REGION Network 33: ET01 - ESTADO REPOSO VACIO
   RUNG wire#powerrail
      Contact( #Mx_ET00 )
      Contact( #EstadoZona.Marcha_CBx )
      I_Contact( #EstadoZona.PerReset_CBx )
      I_Contact( #pHsMx_MQ1 )
      I_Contact( #pHsMx_MQ2 )
      wire#w1
      S_SR(operand := #Mx_ET01, r1 := wire#w2)
   END_RUNG
   RUNG wire#powerrail
      Contact( #Mx_ET51 )
      Contact( #Mx_ET151 )
      I_Contact( #Mx_ET50 )
      I_Contact( #Mx_ET150 )
      I_Contact( #Simultaneo_Mx )
      I_Contact( #EstadoVI.Descarga_Act )
      I_Contact( #pHsMx_MQ1 )
      I_Contact( #pHsMx_MQ2 )
      I_Contact( #Selec_Salida_MQ1_2 )
      I_Contact( #Selec_Salida_MQ1 )
      I_Contact( #Selec_Salida_MQ2 )
   END_RUNG wire#w1
   RUNG wire#powerrail
      Contact( #Mx_ET10 )
      Contact( #Mx_ET110 )
   END_RUNG wire#w2
   // the same network as SCL:
   IF (#Mx_ET00 AND #EstadoZona.Marcha_CBx AND NOT #EstadoZona.PerReset_CBx AND NOT #pHsMx_MQ1 AND NOT #pHsMx_MQ2) OR (#Mx_ET51 AND #Mx_ET151 AND NOT #Mx_ET50 AND NOT #Mx_ET150 AND NOT #Simultaneo_Mx AND NOT #EstadoVI.Descarga_Act AND NOT #pHsMx_MQ1 AND NOT #pHsMx_MQ2 AND NOT #Selec_Salida_MQ1_2 AND NOT #Selec_Salida_MQ1 AND NOT #Selec_Salida_MQ2) THEN
       #Mx_ET01 := TRUE;   // SR flip-flop
   END_IF;
   IF #Mx_ET10 AND #Mx_ET110 THEN #Mx_ET01 := FALSE; END_IF;
END_REGION

REGION Network 34: ET00 - ESTADO DE INICIO
   RUNG wire#powerrail
      I_Contact( #Mx_ET50 )
      I_Contact( #Mx_ET51 )
      I_Contact( #Mx_ET150 )
      I_Contact( #Mx_ET151 )
      Coil( #Aux_ET00 )
   END_RUNG
   // the same network as SCL:
   #Aux_ET00 := NOT #Mx_ET50 AND NOT #Mx_ET51 AND NOT #Mx_ET150 AND NOT #Mx_ET151;
END_REGION

REGION Network 35: ----
   RUNG wire#powerrail
      Contact( #Aux_ET00 )
      I_Contact( #Mx_ET10 )
      I_Contact( #Mx_ET11 )
      I_Contact( #Mx_ET12 )
      I_Contact( #Mx_ET110 )
      I_Contact( #Mx_ET111 )
      Coil( #Aux_ET00 )
   END_RUNG
   // the same network as SCL:
   #Aux_ET00 := #Aux_ET00 AND NOT #Mx_ET10 AND NOT #Mx_ET11 AND NOT #Mx_ET12 AND NOT #Mx_ET110 AND NOT #Mx_ET111;
END_REGION

REGION Network 36: ----
   RUNG wire#powerrail
      Contact( #Aux_ET00 )
      I_Contact( #Mx_ET00 )
      I_Contact( #Mx_ET01 )
      I_Contact( #Mx_ET02 )
      I_Contact( #Mx_ET06 )
      I_Contact( #Mx_ET07 )
      I_Contact( #Mx_ET08 )
      I_Contact( #Mx_ET09 )
      S_SR(operand := #Mx_ET00, r1 := wire#w1)
   END_RUNG
   RUNG wire#powerrail
      Contact( #Mx_ET01 )
   END_RUNG wire#w1
   RUNG wire#powerrail
      Contact( #Mx_ET06 )
   END_RUNG wire#w1
   // the same network as SCL:
   IF #Aux_ET00 AND NOT #Mx_ET00 AND NOT #Mx_ET01 AND NOT #Mx_ET02 AND NOT #Mx_ET06 AND NOT #Mx_ET07 AND NOT #Mx_ET08 AND NOT #Mx_ET09 THEN
       #Mx_ET00 := TRUE;   // SR flip-flop
   END_IF;
   IF #Mx_ET01 OR #Mx_ET06 THEN #Mx_ET00 := FALSE; END_IF;
END_REGION

REGION Network 37: CONTADOR DE SEGURIDAD DE PRESENCIA - CNTSeg_pHsMx
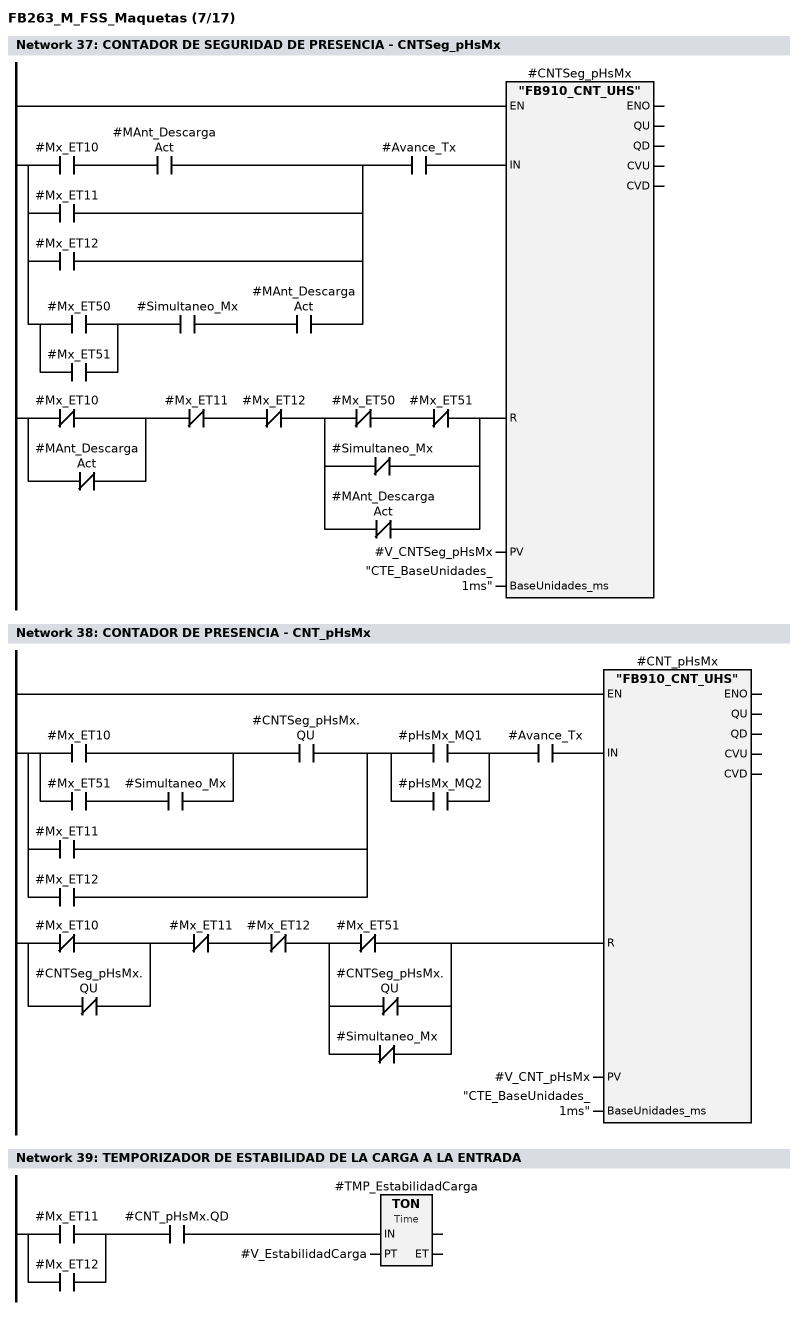
   RUNG wire#powerrail
      #CNTSeg_pHsMx(IN := wire#w3, R := wire#w6, PV := #V_CNTSeg_pHsMx, BaseUnidades_ms := "CTE_BaseUnidades_1ms", QU =>, QD =>, CVU =>, CVD =>)
   END_RUNG
   RUNG wire#powerrail
      Contact( #Mx_ET10 )
      Contact( #MAnt_DescargaAct )
      wire#w1
      Contact( #Avance_Tx )
   END_RUNG wire#w3
   RUNG wire#powerrail
      Contact( #Mx_ET11 )
   END_RUNG wire#w1
   RUNG wire#powerrail
      Contact( #Mx_ET12 )
   END_RUNG wire#w1
   RUNG wire#powerrail
      Contact( #Mx_ET50 )
      wire#w2
      Contact( #Simultaneo_Mx )
      Contact( #MAnt_DescargaAct )
   END_RUNG wire#w1
   RUNG wire#powerrail
      Contact( #Mx_ET51 )
   END_RUNG wire#w2
   RUNG wire#powerrail
      I_Contact( #Mx_ET10 )
      wire#w4
      I_Contact( #Mx_ET11 )
      I_Contact( #Mx_ET12 )
      wire#w5
      I_Contact( #Mx_ET50 )
      I_Contact( #Mx_ET51 )
   END_RUNG wire#w6
   RUNG wire#powerrail
      I_Contact( #MAnt_DescargaAct )
   END_RUNG wire#w4
   RUNG wire#w5
      I_Contact( #Simultaneo_Mx )
   END_RUNG wire#w6
   RUNG wire#w5
      I_Contact( #MAnt_DescargaAct )
   END_RUNG wire#w6
   // the same network as SCL:
   #CNTSeg_pHsMx(IN := ((#Mx_ET10 AND #MAnt_DescargaAct) OR #Mx_ET11 OR #Mx_ET12 OR ((#Mx_ET50 OR #Mx_ET51) AND #Simultaneo_Mx AND #MAnt_DescargaAct)) AND #Avance_Tx,   // "FB910_CNT_UHS"
                 R := (NOT #Mx_ET10 OR NOT #MAnt_DescargaAct) AND NOT #Mx_ET11 AND NOT #Mx_ET12 AND ((NOT #Mx_ET50 AND NOT #Mx_ET51) OR NOT #Simultaneo_Mx OR NOT #MAnt_DescargaAct),
                 PV := #V_CNTSeg_pHsMx,
                 BaseUnidades_ms := "CTE_BaseUnidades_1ms");
END_REGION

REGION Network 38: CONTADOR DE PRESENCIA - CNT_pHsMx
   RUNG wire#powerrail
      #CNT_pHsMx(IN := wire#w4, R := wire#w7, PV := #V_CNT_pHsMx, BaseUnidades_ms := "CTE_BaseUnidades_1ms", QU =>, QD =>, CVU =>, CVD =>)
   END_RUNG
   RUNG wire#powerrail
      Contact( #Mx_ET10 )
      wire#w1
      Contact( #CNTSeg_pHsMx.QU )
      wire#w2
      Contact( #pHsMx_MQ1 )
      wire#w3
      Contact( #Avance_Tx )
   END_RUNG wire#w4
   RUNG wire#powerrail
      Contact( #Mx_ET51 )
      Contact( #Simultaneo_Mx )
   END_RUNG wire#w1
   RUNG wire#powerrail
      Contact( #Mx_ET11 )
   END_RUNG wire#w2
   RUNG wire#powerrail
      Contact( #Mx_ET12 )
   END_RUNG wire#w2
   RUNG wire#w2
      Contact( #pHsMx_MQ2 )
   END_RUNG wire#w3
   RUNG wire#powerrail
      I_Contact( #Mx_ET10 )
      wire#w5
      I_Contact( #Mx_ET11 )
      I_Contact( #Mx_ET12 )
      wire#w6
      I_Contact( #Mx_ET51 )
   END_RUNG wire#w7
   RUNG wire#powerrail
      I_Contact( #CNTSeg_pHsMx.QU )
   END_RUNG wire#w5
   RUNG wire#w6
      I_Contact( #CNTSeg_pHsMx.QU )
   END_RUNG wire#w7
   RUNG wire#w6
      I_Contact( #Simultaneo_Mx )
   END_RUNG wire#w7
   // the same network as SCL:
   #CNT_pHsMx(IN := (((#Mx_ET10 OR (#Mx_ET51 AND #Simultaneo_Mx)) AND #CNTSeg_pHsMx.QU) OR #Mx_ET11 OR #Mx_ET12) AND (#pHsMx_MQ1 OR #pHsMx_MQ2) AND #Avance_Tx,   // "FB910_CNT_UHS"
              R := (NOT #Mx_ET10 OR NOT #CNTSeg_pHsMx.QU) AND NOT #Mx_ET11 AND NOT #Mx_ET12 AND (NOT #Mx_ET51 OR NOT #CNTSeg_pHsMx.QU OR NOT #Simultaneo_Mx),
              PV := #V_CNT_pHsMx,
              BaseUnidades_ms := "CTE_BaseUnidades_1ms");
END_REGION

REGION Network 39: TEMPORIZADOR DE ESTABILIDAD DE LA CARGA A LA ENTRADA
   RUNG wire#powerrail
      Contact( #Mx_ET11 )
      wire#w1
      Contact( #CNT_pHsMx.QD )
      { S7_Templates := "time_type := Time" } #TMP_EstabilidadCarga.TON(pt := #V_EstabilidadCarga, et =>)
   END_RUNG
   RUNG wire#powerrail
      Contact( #Mx_ET12 )
   END_RUNG wire#w1
   // the same network as SCL:
   #TMP_EstabilidadCarga(IN := (#Mx_ET11 OR #Mx_ET12) AND #CNT_pHsMx.QD, PT := #V_EstabilidadCarga);   // TON
END_REGION

REGION Network 40: DETERMINA PASO ET10 - ET11 (Nota: Control de Tiempo para dar el FTF a la Mesa Anterior)
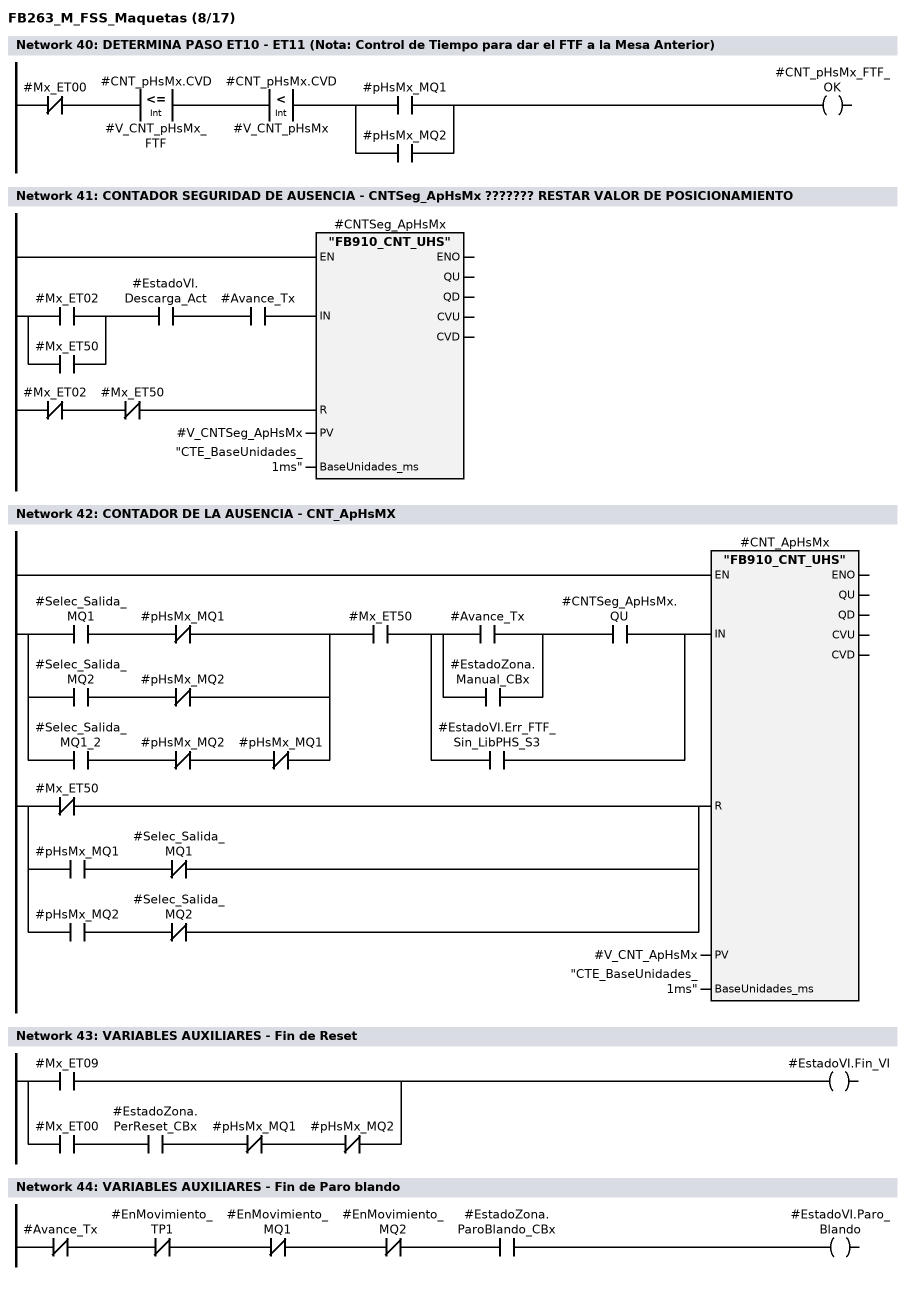
   RUNG wire#powerrail
      I_Contact( #Mx_ET00 )
      { S7_Templates := "SrcType := Int" } LE_Contact(in1 := #CNT_pHsMx.CVD, in2 := #V_CNT_pHsMx_FTF)
      { S7_Templates := "SrcType := Int" } LT_Contact(in1 := #CNT_pHsMx.CVD, in2 := #V_CNT_pHsMx)
      wire#w1
      Contact( #pHsMx_MQ1 )
      wire#w2
      Coil( #CNT_pHsMx_FTF_OK )
   END_RUNG
   RUNG wire#w1
      Contact( #pHsMx_MQ2 )
   END_RUNG wire#w2
   // the same network as SCL:
   #CNT_pHsMx_FTF_OK := NOT #Mx_ET00 AND (#CNT_pHsMx.CVD <= #V_CNT_pHsMx_FTF) AND (#CNT_pHsMx.CVD < #V_CNT_pHsMx) AND (#pHsMx_MQ1 OR #pHsMx_MQ2);
END_REGION

REGION Network 41: CONTADOR SEGURIDAD DE AUSENCIA - CNTSeg_ApHsMx ??????? RESTAR VALOR DE POSICIONAMIENTO
   RUNG wire#powerrail
      #CNTSeg_ApHsMx(IN := wire#w2, R := wire#w3, PV := #V_CNTSeg_ApHsMx, BaseUnidades_ms := "CTE_BaseUnidades_1ms", QU =>, QD =>, CVU =>, CVD =>)
   END_RUNG
   RUNG wire#powerrail
      Contact( #Mx_ET02 )
      wire#w1
      Contact( #EstadoVI.Descarga_Act )
      Contact( #Avance_Tx )
   END_RUNG wire#w2
   RUNG wire#powerrail
      Contact( #Mx_ET50 )
   END_RUNG wire#w1
   RUNG wire#powerrail
      I_Contact( #Mx_ET02 )
      I_Contact( #Mx_ET50 )
   END_RUNG wire#w3
   // the same network as SCL:
   #CNTSeg_ApHsMx(IN := (#Mx_ET02 OR #Mx_ET50) AND #EstadoVI.Descarga_Act AND #Avance_Tx,   // "FB910_CNT_UHS"
                  R := NOT #Mx_ET02 AND NOT #Mx_ET50,
                  PV := #V_CNTSeg_ApHsMx,
                  BaseUnidades_ms := "CTE_BaseUnidades_1ms");
END_REGION

REGION Network 42: CONTADOR DE LA AUSENCIA - CNT_ApHsMX
   RUNG wire#powerrail
      #CNT_ApHsMx(IN := wire#w4, R := wire#w5, PV := #V_CNT_ApHsMx, BaseUnidades_ms := "CTE_BaseUnidades_1ms", QU =>, QD =>, CVU =>, CVD =>)
   END_RUNG
   RUNG wire#powerrail
      Contact( #Selec_Salida_MQ1 )
      I_Contact( #pHsMx_MQ1 )
      wire#w1
      Contact( #Mx_ET50 )
      wire#w2
      Contact( #Avance_Tx )
      wire#w3
      Contact( #CNTSeg_ApHsMx.QU )
   END_RUNG wire#w4
   RUNG wire#powerrail
      Contact( #Selec_Salida_MQ2 )
      I_Contact( #pHsMx_MQ2 )
   END_RUNG wire#w1
   RUNG wire#powerrail
      Contact( #Selec_Salida_MQ1_2 )
      I_Contact( #pHsMx_MQ2 )
      I_Contact( #pHsMx_MQ1 )
   END_RUNG wire#w1
   RUNG wire#w2
      Contact( #EstadoZona.Manual_CBx )
   END_RUNG wire#w3
   RUNG wire#w2
      Contact( #EstadoVI.Err_FTF_Sin_LibPHS_S3 )
   END_RUNG wire#w4
   RUNG wire#powerrail
      I_Contact( #Mx_ET50 )
   END_RUNG wire#w5
   RUNG wire#powerrail
      Contact( #pHsMx_MQ1 )
      I_Contact( #Selec_Salida_MQ1 )
   END_RUNG wire#w5
   RUNG wire#powerrail
      Contact( #pHsMx_MQ2 )
      I_Contact( #Selec_Salida_MQ2 )
   END_RUNG wire#w5
   // the same network as SCL:
   #CNT_ApHsMx(IN := ((#Selec_Salida_MQ1 AND NOT #pHsMx_MQ1) OR (#Selec_Salida_MQ2 AND NOT #pHsMx_MQ2) OR (#Selec_Salida_MQ1_2 AND NOT #pHsMx_MQ2 AND NOT #pHsMx_MQ1)) AND #Mx_ET50 AND (((#Avance_Tx OR #EstadoZona.Manual_CBx) AND #CNTSeg_ApHsMx.QU) OR #EstadoVI.Err_FTF_Sin_LibPHS_S3),   // "FB910_CNT_UHS"
               R := NOT #Mx_ET50 OR (#pHsMx_MQ1 AND NOT #Selec_Salida_MQ1) OR (#pHsMx_MQ2 AND NOT #Selec_Salida_MQ2),
               PV := #V_CNT_ApHsMx,
               BaseUnidades_ms := "CTE_BaseUnidades_1ms");
END_REGION

REGION Network 43: VARIABLES AUXILIARES - Fin de Reset
   RUNG wire#powerrail
      Contact( #Mx_ET09 )
      wire#w1
      Coil( #EstadoVI.Fin_VI )
   END_RUNG
   RUNG wire#powerrail
      Contact( #Mx_ET00 )
      Contact( #EstadoZona.PerReset_CBx )
      I_Contact( #pHsMx_MQ1 )
      I_Contact( #pHsMx_MQ2 )
   END_RUNG wire#w1
   // the same network as SCL:
   #EstadoVI.Fin_VI := #Mx_ET09 OR (#Mx_ET00 AND #EstadoZona.PerReset_CBx AND NOT #pHsMx_MQ1 AND NOT #pHsMx_MQ2);
END_REGION

REGION Network 44: VARIABLES AUXILIARES - Fin de Paro blando
   RUNG wire#powerrail
      I_Contact( #Avance_Tx )
      I_Contact( #EnMovimiento_TP1 )
      I_Contact( #EnMovimiento_MQ1 )
      I_Contact( #EnMovimiento_MQ2 )
      Contact( #EstadoZona.ParoBlando_CBx )
      Coil( #EstadoVI.Paro_Blando )
   END_RUNG
   // the same network as SCL:
   #EstadoVI.Paro_Blando := NOT #Avance_Tx AND NOT #EnMovimiento_TP1 AND NOT #EnMovimiento_MQ1 AND NOT #EnMovimiento_MQ2 AND #EstadoZona.ParoBlando_CBx;
END_REGION

REGION Network 45: VARIABLES AUXILIARES - Permiso de Entrada - PTF_MAnt_Mx
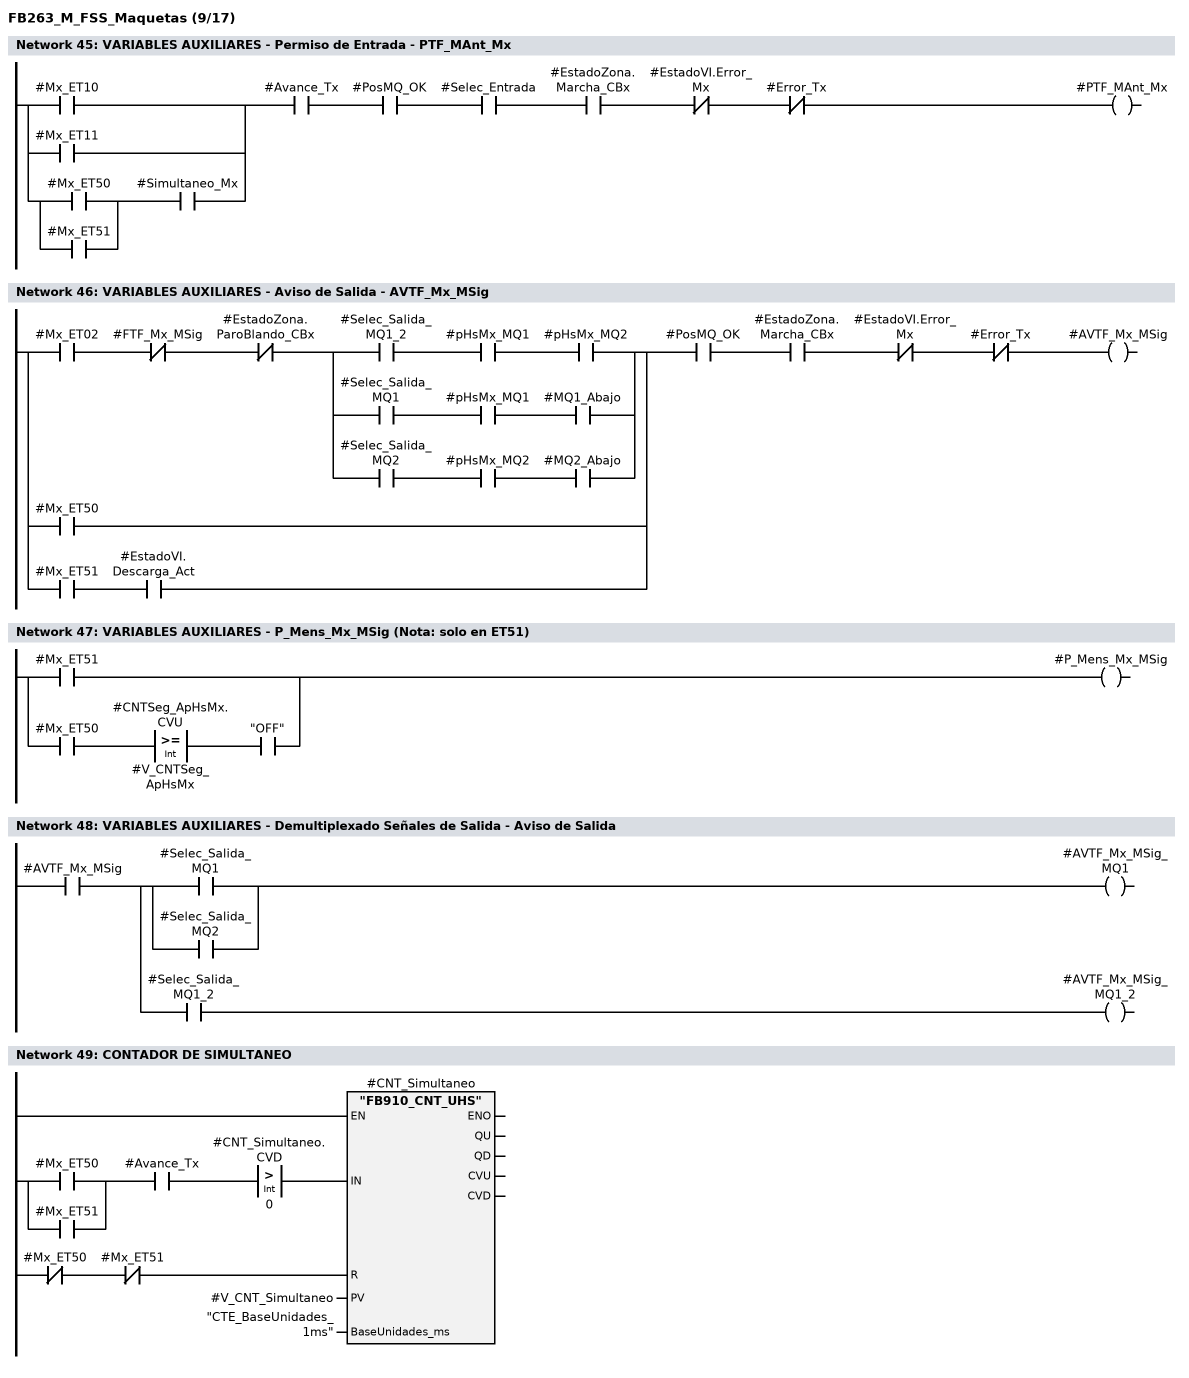
   RUNG wire#powerrail
      Contact( #Mx_ET10 )
      wire#w1
      Contact( #Avance_Tx )
      Contact( #PosMQ_OK )
      Contact( #Selec_Entrada )
      Contact( #EstadoZona.Marcha_CBx )
      I_Contact( #EstadoVI.Error_Mx )
      I_Contact( #Error_Tx )
      Coil( #PTF_MAnt_Mx )
   END_RUNG
   RUNG wire#powerrail
      Contact( #Mx_ET11 )
   END_RUNG wire#w1
   RUNG wire#powerrail
      Contact( #Mx_ET50 )
      wire#w2
      Contact( #Simultaneo_Mx )
   END_RUNG wire#w1
   RUNG wire#powerrail
      Contact( #Mx_ET51 )
   END_RUNG wire#w2
   // the same network as SCL:
   #PTF_MAnt_Mx := (#Mx_ET10 OR #Mx_ET11 OR ((#Mx_ET50 OR #Mx_ET51) AND #Simultaneo_Mx)) AND #Avance_Tx AND #PosMQ_OK AND #Selec_Entrada AND #EstadoZona.Marcha_CBx AND NOT #EstadoVI.Error_Mx AND NOT #Error_Tx;
END_REGION

REGION Network 46: VARIABLES AUXILIARES - Aviso de Salida - AVTF_Mx_MSig
   RUNG wire#powerrail
      Contact( #Mx_ET02 )
      I_Contact( #FTF_Mx_MSig )
      I_Contact( #EstadoZona.ParoBlando_CBx )
      wire#w1
      Contact( #Selec_Salida_MQ1_2 )
      Contact( #pHsMx_MQ1 )
      Contact( #pHsMx_MQ2 )
      wire#w2
      Contact( #PosMQ_OK )
      Contact( #EstadoZona.Marcha_CBx )
      I_Contact( #EstadoVI.Error_Mx )
      I_Contact( #Error_Tx )
      Coil( #AVTF_Mx_MSig )
   END_RUNG
   RUNG wire#w1
      Contact( #Selec_Salida_MQ1 )
      Contact( #pHsMx_MQ1 )
      Contact( #MQ1_Abajo )
   END_RUNG wire#w2
   RUNG wire#w1
      Contact( #Selec_Salida_MQ2 )
      Contact( #pHsMx_MQ2 )
      Contact( #MQ2_Abajo )
   END_RUNG wire#w2
   RUNG wire#powerrail
      Contact( #Mx_ET50 )
   END_RUNG wire#w2
   RUNG wire#powerrail
      Contact( #Mx_ET51 )
      Contact( #EstadoVI.Descarga_Act )
   END_RUNG wire#w2
   // the same network as SCL:
   #AVTF_Mx_MSig := ((#Mx_ET02 AND NOT #FTF_Mx_MSig AND NOT #EstadoZona.ParoBlando_CBx AND ((#Selec_Salida_MQ1_2 AND #pHsMx_MQ1 AND #pHsMx_MQ2) OR (#Selec_Salida_MQ1 AND #pHsMx_MQ1 AND #MQ1_Abajo) OR (#Selec_Salida_MQ2 AND #pHsMx_MQ2 AND #MQ2_Abajo))) OR #Mx_ET50 OR (#Mx_ET51 AND #EstadoVI.Descarga_Act)) AND #PosMQ_OK AND #EstadoZona.Marcha_CBx AND NOT #EstadoVI.Error_Mx AND NOT #Error_Tx;
END_REGION

REGION Network 47: VARIABLES AUXILIARES - P_Mens_Mx_MSig (Nota: solo en ET51)
   RUNG wire#powerrail
      Contact( #Mx_ET51 )
      wire#w1
      Coil( #P_Mens_Mx_MSig )
   END_RUNG
   RUNG wire#powerrail
      Contact( #Mx_ET50 )
      { S7_Templates := "SrcType := Int" } GE_Contact(in1 := #CNTSeg_ApHsMx.CVU, in2 := #V_CNTSeg_ApHsMx)
      Contact( "OFF" )
   END_RUNG wire#w1
   // the same network as SCL:
   #P_Mens_Mx_MSig := #Mx_ET51 OR (#Mx_ET50 AND (#CNTSeg_ApHsMx.CVU >= #V_CNTSeg_ApHsMx) AND "OFF");
END_REGION

REGION Network 48: VARIABLES AUXILIARES - Demultiplexado Señales de Salida - Aviso de Salida
   RUNG wire#powerrail
      Contact( #AVTF_Mx_MSig )
      wire#w1
      Contact( #Selec_Salida_MQ1 )
      wire#w2
      Coil( #AVTF_Mx_MSig_MQ1 )
   END_RUNG
   RUNG wire#w1
      Contact( #Selec_Salida_MQ2 )
   END_RUNG wire#w2
   RUNG wire#w1
      Contact( #Selec_Salida_MQ1_2 )
      Coil( #AVTF_Mx_MSig_MQ1_2 )
   END_RUNG
   // the same network as SCL:
   #AVTF_Mx_MSig_MQ1 := #AVTF_Mx_MSig AND (#Selec_Salida_MQ1 OR #Selec_Salida_MQ2);
   #AVTF_Mx_MSig_MQ1_2 := #AVTF_Mx_MSig AND #Selec_Salida_MQ1_2;
END_REGION

REGION Network 49: CONTADOR DE SIMULTANEO
   RUNG wire#powerrail
      #CNT_Simultaneo(IN := wire#w2, R := wire#w3, PV := #V_CNT_Simultaneo, BaseUnidades_ms := "CTE_BaseUnidades_1ms", QU =>, QD =>, CVU =>, CVD =>)
   END_RUNG
   RUNG wire#powerrail
      Contact( #Mx_ET50 )
      wire#w1
      Contact( #Avance_Tx )
      { S7_Templates := "SrcType := Int" } GT_Contact(in1 := #CNT_Simultaneo.CVD, in2 := 0)
   END_RUNG wire#w2
   RUNG wire#powerrail
      Contact( #Mx_ET51 )
   END_RUNG wire#w1
   RUNG wire#powerrail
      I_Contact( #Mx_ET50 )
      I_Contact( #Mx_ET51 )
   END_RUNG wire#w3
   // the same network as SCL:
   #CNT_Simultaneo(IN := (#Mx_ET50 OR #Mx_ET51) AND #Avance_Tx AND (#CNT_Simultaneo.CVD > 0),   // "FB910_CNT_UHS"
                   R := NOT #Mx_ET50 AND NOT #Mx_ET51,
                   PV := #V_CNT_Simultaneo,
                   BaseUnidades_ms := "CTE_BaseUnidades_1ms");
END_REGION

REGION Network 50: CONTROL DE MOVIMIENTO SIMULTANEO
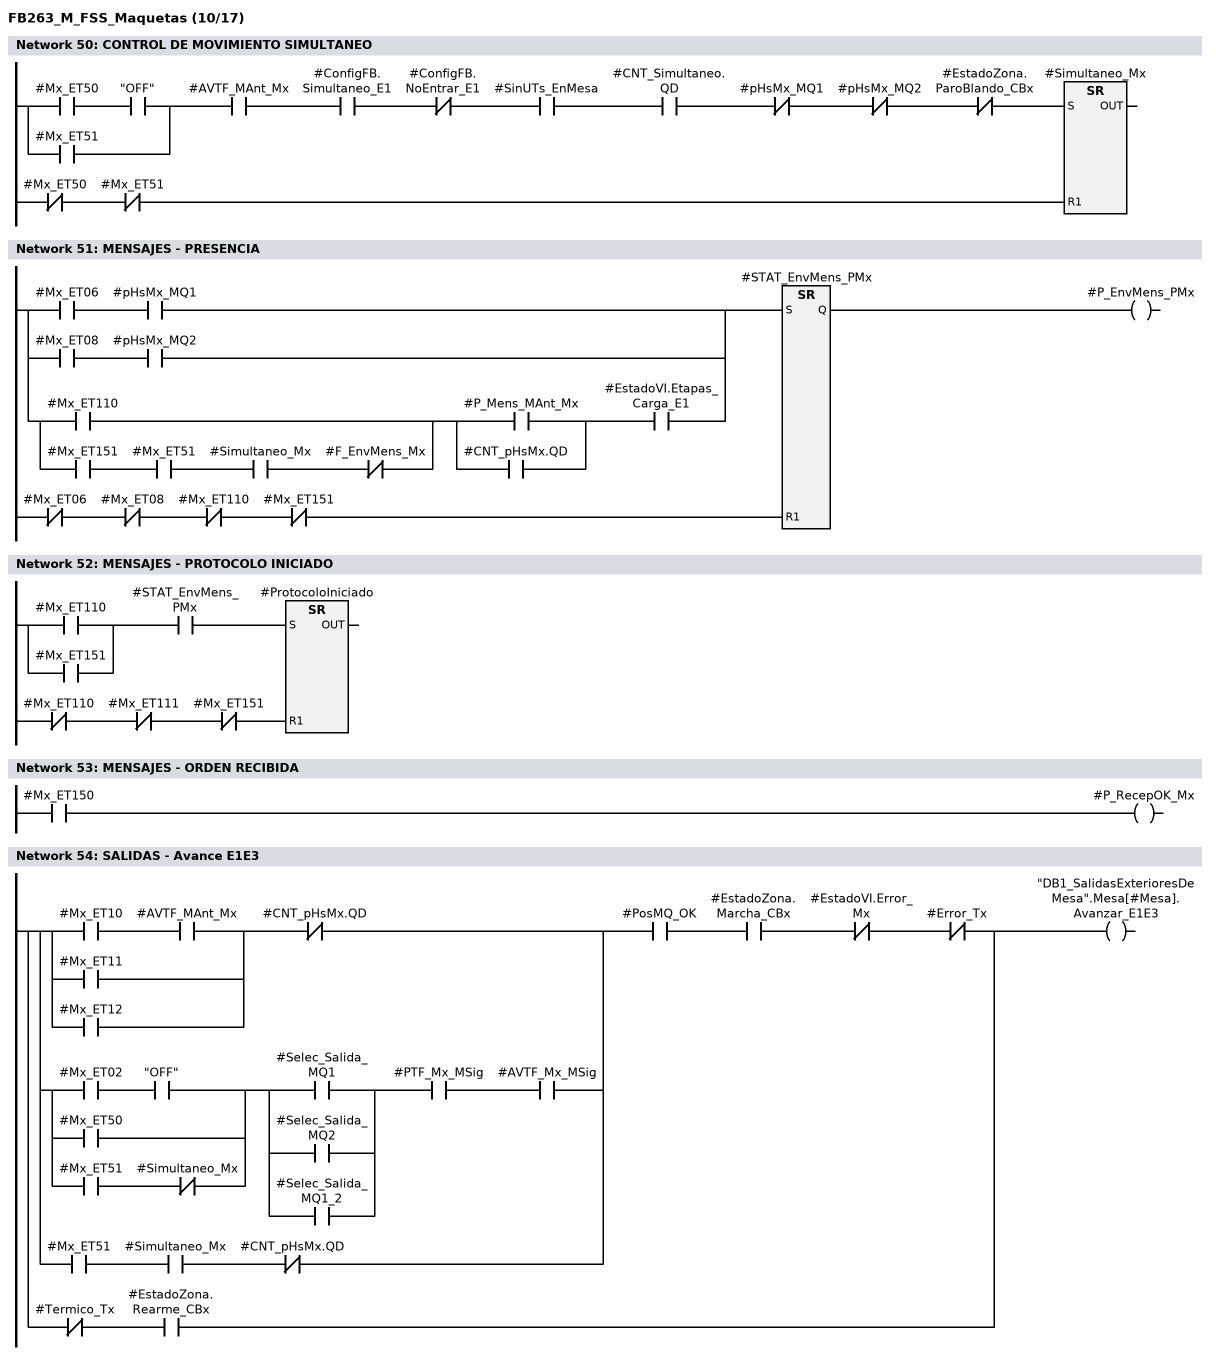
   RUNG wire#powerrail
      Contact( #Mx_ET50 )
      Contact( "OFF" )
      wire#w1
      Contact( #AVTF_MAnt_Mx )
      Contact( #ConfigFB.Simultaneo_E1 )
      I_Contact( #ConfigFB.NoEntrar_E1 )
      Contact( #SinUTs_EnMesa )
      Contact( #CNT_Simultaneo.QD )
      I_Contact( #pHsMx_MQ1 )
      I_Contact( #pHsMx_MQ2 )
      I_Contact( #EstadoZona.ParoBlando_CBx )
      S_SR(operand := #Simultaneo_Mx, r1 := wire#w2)
   END_RUNG
   RUNG wire#powerrail
      Contact( #Mx_ET51 )
   END_RUNG wire#w1
   RUNG wire#powerrail
      I_Contact( #Mx_ET50 )
      I_Contact( #Mx_ET51 )
   END_RUNG wire#w2
   // the same network as SCL:
   IF ((#Mx_ET50 AND "OFF") OR #Mx_ET51) AND #AVTF_MAnt_Mx AND #ConfigFB.Simultaneo_E1 AND NOT #ConfigFB.NoEntrar_E1 AND #SinUTs_EnMesa AND #CNT_Simultaneo.QD AND NOT #pHsMx_MQ1 AND NOT #pHsMx_MQ2 AND NOT #EstadoZona.ParoBlando_CBx THEN
       #Simultaneo_Mx := TRUE;   // SR flip-flop
   END_IF;
   IF NOT #Mx_ET50 AND NOT #Mx_ET51 THEN #Simultaneo_Mx := FALSE; END_IF;
END_REGION

REGION Network 51: MENSAJES - PRESENCIA
   RUNG wire#powerrail
      Contact( #Mx_ET06 )
      Contact( #pHsMx_MQ1 )
      wire#w1
      S_SR(operand := #STAT_EnvMens_PMx, r1 := wire#w4)
      Coil( #P_EnvMens_PMx )
   END_RUNG
   RUNG wire#powerrail
      Contact( #Mx_ET08 )
      Contact( #pHsMx_MQ2 )
   END_RUNG wire#w1
   RUNG wire#powerrail
      Contact( #Mx_ET110 )
      wire#w2
      Contact( #P_Mens_MAnt_Mx )
      wire#w3
      Contact( #EstadoVI.Etapas_Carga_E1 )
   END_RUNG wire#w1
   RUNG wire#powerrail
      Contact( #Mx_ET151 )
      Contact( #Mx_ET51 )
      Contact( #Simultaneo_Mx )
      I_Contact( #F_EnvMens_Mx )
   END_RUNG wire#w2
   RUNG wire#w2
      Contact( #CNT_pHsMx.QD )
   END_RUNG wire#w3
   RUNG wire#powerrail
      I_Contact( #Mx_ET06 )
      I_Contact( #Mx_ET08 )
      I_Contact( #Mx_ET110 )
      I_Contact( #Mx_ET151 )
   END_RUNG wire#w4
   // the same network as SCL:
   IF (#Mx_ET06 AND #pHsMx_MQ1) OR (#Mx_ET08 AND #pHsMx_MQ2) OR ((#Mx_ET110 OR (#Mx_ET151 AND #Mx_ET51 AND #Simultaneo_Mx AND NOT #F_EnvMens_Mx)) AND (#P_Mens_MAnt_Mx OR #CNT_pHsMx.QD) AND #EstadoVI.Etapas_Carga_E1) THEN
       #STAT_EnvMens_PMx := TRUE;   // SR flip-flop
   END_IF;
   IF NOT #Mx_ET06 AND NOT #Mx_ET08 AND NOT #Mx_ET110 AND NOT #Mx_ET151 THEN
       #STAT_EnvMens_PMx := FALSE;
   END_IF;
   #P_EnvMens_PMx := #STAT_EnvMens_PMx;
END_REGION

REGION Network 52: MENSAJES - PROTOCOLO INICIADO
   RUNG wire#powerrail
      Contact( #Mx_ET110 )
      wire#w1
      Contact( #STAT_EnvMens_PMx )
      S_SR(operand := #ProtocoloIniciado, r1 := wire#w2)
   END_RUNG
   RUNG wire#powerrail
      Contact( #Mx_ET151 )
   END_RUNG wire#w1
   RUNG wire#powerrail
      I_Contact( #Mx_ET110 )
      I_Contact( #Mx_ET111 )
      I_Contact( #Mx_ET151 )
   END_RUNG wire#w2
   // the same network as SCL:
   IF (#Mx_ET110 OR #Mx_ET151) AND #STAT_EnvMens_PMx THEN
       #ProtocoloIniciado := TRUE;   // SR flip-flop
   END_IF;
   IF NOT #Mx_ET110 AND NOT #Mx_ET111 AND NOT #Mx_ET151 THEN #ProtocoloIniciado := FALSE; END_IF;
END_REGION

REGION Network 53: MENSAJES - ORDEN RECIBIDA
   RUNG wire#powerrail
      Contact( #Mx_ET150 )
      Coil( #P_RecepOK_Mx )
   END_RUNG
   // the same network as SCL:
   #P_RecepOK_Mx := #Mx_ET150;
END_REGION

REGION Network 54: SALIDAS - Avance E1E3
   RUNG wire#powerrail
      Contact( #Mx_ET10 )
      Contact( #AVTF_MAnt_Mx )
      wire#w1
      I_Contact( #CNT_pHsMx.QD )
      wire#w2
      Contact( #PosMQ_OK )
      Contact( #EstadoZona.Marcha_CBx )
      I_Contact( #EstadoVI.Error_Mx )
      I_Contact( #Error_Tx )
      wire#w5
      Coil( "DB1_SalidasExterioresDeMesa".Mesa[#Mesa].Avanzar_E1E3 )
   END_RUNG
   RUNG wire#powerrail
      Contact( #Mx_ET11 )
   END_RUNG wire#w1
   RUNG wire#powerrail
      Contact( #Mx_ET12 )
   END_RUNG wire#w1
   RUNG wire#powerrail
      Contact( #Mx_ET02 )
      Contact( "OFF" )
      wire#w3
      Contact( #Selec_Salida_MQ1 )
      wire#w4
      Contact( #PTF_Mx_MSig )
      Contact( #AVTF_Mx_MSig )
   END_RUNG wire#w2
   RUNG wire#powerrail
      Contact( #Mx_ET50 )
   END_RUNG wire#w3
   RUNG wire#powerrail
      Contact( #Mx_ET51 )
      I_Contact( #Simultaneo_Mx )
   END_RUNG wire#w3
   RUNG wire#w3
      Contact( #Selec_Salida_MQ2 )
   END_RUNG wire#w4
   RUNG wire#w3
      Contact( #Selec_Salida_MQ1_2 )
   END_RUNG wire#w4
   RUNG wire#powerrail
      Contact( #Mx_ET51 )
      Contact( #Simultaneo_Mx )
      I_Contact( #CNT_pHsMx.QD )
   END_RUNG wire#w2
   RUNG wire#powerrail
      I_Contact( #Termico_Tx )
      Contact( #EstadoZona.Rearme_CBx )
   END_RUNG wire#w5
   // the same network as SCL:
   "DB1_SalidasExterioresDeMesa".Mesa[#Mesa].Avanzar_E1E3 := (((((#Mx_ET10 AND #AVTF_MAnt_Mx) OR #Mx_ET11 OR #Mx_ET12) AND NOT #CNT_pHsMx.QD) OR (((#Mx_ET02 AND "OFF") OR #Mx_ET50 OR (#Mx_ET51 AND NOT #Simultaneo_Mx)) AND (#Selec_Salida_MQ1 OR #Selec_Salida_MQ2 OR #Selec_Salida_MQ1_2) AND #PTF_Mx_MSig AND #AVTF_Mx_MSig) OR (#Mx_ET51 AND #Simultaneo_Mx AND NOT #CNT_pHsMx.QD)) AND #PosMQ_OK AND #EstadoZona.Marcha_CBx AND NOT #EstadoVI.Error_Mx AND NOT #Error_Tx) OR (NOT #Termico_Tx AND #EstadoZona.Rearme_CBx);
END_REGION

REGION Network 55: SALIDAS - Subir Tope (TP1)
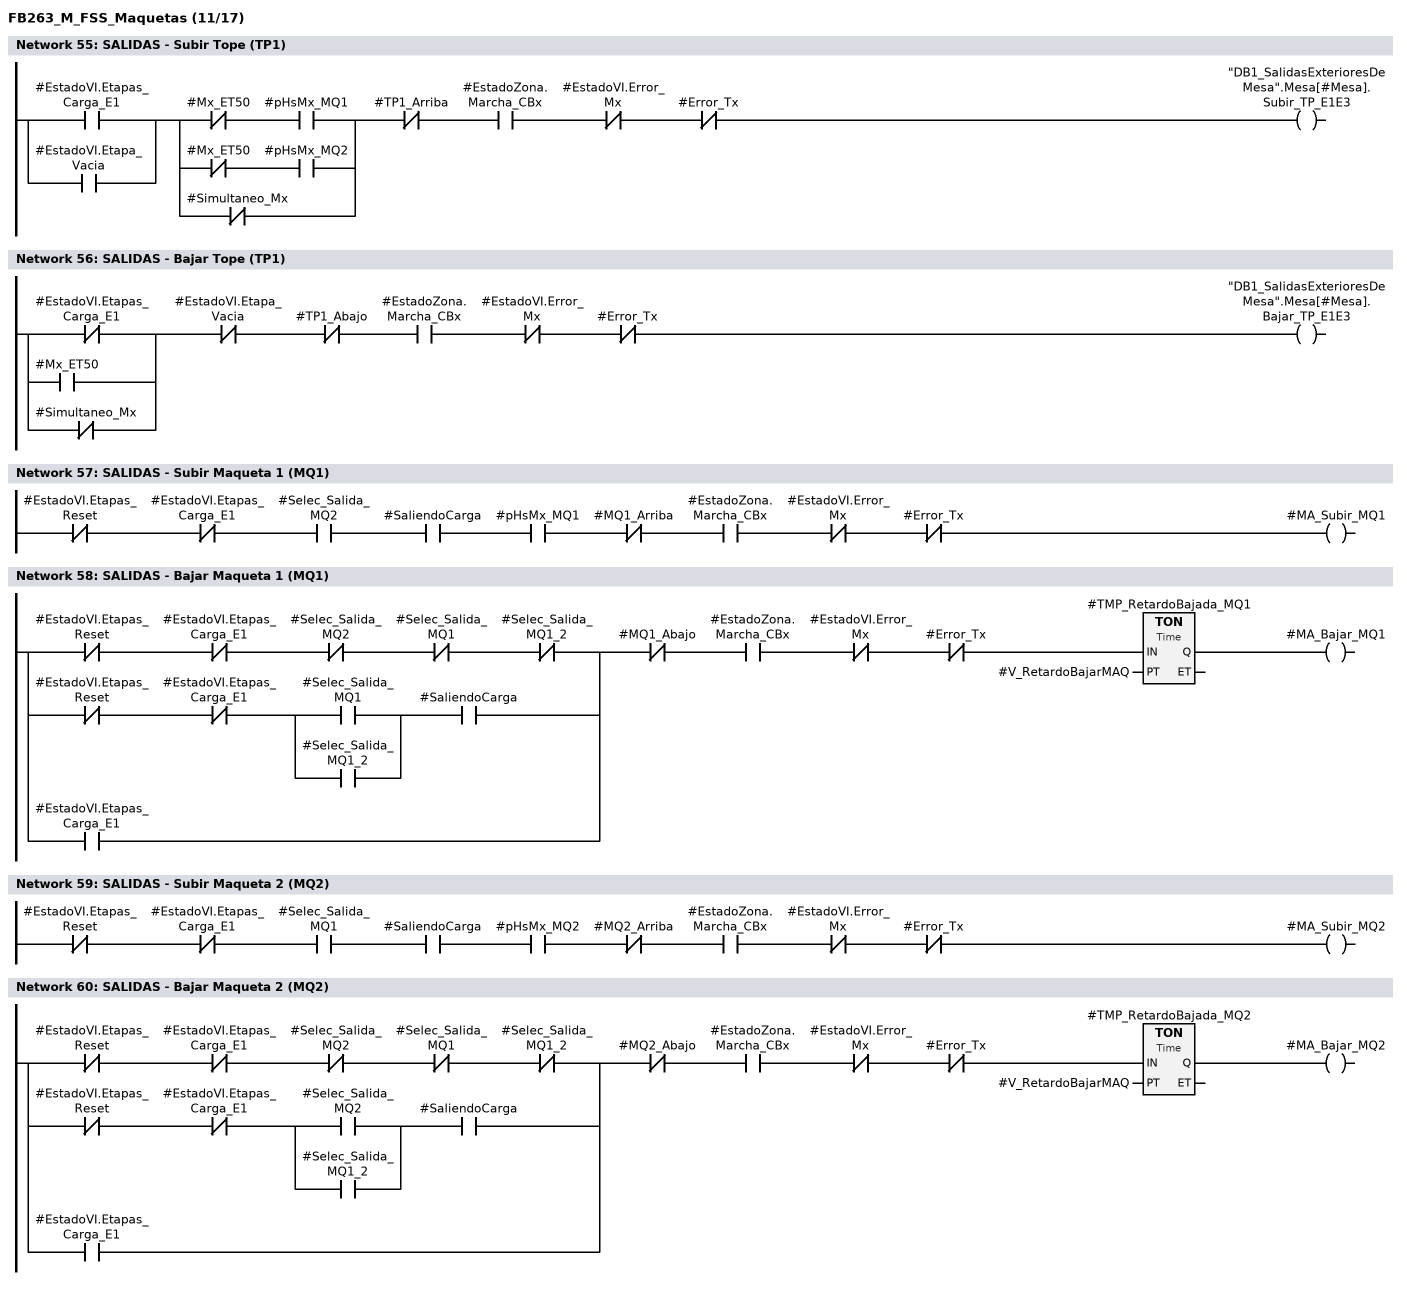
   RUNG wire#powerrail
      Contact( #EstadoVI.Etapas_Carga_E1 )
      wire#w1
      I_Contact( #Mx_ET50 )
      Contact( #pHsMx_MQ1 )
      wire#w2
      I_Contact( #TP1_Arriba )
      Contact( #EstadoZona.Marcha_CBx )
      I_Contact( #EstadoVI.Error_Mx )
      I_Contact( #Error_Tx )
      Coil( "DB1_SalidasExterioresDeMesa".Mesa[#Mesa].Subir_TP_E1E3 )
   END_RUNG
   RUNG wire#powerrail
      Contact( #EstadoVI.Etapa_Vacia )
   END_RUNG wire#w1
   RUNG wire#w1
      I_Contact( #Mx_ET50 )
      Contact( #pHsMx_MQ2 )
   END_RUNG wire#w2
   RUNG wire#w1
      I_Contact( #Simultaneo_Mx )
   END_RUNG wire#w2
   // the same network as SCL:
   "DB1_SalidasExterioresDeMesa".Mesa[#Mesa].Subir_TP_E1E3 := (#EstadoVI.Etapas_Carga_E1 OR #EstadoVI.Etapa_Vacia) AND ((NOT #Mx_ET50 AND #pHsMx_MQ1) OR (NOT #Mx_ET50 AND #pHsMx_MQ2) OR NOT #Simultaneo_Mx) AND NOT #TP1_Arriba AND #EstadoZona.Marcha_CBx AND NOT #EstadoVI.Error_Mx AND NOT #Error_Tx;
END_REGION

REGION Network 56: SALIDAS - Bajar Tope (TP1)
   RUNG wire#powerrail
      I_Contact( #EstadoVI.Etapas_Carga_E1 )
      wire#w1
      I_Contact( #EstadoVI.Etapa_Vacia )
      I_Contact( #TP1_Abajo )
      Contact( #EstadoZona.Marcha_CBx )
      I_Contact( #EstadoVI.Error_Mx )
      I_Contact( #Error_Tx )
      Coil( "DB1_SalidasExterioresDeMesa".Mesa[#Mesa].Bajar_TP_E1E3 )
   END_RUNG
   RUNG wire#powerrail
      Contact( #Mx_ET50 )
   END_RUNG wire#w1
   RUNG wire#powerrail
      I_Contact( #Simultaneo_Mx )
   END_RUNG wire#w1
   // the same network as SCL:
   "DB1_SalidasExterioresDeMesa".Mesa[#Mesa].Bajar_TP_E1E3 := (NOT #EstadoVI.Etapas_Carga_E1 OR #Mx_ET50 OR NOT #Simultaneo_Mx) AND NOT #EstadoVI.Etapa_Vacia AND NOT #TP1_Abajo AND #EstadoZona.Marcha_CBx AND NOT #EstadoVI.Error_Mx AND NOT #Error_Tx;
END_REGION

REGION Network 57: SALIDAS - Subir Maqueta 1 (MQ1)
   RUNG wire#powerrail
      I_Contact( #EstadoVI.Etapas_Reset )
      I_Contact( #EstadoVI.Etapas_Carga_E1 )
      Contact( #Selec_Salida_MQ2 )
      Contact( #SaliendoCarga )
      Contact( #pHsMx_MQ1 )
      I_Contact( #MQ1_Arriba )
      Contact( #EstadoZona.Marcha_CBx )
      I_Contact( #EstadoVI.Error_Mx )
      I_Contact( #Error_Tx )
      Coil( #MA_Subir_MQ1 )
   END_RUNG
   // the same network as SCL:
   #MA_Subir_MQ1 := NOT #EstadoVI.Etapas_Reset AND NOT #EstadoVI.Etapas_Carga_E1 AND #Selec_Salida_MQ2 AND #SaliendoCarga AND #pHsMx_MQ1 AND NOT #MQ1_Arriba AND #EstadoZona.Marcha_CBx AND NOT #EstadoVI.Error_Mx AND NOT #Error_Tx;
END_REGION

REGION Network 58: SALIDAS - Bajar Maqueta 1 (MQ1)
   RUNG wire#powerrail
      I_Contact( #EstadoVI.Etapas_Reset )
      I_Contact( #EstadoVI.Etapas_Carga_E1 )
      I_Contact( #Selec_Salida_MQ2 )
      I_Contact( #Selec_Salida_MQ1 )
      I_Contact( #Selec_Salida_MQ1_2 )
      wire#w1
      I_Contact( #MQ1_Abajo )
      Contact( #EstadoZona.Marcha_CBx )
      I_Contact( #EstadoVI.Error_Mx )
      I_Contact( #Error_Tx )
      { S7_Templates := "time_type := Time" } #TMP_RetardoBajada_MQ1.TON(pt := #V_RetardoBajarMAQ, et =>)
      Coil( #MA_Bajar_MQ1 )
   END_RUNG
   RUNG wire#powerrail
      I_Contact( #EstadoVI.Etapas_Reset )
      I_Contact( #EstadoVI.Etapas_Carga_E1 )
      wire#w2
      Contact( #Selec_Salida_MQ1 )
      wire#w3
      Contact( #SaliendoCarga )
   END_RUNG wire#w1
   RUNG wire#w2
      Contact( #Selec_Salida_MQ1_2 )
   END_RUNG wire#w3
   RUNG wire#powerrail
      Contact( #EstadoVI.Etapas_Carga_E1 )
   END_RUNG wire#w1
   // the same network as SCL:
   #TMP_RetardoBajada_MQ1(IN := ((NOT #EstadoVI.Etapas_Reset AND NOT #EstadoVI.Etapas_Carga_E1 AND NOT #Selec_Salida_MQ2 AND NOT #Selec_Salida_MQ1 AND NOT #Selec_Salida_MQ1_2) OR (NOT #EstadoVI.Etapas_Reset AND NOT #EstadoVI.Etapas_Carga_E1 AND (#Selec_Salida_MQ1 OR #Selec_Salida_MQ1_2) AND #SaliendoCarga) OR #EstadoVI.Etapas_Carga_E1) AND NOT #MQ1_Abajo AND #EstadoZona.Marcha_CBx AND NOT #EstadoVI.Error_Mx AND NOT #Error_Tx,   // TON
                          PT := #V_RetardoBajarMAQ);
   #MA_Bajar_MQ1 := #TMP_RetardoBajada_MQ1.Q;
END_REGION

REGION Network 59: SALIDAS - Subir Maqueta 2 (MQ2)
   RUNG wire#powerrail
      I_Contact( #EstadoVI.Etapas_Reset )
      I_Contact( #EstadoVI.Etapas_Carga_E1 )
      Contact( #Selec_Salida_MQ1 )
      Contact( #SaliendoCarga )
      Contact( #pHsMx_MQ2 )
      I_Contact( #MQ2_Arriba )
      Contact( #EstadoZona.Marcha_CBx )
      I_Contact( #EstadoVI.Error_Mx )
      I_Contact( #Error_Tx )
      Coil( #MA_Subir_MQ2 )
   END_RUNG
   // the same network as SCL:
   #MA_Subir_MQ2 := NOT #EstadoVI.Etapas_Reset AND NOT #EstadoVI.Etapas_Carga_E1 AND #Selec_Salida_MQ1 AND #SaliendoCarga AND #pHsMx_MQ2 AND NOT #MQ2_Arriba AND #EstadoZona.Marcha_CBx AND NOT #EstadoVI.Error_Mx AND NOT #Error_Tx;
END_REGION

REGION Network 60: SALIDAS - Bajar Maqueta 2 (MQ2)
   RUNG wire#powerrail
      I_Contact( #EstadoVI.Etapas_Reset )
      I_Contact( #EstadoVI.Etapas_Carga_E1 )
      I_Contact( #Selec_Salida_MQ2 )
      I_Contact( #Selec_Salida_MQ1 )
      I_Contact( #Selec_Salida_MQ1_2 )
      wire#w1
      I_Contact( #MQ2_Abajo )
      Contact( #EstadoZona.Marcha_CBx )
      I_Contact( #EstadoVI.Error_Mx )
      I_Contact( #Error_Tx )
      { S7_Templates := "time_type := Time" } #TMP_RetardoBajada_MQ2.TON(pt := #V_RetardoBajarMAQ, et =>)
      Coil( #MA_Bajar_MQ2 )
   END_RUNG
   RUNG wire#powerrail
      I_Contact( #EstadoVI.Etapas_Reset )
      I_Contact( #EstadoVI.Etapas_Carga_E1 )
      wire#w2
      Contact( #Selec_Salida_MQ2 )
      wire#w3
      Contact( #SaliendoCarga )
   END_RUNG wire#w1
   RUNG wire#w2
      Contact( #Selec_Salida_MQ1_2 )
   END_RUNG wire#w3
   RUNG wire#powerrail
      Contact( #EstadoVI.Etapas_Carga_E1 )
   END_RUNG wire#w1
   // the same network as SCL:
   #TMP_RetardoBajada_MQ2(IN := ((NOT #EstadoVI.Etapas_Reset AND NOT #EstadoVI.Etapas_Carga_E1 AND NOT #Selec_Salida_MQ2 AND NOT #Selec_Salida_MQ1 AND NOT #Selec_Salida_MQ1_2) OR (NOT #EstadoVI.Etapas_Reset AND NOT #EstadoVI.Etapas_Carga_E1 AND (#Selec_Salida_MQ2 OR #Selec_Salida_MQ1_2) AND #SaliendoCarga) OR #EstadoVI.Etapas_Carga_E1) AND NOT #MQ2_Abajo AND #EstadoZona.Marcha_CBx AND NOT #EstadoVI.Error_Mx AND NOT #Error_Tx,   // TON
                          PT := #V_RetardoBajarMAQ);
   #MA_Bajar_MQ2 := #TMP_RetardoBajada_MQ2.Q;
END_REGION

REGION Network 61: TMP - Espera En Tension
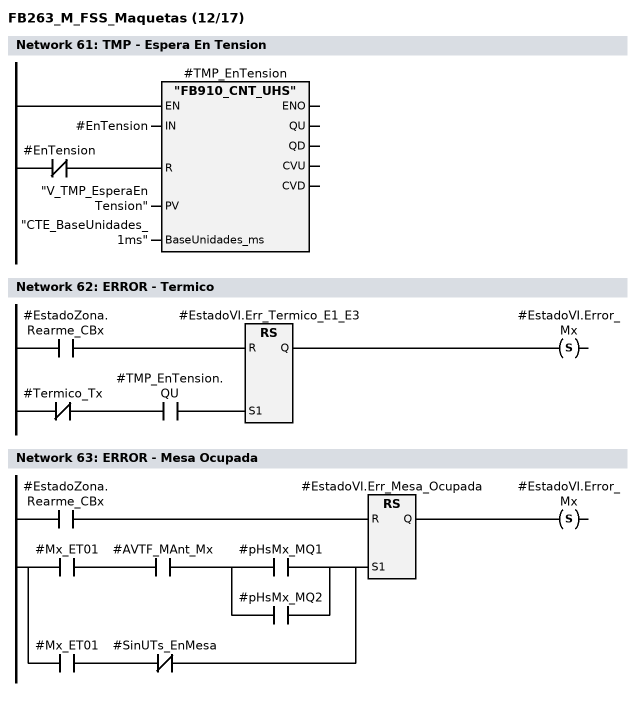
   RUNG wire#powerrail
      #TMP_EnTension(R := wire#w1, IN := #EnTension, PV := "V_TMP_EsperaEnTension", BaseUnidades_ms := "CTE_BaseUnidades_1ms", QU =>, QD =>, CVU =>, CVD =>)
   END_RUNG
   RUNG wire#powerrail
      I_Contact( #EnTension )
   END_RUNG wire#w1
   // the same network as SCL:
   #TMP_EnTension(IN := #EnTension,   // "FB910_CNT_UHS"
                  R := NOT #EnTension,
                  PV := "V_TMP_EsperaEnTension",
                  BaseUnidades_ms := "CTE_BaseUnidades_1ms");
END_REGION

REGION Network 62: ERROR - Termico
   RUNG wire#powerrail
      Contact( #EstadoZona.Rearme_CBx )
      S_RS(operand := #EstadoVI.Err_Termico_E1_E3, s1 := wire#w1)
      S_Coil( #EstadoVI.Error_Mx )
   END_RUNG
   RUNG wire#powerrail
      I_Contact( #Termico_Tx )
      Contact( #TMP_EnTension.QU )
   END_RUNG wire#w1
   // the same network as SCL:
   IF #EstadoZona.Rearme_CBx THEN
       #EstadoVI.Err_Termico_E1_E3 := FALSE;   // RS flip-flop
   END_IF;
   IF NOT #Termico_Tx AND #TMP_EnTension.QU THEN #EstadoVI.Err_Termico_E1_E3 := TRUE; END_IF;
   IF #EstadoVI.Err_Termico_E1_E3 THEN #EstadoVI.Error_Mx := TRUE; END_IF;
END_REGION

REGION Network 63: ERROR - Mesa Ocupada
   RUNG wire#powerrail
      Contact( #EstadoZona.Rearme_CBx )
      S_RS(operand := #EstadoVI.Err_Mesa_Ocupada, s1 := wire#w2)
      S_Coil( #EstadoVI.Error_Mx )
   END_RUNG
   RUNG wire#powerrail
      Contact( #Mx_ET01 )
      Contact( #AVTF_MAnt_Mx )
      wire#w1
      Contact( #pHsMx_MQ1 )
   END_RUNG wire#w2
   RUNG wire#w1
      Contact( #pHsMx_MQ2 )
   END_RUNG wire#w2
   RUNG wire#powerrail
      Contact( #Mx_ET01 )
      I_Contact( #SinUTs_EnMesa )
   END_RUNG wire#w2
   // the same network as SCL:
   IF #EstadoZona.Rearme_CBx THEN
       #EstadoVI.Err_Mesa_Ocupada := FALSE;   // RS flip-flop
   END_IF;
   IF (#Mx_ET01 AND #AVTF_MAnt_Mx AND (#pHsMx_MQ1 OR #pHsMx_MQ2)) OR (#Mx_ET01 AND NOT #SinUTs_EnMesa) THEN
       #EstadoVI.Err_Mesa_Ocupada := TRUE;
   END_IF;
   IF #EstadoVI.Err_Mesa_Ocupada THEN #EstadoVI.Error_Mx := TRUE; END_IF;
END_REGION

REGION Network 64: CNT - ERROR - Arrastre
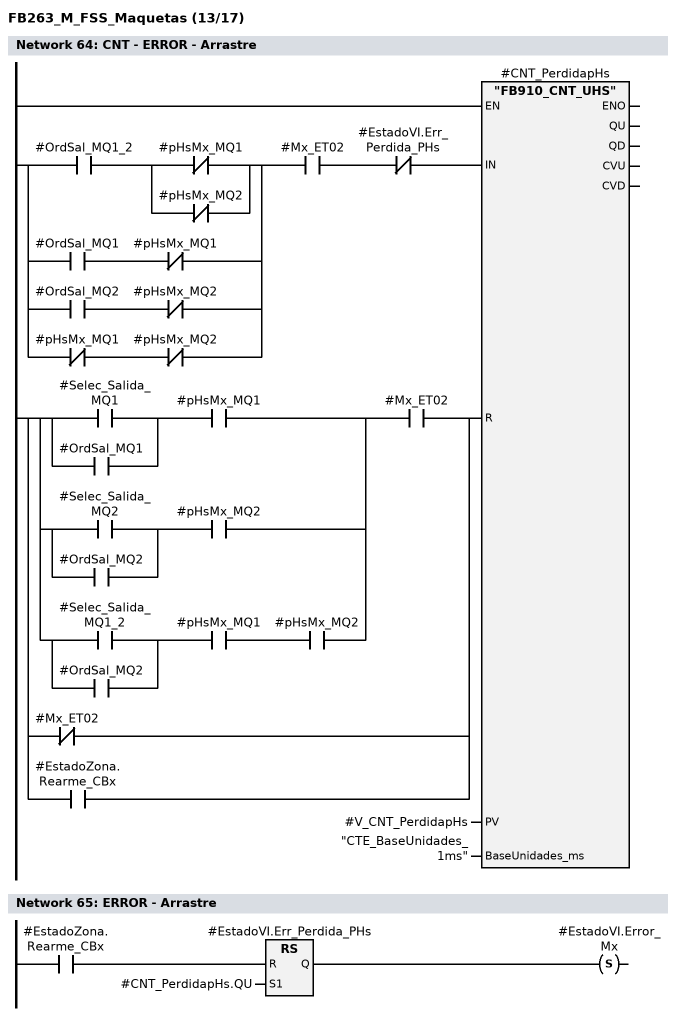
   RUNG wire#powerrail
      #CNT_PerdidapHs(IN := wire#w3, R := wire#w8, PV := #V_CNT_PerdidapHs, BaseUnidades_ms := "CTE_BaseUnidades_1ms", QU =>, QD =>, CVU =>, CVD =>)
   END_RUNG
   RUNG wire#powerrail
      Contact( #OrdSal_MQ1_2 )
      wire#w1
      I_Contact( #pHsMx_MQ1 )
      wire#w2
      Contact( #Mx_ET02 )
      I_Contact( #EstadoVI.Err_Perdida_PHs )
   END_RUNG wire#w3
   RUNG wire#w1
      I_Contact( #pHsMx_MQ2 )
   END_RUNG wire#w2
   RUNG wire#powerrail
      Contact( #OrdSal_MQ1 )
      I_Contact( #pHsMx_MQ1 )
   END_RUNG wire#w2
   RUNG wire#powerrail
      Contact( #OrdSal_MQ2 )
      I_Contact( #pHsMx_MQ2 )
   END_RUNG wire#w2
   RUNG wire#powerrail
      I_Contact( #pHsMx_MQ1 )
      I_Contact( #pHsMx_MQ2 )
   END_RUNG wire#w2
   RUNG wire#powerrail
      Contact( #Selec_Salida_MQ1 )
      wire#w4
      Contact( #pHsMx_MQ1 )
      wire#w5
      Contact( #Mx_ET02 )
   END_RUNG wire#w8
   RUNG wire#powerrail
      Contact( #OrdSal_MQ1 )
   END_RUNG wire#w4
   RUNG wire#powerrail
      Contact( #Selec_Salida_MQ2 )
      wire#w6
      Contact( #pHsMx_MQ2 )
   END_RUNG wire#w5
   RUNG wire#powerrail
      Contact( #OrdSal_MQ2 )
   END_RUNG wire#w6
   RUNG wire#powerrail
      Contact( #Selec_Salida_MQ1_2 )
      wire#w7
      Contact( #pHsMx_MQ1 )
      Contact( #pHsMx_MQ2 )
   END_RUNG wire#w5
   RUNG wire#powerrail
      Contact( #OrdSal_MQ2 )
   END_RUNG wire#w7
   RUNG wire#powerrail
      I_Contact( #Mx_ET02 )
   END_RUNG wire#w8
   RUNG wire#powerrail
      Contact( #EstadoZona.Rearme_CBx )
   END_RUNG wire#w8
   // the same network as SCL:
   #CNT_PerdidapHs(IN := ((#OrdSal_MQ1_2 AND (NOT #pHsMx_MQ1 OR NOT #pHsMx_MQ2)) OR (#OrdSal_MQ1 AND NOT #pHsMx_MQ1) OR (#OrdSal_MQ2 AND NOT #pHsMx_MQ2) OR (NOT #pHsMx_MQ1 AND NOT #pHsMx_MQ2)) AND #Mx_ET02 AND NOT #EstadoVI.Err_Perdida_PHs,   // "FB910_CNT_UHS"
                   R := ((((#Selec_Salida_MQ1 OR #OrdSal_MQ1) AND #pHsMx_MQ1) OR ((#Selec_Salida_MQ2 OR #OrdSal_MQ2) AND #pHsMx_MQ2) OR ((#Selec_Salida_MQ1_2 OR #OrdSal_MQ2) AND #pHsMx_MQ1 AND #pHsMx_MQ2)) AND #Mx_ET02) OR NOT #Mx_ET02 OR #EstadoZona.Rearme_CBx,
                   PV := #V_CNT_PerdidapHs,
                   BaseUnidades_ms := "CTE_BaseUnidades_1ms");
END_REGION

REGION Network 65: ERROR - Arrastre
   RUNG wire#powerrail
      Contact( #EstadoZona.Rearme_CBx )
      S_RS(operand := #EstadoVI.Err_Perdida_PHs, s1 := #CNT_PerdidapHs.QU)
      S_Coil( #EstadoVI.Error_Mx )
   END_RUNG
   // the same network as SCL:
   IF #EstadoZona.Rearme_CBx THEN
       #EstadoVI.Err_Perdida_PHs := FALSE;   // RS flip-flop
   END_IF;
   IF #CNT_PerdidapHs.QU THEN #EstadoVI.Err_Perdida_PHs := TRUE; END_IF;
   IF #EstadoVI.Err_Perdida_PHs THEN #EstadoVI.Error_Mx := TRUE; END_IF;
END_REGION

REGION Network 66: ERROR - Descarga por S3
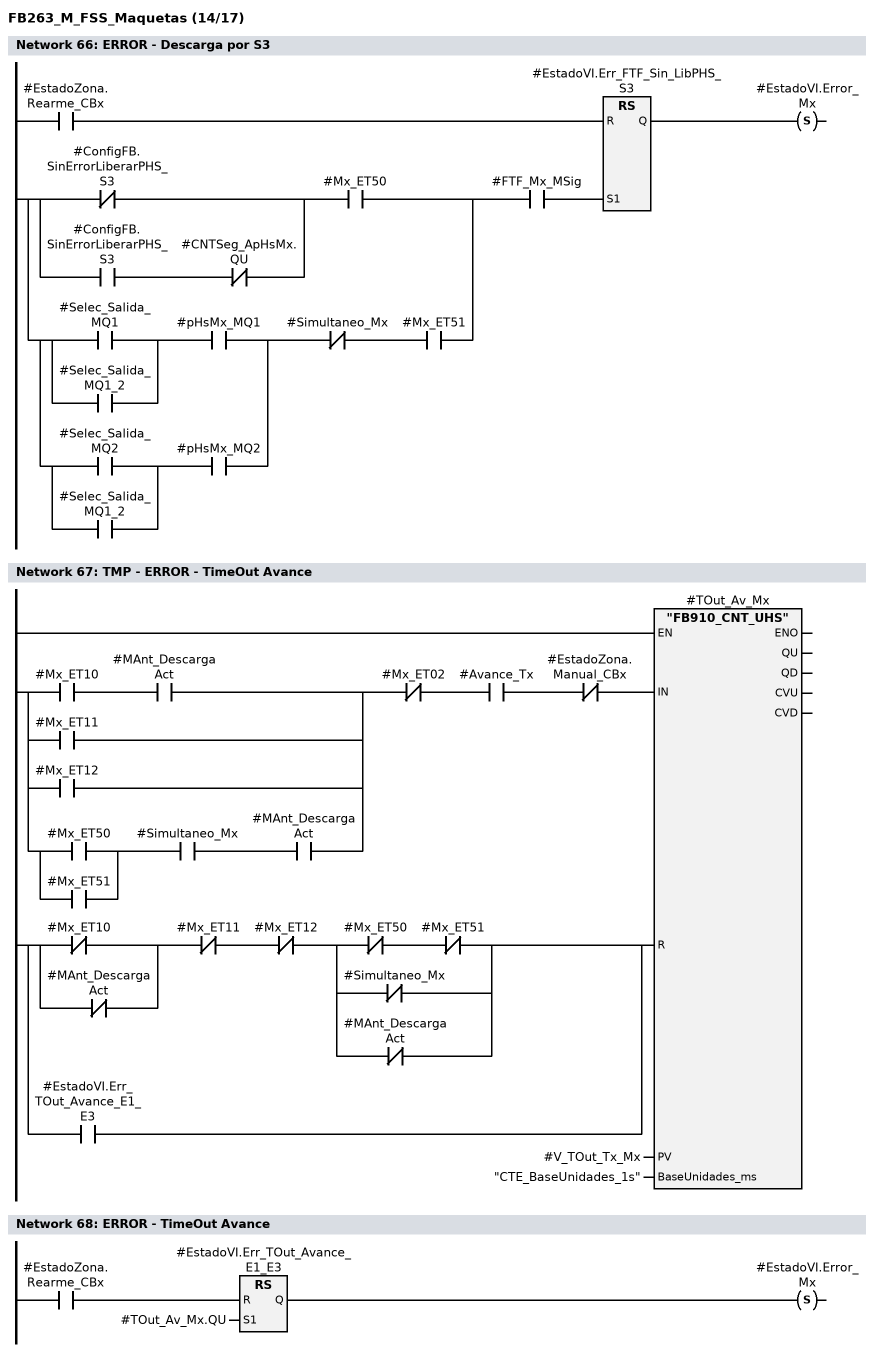
   RUNG wire#powerrail
      Contact( #EstadoZona.Rearme_CBx )
      S_RS(operand := #EstadoVI.Err_FTF_Sin_LibPHS_S3, s1 := wire#w6)
      S_Coil( #EstadoVI.Error_Mx )
   END_RUNG
   RUNG wire#powerrail
      I_Contact( #ConfigFB.SinErrorLiberarPHS_S3 )
      wire#w1
      Contact( #Mx_ET50 )
      wire#w2
      Contact( #FTF_Mx_MSig )
   END_RUNG wire#w6
   RUNG wire#powerrail
      Contact( #ConfigFB.SinErrorLiberarPHS_S3 )
      I_Contact( #CNTSeg_ApHsMx.QU )
   END_RUNG wire#w1
   RUNG wire#powerrail
      Contact( #Selec_Salida_MQ1 )
      wire#w3
      Contact( #pHsMx_MQ1 )
      wire#w4
      I_Contact( #Simultaneo_Mx )
      Contact( #Mx_ET51 )
   END_RUNG wire#w2
   RUNG wire#powerrail
      Contact( #Selec_Salida_MQ1_2 )
   END_RUNG wire#w3
   RUNG wire#powerrail
      Contact( #Selec_Salida_MQ2 )
      wire#w5
      Contact( #pHsMx_MQ2 )
   END_RUNG wire#w4
   RUNG wire#powerrail
      Contact( #Selec_Salida_MQ1_2 )
   END_RUNG wire#w5
   // the same network as SCL:
   IF #EstadoZona.Rearme_CBx THEN
       #EstadoVI.Err_FTF_Sin_LibPHS_S3 := FALSE;   // RS flip-flop
   END_IF;
   IF (((NOT #ConfigFB.SinErrorLiberarPHS_S3 OR (#ConfigFB.SinErrorLiberarPHS_S3 AND NOT #CNTSeg_ApHsMx.QU)) AND #Mx_ET50) OR ((((#Selec_Salida_MQ1 OR #Selec_Salida_MQ1_2) AND #pHsMx_MQ1) OR ((#Selec_Salida_MQ2 OR #Selec_Salida_MQ1_2) AND #pHsMx_MQ2)) AND NOT #Simultaneo_Mx AND #Mx_ET51)) AND #FTF_Mx_MSig THEN
       #EstadoVI.Err_FTF_Sin_LibPHS_S3 := TRUE;
   END_IF;
   IF #EstadoVI.Err_FTF_Sin_LibPHS_S3 THEN #EstadoVI.Error_Mx := TRUE; END_IF;
END_REGION

REGION Network 67: TMP - ERROR - TimeOut Avance
   RUNG wire#powerrail
      #TOut_Av_Mx(IN := wire#w3, R := wire#w6, PV := #V_TOut_Tx_Mx, BaseUnidades_ms := "CTE_BaseUnidades_1s", QU =>, QD =>, CVU =>, CVD =>)
   END_RUNG
   RUNG wire#powerrail
      Contact( #Mx_ET10 )
      Contact( #MAnt_DescargaAct )
      wire#w1
      I_Contact( #Mx_ET02 )
      Contact( #Avance_Tx )
      I_Contact( #EstadoZona.Manual_CBx )
   END_RUNG wire#w3
   RUNG wire#powerrail
      Contact( #Mx_ET11 )
   END_RUNG wire#w1
   RUNG wire#powerrail
      Contact( #Mx_ET12 )
   END_RUNG wire#w1
   RUNG wire#powerrail
      Contact( #Mx_ET50 )
      wire#w2
      Contact( #Simultaneo_Mx )
      Contact( #MAnt_DescargaAct )
   END_RUNG wire#w1
   RUNG wire#powerrail
      Contact( #Mx_ET51 )
   END_RUNG wire#w2
   RUNG wire#powerrail
      I_Contact( #Mx_ET10 )
      wire#w4
      I_Contact( #Mx_ET11 )
      I_Contact( #Mx_ET12 )
      wire#w5
      I_Contact( #Mx_ET50 )
      I_Contact( #Mx_ET51 )
   END_RUNG wire#w6
   RUNG wire#powerrail
      I_Contact( #MAnt_DescargaAct )
   END_RUNG wire#w4
   RUNG wire#w5
      I_Contact( #Simultaneo_Mx )
   END_RUNG wire#w6
   RUNG wire#w5
      I_Contact( #MAnt_DescargaAct )
   END_RUNG wire#w6
   RUNG wire#powerrail
      Contact( #EstadoVI.Err_TOut_Avance_E1_E3 )
   END_RUNG wire#w6
   // the same network as SCL:
   #TOut_Av_Mx(IN := ((#Mx_ET10 AND #MAnt_DescargaAct) OR #Mx_ET11 OR #Mx_ET12 OR ((#Mx_ET50 OR #Mx_ET51) AND #Simultaneo_Mx AND #MAnt_DescargaAct)) AND NOT #Mx_ET02 AND #Avance_Tx AND NOT #EstadoZona.Manual_CBx,   // "FB910_CNT_UHS"
               R := ((NOT #Mx_ET10 OR NOT #MAnt_DescargaAct) AND NOT #Mx_ET11 AND NOT #Mx_ET12 AND ((NOT #Mx_ET50 AND NOT #Mx_ET51) OR NOT #Simultaneo_Mx OR NOT #MAnt_DescargaAct)) OR #EstadoVI.Err_TOut_Avance_E1_E3,
               PV := #V_TOut_Tx_Mx,
               BaseUnidades_ms := "CTE_BaseUnidades_1s");
END_REGION

REGION Network 68: ERROR - TimeOut Avance
   RUNG wire#powerrail
      Contact( #EstadoZona.Rearme_CBx )
      S_RS(operand := #EstadoVI.Err_TOut_Avance_E1_E3, s1 := #TOut_Av_Mx.QU)
      S_Coil( #EstadoVI.Error_Mx )
   END_RUNG
   // the same network as SCL:
   IF #EstadoZona.Rearme_CBx THEN
       #EstadoVI.Err_TOut_Avance_E1_E3 := FALSE;   // RS flip-flop
   END_IF;
   IF #TOut_Av_Mx.QU THEN #EstadoVI.Err_TOut_Avance_E1_E3 := TRUE; END_IF;
   IF #EstadoVI.Err_TOut_Avance_E1_E3 THEN #EstadoVI.Error_Mx := TRUE; END_IF;
END_REGION

REGION Network 69: TMP - ERROR - TimeOut Subir TP
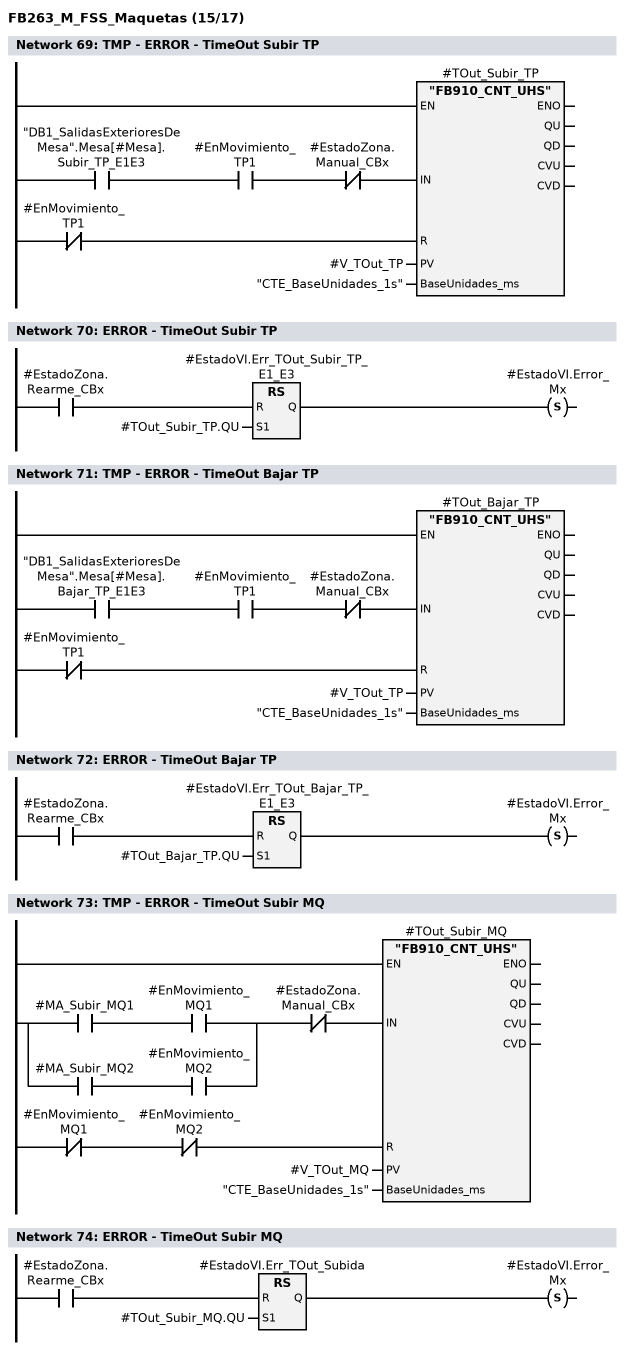
   RUNG wire#powerrail
      #TOut_Subir_TP(IN := wire#w1, R := wire#w2, PV := #V_TOut_TP, BaseUnidades_ms := "CTE_BaseUnidades_1s", QU =>, QD =>, CVU =>, CVD =>)
   END_RUNG
   RUNG wire#powerrail
      Contact( "DB1_SalidasExterioresDeMesa".Mesa[#Mesa].Subir_TP_E1E3 )
      Contact( #EnMovimiento_TP1 )
      I_Contact( #EstadoZona.Manual_CBx )
   END_RUNG wire#w1
   RUNG wire#powerrail
      I_Contact( #EnMovimiento_TP1 )
   END_RUNG wire#w2
   // the same network as SCL:
   #TOut_Subir_TP(IN := "DB1_SalidasExterioresDeMesa".Mesa[#Mesa].Subir_TP_E1E3 AND #EnMovimiento_TP1 AND NOT #EstadoZona.Manual_CBx,   // "FB910_CNT_UHS"
                  R := NOT #EnMovimiento_TP1,
                  PV := #V_TOut_TP,
                  BaseUnidades_ms := "CTE_BaseUnidades_1s");
END_REGION

REGION Network 70: ERROR - TimeOut Subir TP
   RUNG wire#powerrail
      Contact( #EstadoZona.Rearme_CBx )
      S_RS(operand := #EstadoVI.Err_TOut_Subir_TP_E1_E3, s1 := #TOut_Subir_TP.QU)
      S_Coil( #EstadoVI.Error_Mx )
   END_RUNG
   // the same network as SCL:
   IF #EstadoZona.Rearme_CBx THEN
       #EstadoVI.Err_TOut_Subir_TP_E1_E3 := FALSE;   // RS flip-flop
   END_IF;
   IF #TOut_Subir_TP.QU THEN #EstadoVI.Err_TOut_Subir_TP_E1_E3 := TRUE; END_IF;
   IF #EstadoVI.Err_TOut_Subir_TP_E1_E3 THEN #EstadoVI.Error_Mx := TRUE; END_IF;
END_REGION

REGION Network 71: TMP - ERROR - TimeOut Bajar TP
   RUNG wire#powerrail
      #TOut_Bajar_TP(IN := wire#w1, R := wire#w2, PV := #V_TOut_TP, BaseUnidades_ms := "CTE_BaseUnidades_1s", QU =>, QD =>, CVU =>, CVD =>)
   END_RUNG
   RUNG wire#powerrail
      Contact( "DB1_SalidasExterioresDeMesa".Mesa[#Mesa].Bajar_TP_E1E3 )
      Contact( #EnMovimiento_TP1 )
      I_Contact( #EstadoZona.Manual_CBx )
   END_RUNG wire#w1
   RUNG wire#powerrail
      I_Contact( #EnMovimiento_TP1 )
   END_RUNG wire#w2
   // the same network as SCL:
   #TOut_Bajar_TP(IN := "DB1_SalidasExterioresDeMesa".Mesa[#Mesa].Bajar_TP_E1E3 AND #EnMovimiento_TP1 AND NOT #EstadoZona.Manual_CBx,   // "FB910_CNT_UHS"
                  R := NOT #EnMovimiento_TP1,
                  PV := #V_TOut_TP,
                  BaseUnidades_ms := "CTE_BaseUnidades_1s");
END_REGION

REGION Network 72: ERROR - TimeOut Bajar TP
   RUNG wire#powerrail
      Contact( #EstadoZona.Rearme_CBx )
      S_RS(operand := #EstadoVI.Err_TOut_Bajar_TP_E1_E3, s1 := #TOut_Bajar_TP.QU)
      S_Coil( #EstadoVI.Error_Mx )
   END_RUNG
   // the same network as SCL:
   IF #EstadoZona.Rearme_CBx THEN
       #EstadoVI.Err_TOut_Bajar_TP_E1_E3 := FALSE;   // RS flip-flop
   END_IF;
   IF #TOut_Bajar_TP.QU THEN #EstadoVI.Err_TOut_Bajar_TP_E1_E3 := TRUE; END_IF;
   IF #EstadoVI.Err_TOut_Bajar_TP_E1_E3 THEN #EstadoVI.Error_Mx := TRUE; END_IF;
END_REGION

REGION Network 73: TMP - ERROR - TimeOut Subir MQ
   RUNG wire#powerrail
      #TOut_Subir_MQ(IN := wire#w2, R := wire#w3, PV := #V_TOut_MQ, BaseUnidades_ms := "CTE_BaseUnidades_1s", QU =>, QD =>, CVU =>, CVD =>)
   END_RUNG
   RUNG wire#powerrail
      Contact( #MA_Subir_MQ1 )
      Contact( #EnMovimiento_MQ1 )
      wire#w1
      I_Contact( #EstadoZona.Manual_CBx )
   END_RUNG wire#w2
   RUNG wire#powerrail
      Contact( #MA_Subir_MQ2 )
      Contact( #EnMovimiento_MQ2 )
   END_RUNG wire#w1
   RUNG wire#powerrail
      I_Contact( #EnMovimiento_MQ1 )
      I_Contact( #EnMovimiento_MQ2 )
   END_RUNG wire#w3
   // the same network as SCL:
   #TOut_Subir_MQ(IN := ((#MA_Subir_MQ1 AND #EnMovimiento_MQ1) OR (#MA_Subir_MQ2 AND #EnMovimiento_MQ2)) AND NOT #EstadoZona.Manual_CBx,   // "FB910_CNT_UHS"
                  R := NOT #EnMovimiento_MQ1 AND NOT #EnMovimiento_MQ2,
                  PV := #V_TOut_MQ,
                  BaseUnidades_ms := "CTE_BaseUnidades_1s");
END_REGION

REGION Network 74: ERROR - TimeOut Subir MQ
   RUNG wire#powerrail
      Contact( #EstadoZona.Rearme_CBx )
      S_RS(operand := #EstadoVI.Err_TOut_Subida, s1 := #TOut_Subir_MQ.QU)
      S_Coil( #EstadoVI.Error_Mx )
   END_RUNG
   // the same network as SCL:
   IF #EstadoZona.Rearme_CBx THEN
       #EstadoVI.Err_TOut_Subida := FALSE;   // RS flip-flop
   END_IF;
   IF #TOut_Subir_MQ.QU THEN #EstadoVI.Err_TOut_Subida := TRUE; END_IF;
   IF #EstadoVI.Err_TOut_Subida THEN #EstadoVI.Error_Mx := TRUE; END_IF;
END_REGION

REGION Network 75: TMP - ERROR - TimeOut Bajar MQ
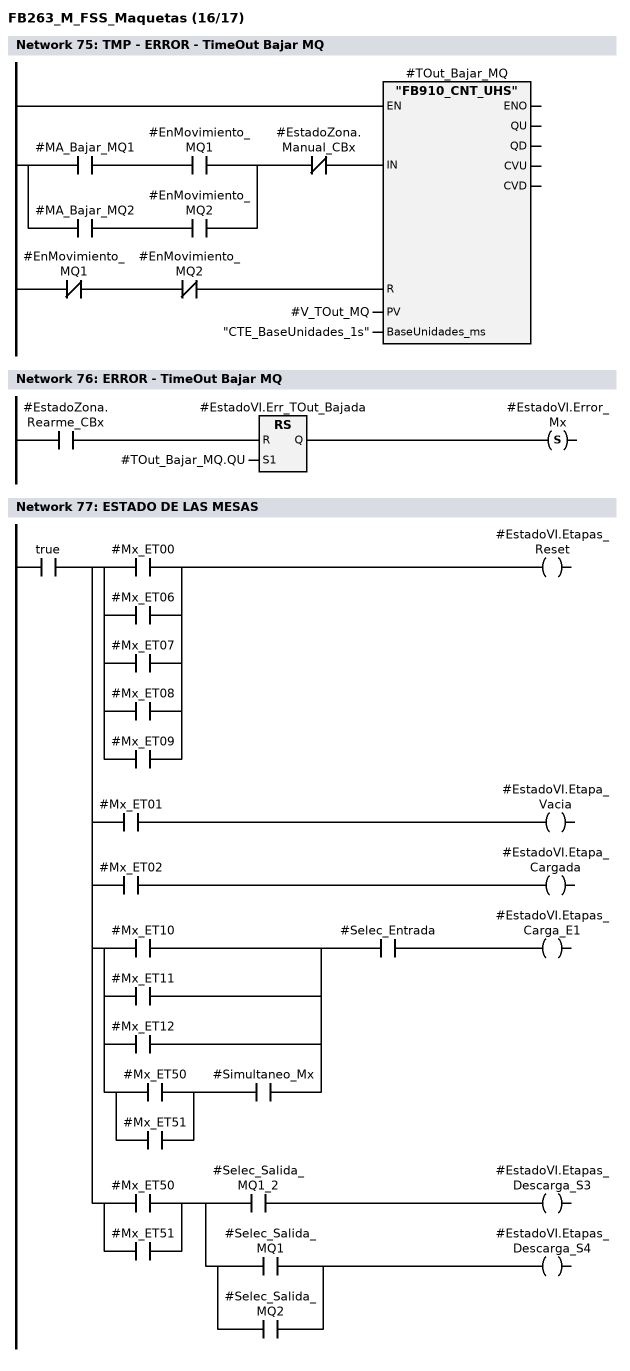
   RUNG wire#powerrail
      #TOut_Bajar_MQ(IN := wire#w2, R := wire#w3, PV := #V_TOut_MQ, BaseUnidades_ms := "CTE_BaseUnidades_1s", QU =>, QD =>, CVU =>, CVD =>)
   END_RUNG
   RUNG wire#powerrail
      Contact( #MA_Bajar_MQ1 )
      Contact( #EnMovimiento_MQ1 )
      wire#w1
      I_Contact( #EstadoZona.Manual_CBx )
   END_RUNG wire#w2
   RUNG wire#powerrail
      Contact( #MA_Bajar_MQ2 )
      Contact( #EnMovimiento_MQ2 )
   END_RUNG wire#w1
   RUNG wire#powerrail
      I_Contact( #EnMovimiento_MQ1 )
      I_Contact( #EnMovimiento_MQ2 )
   END_RUNG wire#w3
   // the same network as SCL:
   #TOut_Bajar_MQ(IN := ((#MA_Bajar_MQ1 AND #EnMovimiento_MQ1) OR (#MA_Bajar_MQ2 AND #EnMovimiento_MQ2)) AND NOT #EstadoZona.Manual_CBx,   // "FB910_CNT_UHS"
                  R := NOT #EnMovimiento_MQ1 AND NOT #EnMovimiento_MQ2,
                  PV := #V_TOut_MQ,
                  BaseUnidades_ms := "CTE_BaseUnidades_1s");
END_REGION

REGION Network 76: ERROR - TimeOut Bajar MQ
   RUNG wire#powerrail
      Contact( #EstadoZona.Rearme_CBx )
      S_RS(operand := #EstadoVI.Err_TOut_Bajada, s1 := #TOut_Bajar_MQ.QU)
      S_Coil( #EstadoVI.Error_Mx )
   END_RUNG
   // the same network as SCL:
   IF #EstadoZona.Rearme_CBx THEN
       #EstadoVI.Err_TOut_Bajada := FALSE;   // RS flip-flop
   END_IF;
   IF #TOut_Bajar_MQ.QU THEN #EstadoVI.Err_TOut_Bajada := TRUE; END_IF;
   IF #EstadoVI.Err_TOut_Bajada THEN #EstadoVI.Error_Mx := TRUE; END_IF;
END_REGION

REGION Network 77: ESTADO DE LAS MESAS
   RUNG wire#powerrail
      Contact( true )
      wire#w1
      Contact( #Mx_ET00 )
      wire#w2
      Coil( #EstadoVI.Etapas_Reset )
   END_RUNG
   RUNG wire#w1
      Contact( #Mx_ET06 )
   END_RUNG wire#w2
   RUNG wire#w1
      Contact( #Mx_ET07 )
   END_RUNG wire#w2
   RUNG wire#w1
      Contact( #Mx_ET08 )
   END_RUNG wire#w2
   RUNG wire#w1
      Contact( #Mx_ET09 )
   END_RUNG wire#w2
   RUNG wire#w1
      Contact( #Mx_ET01 )
      Coil( #EstadoVI.Etapa_Vacia )
   END_RUNG
   RUNG wire#w1
      Contact( #Mx_ET02 )
      Coil( #EstadoVI.Etapa_Cargada )
   END_RUNG
   RUNG wire#w1
      Contact( #Mx_ET10 )
      wire#w3
      Contact( #Selec_Entrada )
      Coil( #EstadoVI.Etapas_Carga_E1 )
   END_RUNG
   RUNG wire#w1
      Contact( #Mx_ET11 )
   END_RUNG wire#w3
   RUNG wire#w1
      Contact( #Mx_ET12 )
   END_RUNG wire#w3
   RUNG wire#w1
      Contact( #Mx_ET50 )
      wire#w4
      Contact( #Simultaneo_Mx )
   END_RUNG wire#w3
   RUNG wire#w1
      Contact( #Mx_ET51 )
   END_RUNG wire#w4
   RUNG wire#w1
      Contact( #Mx_ET50 )
      wire#w5
      Contact( #Selec_Salida_MQ1_2 )
      Coil( #EstadoVI.Etapas_Descarga_S3 )
   END_RUNG
   RUNG wire#w1
      Contact( #Mx_ET51 )
   END_RUNG wire#w5
   RUNG wire#w5
      Contact( #Selec_Salida_MQ1 )
      wire#w6
      Coil( #EstadoVI.Etapas_Descarga_S4 )
   END_RUNG
   RUNG wire#w5
      Contact( #Selec_Salida_MQ2 )
   END_RUNG wire#w6
   // the same network as SCL:
   #EstadoVI.Etapas_Reset := true AND (#Mx_ET00 OR #Mx_ET06 OR #Mx_ET07 OR #Mx_ET08 OR #Mx_ET09);
   #EstadoVI.Etapa_Vacia := true AND #Mx_ET01;
   #EstadoVI.Etapa_Cargada := true AND #Mx_ET02;
   #EstadoVI.Etapas_Carga_E1 := true AND (#Mx_ET10 OR #Mx_ET11 OR #Mx_ET12 OR ((#Mx_ET50 OR #Mx_ET51) AND #Simultaneo_Mx)) AND #Selec_Entrada;
   #_w1 := true AND (#Mx_ET50 OR #Mx_ET51);
   #EstadoVI.Etapas_Descarga_S3 := #_w1 AND #Selec_Salida_MQ1_2;
   #EstadoVI.Etapas_Descarga_S4 := #_w1 AND (#Selec_Salida_MQ1 OR #Selec_Salida_MQ2);
END_REGION

REGION Network 78: ENTRADAS DE LA MESA
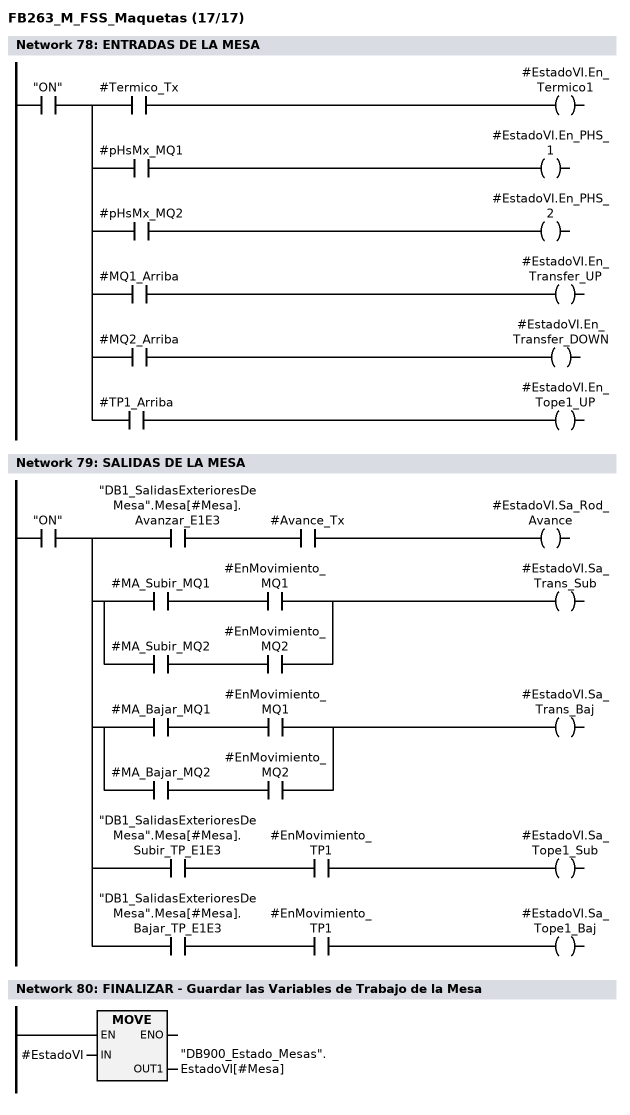
   RUNG wire#powerrail
      Contact( "ON" )
      wire#w1
      Contact( #Termico_Tx )
      Coil( #EstadoVI.En_Termico1 )
   END_RUNG
   RUNG wire#w1
      Contact( #pHsMx_MQ1 )
      Coil( #EstadoVI.En_PHS_1 )
   END_RUNG
   RUNG wire#w1
      Contact( #pHsMx_MQ2 )
      Coil( #EstadoVI.En_PHS_2 )
   END_RUNG
   RUNG wire#w1
      Contact( #MQ1_Arriba )
      Coil( #EstadoVI.En_Transfer_UP )
   END_RUNG
   RUNG wire#w1
      Contact( #MQ2_Arriba )
      Coil( #EstadoVI.En_Transfer_DOWN )
   END_RUNG
   RUNG wire#w1
      Contact( #TP1_Arriba )
      Coil( #EstadoVI.En_Tope1_UP )
   END_RUNG
   // the same network as SCL:
   #EstadoVI.En_Termico1 := "ON" AND #Termico_Tx;
   #EstadoVI.En_PHS_1 := "ON" AND #pHsMx_MQ1;
   #EstadoVI.En_PHS_2 := "ON" AND #pHsMx_MQ2;
   #EstadoVI.En_Transfer_UP := "ON" AND #MQ1_Arriba;
   #EstadoVI.En_Transfer_DOWN := "ON" AND #MQ2_Arriba;
   #EstadoVI.En_Tope1_UP := "ON" AND #TP1_Arriba;
END_REGION

REGION Network 79: SALIDAS DE LA MESA
   RUNG wire#powerrail
      Contact( "ON" )
      wire#w1
      Contact( "DB1_SalidasExterioresDeMesa".Mesa[#Mesa].Avanzar_E1E3 )
      Contact( #Avance_Tx )
      Coil( #EstadoVI.Sa_Rod_Avance )
   END_RUNG
   RUNG wire#w1
      Contact( #MA_Subir_MQ1 )
      Contact( #EnMovimiento_MQ1 )
      wire#w2
      Coil( #EstadoVI.Sa_Trans_Sub )
   END_RUNG
   RUNG wire#w1
      Contact( #MA_Subir_MQ2 )
      Contact( #EnMovimiento_MQ2 )
   END_RUNG wire#w2
   RUNG wire#w1
      Contact( #MA_Bajar_MQ1 )
      Contact( #EnMovimiento_MQ1 )
      wire#w3
      Coil( #EstadoVI.Sa_Trans_Baj )
   END_RUNG
   RUNG wire#w1
      Contact( #MA_Bajar_MQ2 )
      Contact( #EnMovimiento_MQ2 )
   END_RUNG wire#w3
   RUNG wire#w1
      Contact( "DB1_SalidasExterioresDeMesa".Mesa[#Mesa].Subir_TP_E1E3 )
      Contact( #EnMovimiento_TP1 )
      Coil( #EstadoVI.Sa_Tope1_Sub )
   END_RUNG
   RUNG wire#w1
      Contact( "DB1_SalidasExterioresDeMesa".Mesa[#Mesa].Bajar_TP_E1E3 )
      Contact( #EnMovimiento_TP1 )
      Coil( #EstadoVI.Sa_Tope1_Baj )
   END_RUNG
   // the same network as SCL:
   #EstadoVI.Sa_Rod_Avance := "ON" AND "DB1_SalidasExterioresDeMesa".Mesa[#Mesa].Avanzar_E1E3 AND #Avance_Tx;
   #EstadoVI.Sa_Trans_Sub := "ON" AND ((#MA_Subir_MQ1 AND #EnMovimiento_MQ1) OR (#MA_Subir_MQ2 AND #EnMovimiento_MQ2));
   #EstadoVI.Sa_Trans_Baj := "ON" AND ((#MA_Bajar_MQ1 AND #EnMovimiento_MQ1) OR (#MA_Bajar_MQ2 AND #EnMovimiento_MQ2));
   #EstadoVI.Sa_Tope1_Sub := "ON" AND "DB1_SalidasExterioresDeMesa".Mesa[#Mesa].Subir_TP_E1E3 AND #EnMovimiento_TP1;
   #EstadoVI.Sa_Tope1_Baj := "ON" AND "DB1_SalidasExterioresDeMesa".Mesa[#Mesa].Bajar_TP_E1E3 AND #EnMovimiento_TP1;
END_REGION

REGION Network 80: FINALIZAR - Guardar las Variables de Trabajo de la Mesa
   RUNG wire#powerrail
      Move(in := #EstadoVI, out1 => "DB900_Estado_Mesas".EstadoVI[#Mesa])
   END_RUNG
   // the same network as SCL:
   "DB900_Estado_Mesas".EstadoVI[#Mesa] := #EstadoVI;
END_REGION
END_FUNCTION_BLOCK

FUNCTION "FC870_MesaSinUT" : Void   // FC870, LAD
TITLE = "MesaSinUT"
{ S7_Optimized_Access := 'FALSE' }
AUTHOR : TRACKING
NAME : 20130301
VERSION : 3.0
// Devuelve si hay UT o no en la Mesa (bool)
// stored: AutoNumber false, SetENOAutomatically false
   VAR_INPUT
      Mesa : UInt;   // Mesa que se quiere ver si no hay UT's
   END_VAR
   VAR_OUTPUT
      SinUT : Bool;   // La Mesa no tiene UT
   END_VAR
   VAR_TEMP
      Relleno : Byte;
      ValorReturn : Int;
   END_VAR
BEGIN

NETWORK
TITLE = Inicializar
////////////////////////////////////////////////////////////////////////////
// --- Reseteo Variable de Salida

      SET;
      =     #SinUT;  // Activo: No hay UT's



NETWORK
TITLE = Comprobar si hay UT en la Mesa
////////////////////////////////////////////////////////////////////////////
// --- Leer Cola de la Mesa


////////////////////////////////////////////////////////////////////////////
// --- Comprobacion de que la Mesa tenga UT o No

      L     "DB810_ColasMesas".Colas[#Mesa].UT_PrimeraMesa;
      L     0;
      ==I;
      JC    Final;  // No hay UT's ?

      CLR;
      =     #SinUT;  // Desactivo: Hay UT's

Final:NOP   0;  // Finalizar Funcion


END_FUNCTION

FUNCTION_BLOCK "FB270_M_FSS_Carga_V5"   // FB270, LAD
TITLE = FSS_Carga
{ S7_Optimized_Access := 'FALSE' }
AUTHOR : TE_FSS
FAMILY : FSS
NAME : 20160509
VERSION : 3.2
// stored: AutoNumber false, SetENOAutomatically false
   VAR_INPUT
      Mesa : UInt;   // Mesa de la FB
      Mx_TRxConAusencia : Bool;   // Config >> TRx Con Ausencia para entrada de la siguiente carga
      Error_Tx : Bool;   // Error en el Tx
      EnTension : Bool;   // Existe Tension en la Mesa
      Termico_T1 : Bool;   // Proteccion del T1
      Termico_T2 : Bool;   // Proteccion del T2
      Termico_T3 : Bool;   // Proteccion del T3
      Termico_T4 : Bool;   // Proteccion del T4
      pHsMx_1 : Bool;   // pHs 1 de la Mesa
      pHsMx_2 : Bool;   // pHs 2 de la Mesa
      pHsMx_3 : Bool;   // pHs 3 de la Mesa
      pHsMx_4 : Bool;   // pHs 4 de la Mesa
      Avance_T1 : Bool;   // Avance del T1
      Avance_T2 : Bool;   // Avance del T2
      Avance_T3 : Bool;   // Avance del T3
      Avance_T4 : Bool;   // Avance del T4
      Termico_TR1 : Bool;   // Proteccion del TR1
      Termico_TR2 : Bool;   // Proteccion del TR1
      Avance_TR1 : Bool;   // Avance del TR1
      Avance_TR2 : Bool;   // Avance del TR2
      TR1_Arriba : Bool;   // TR1 >> Arriba
      TR1_Abajo : Bool;   // TR1 >> Abajo
      TR1_EnMovimiento : Bool;   // TR1 >> En Movimiento
      TR2_Arriba : Bool;   // TR2 >> Arriba
      TR2_Abajo : Bool;   // TR2 >> Abajo
      TR2_EnMovimiento : Bool;   // TR2 >> En Movimiento
      TP1_Arriba : Bool;   // TP1 >> Arriba
      TP1_Abajo : Bool;   // TP1 >> Abajo
      TP1_EnMovimiento : Bool;   // TP1 >> En Movimiento
      TP2_Arriba : Bool;   // TP2 >> Arriba
      TP2_Abajo : Bool;   // TP2 >> Abajo
      TP2_EnMovimiento : Bool;   // TP2 >> En Movimiento
      TPS1_Arriba : Bool;   // TPS1 >> Arriba
      TPS1_Abajo : Bool;   // TPS1 >> Abajo
      TPS1_EnMovimiento : Bool;   // TPS1 >> En Movimiento
      TPS3_Arriba : Bool;   // TPS2 >> Arriba
      TPS3_Abajo : Bool;   // TPS2 >> Abajo
      TPS3_EnMovimiento : Bool;   // TPS2 >> En Movimiento
      MAnt_DescargaAct : Bool;   // E2 >> Mesa Anterior DescargaAct
      AVTF_MAnt_Mx_BGrande : Bool;   // E2 >> Mesa Anterior AVTF - Grande
      AVTF_MAnt_Mx_BPequena : Bool;   // E2 >> Mesa Anterior AVTF - Pequeña
      P_Mens_MAnt_Mx : Bool;   // E2 >> Mesa Anterior P_Mens
      S1_Arrival : Bool;   // S1 a FSS >> Arrival
      S1_Rotative : Bool;   // S1 a FSS >> Rotative
      S1_Complete : Bool;   // S1 a FSS >> Complete
      S3_Arrival : Bool;   // S3 a FSS >> Arrival
      S3_Rotative : Bool;   // S3 a FSS >> Rotative
      S3_Complete : Bool;   // S3 a FSS >> Complete
      MAnt_MSig_DesCargaAct : Bool;   // Pasarela >> Descarga Act
      AVTF_MAnt_MSig_BGrande : Bool;   // Pasarela >> AVTF - Grande
      AVTF_MAnt_MSig_BPequena : Bool;   // Pasarela >> AVTF - Pequeña
      PTF_MAnt_MSig : Bool;   // Pasarela >> PTF
      FTF_MAnt_MSig : Bool;   // Pasarela >> FTF
      F_EnvMens_Mx : Bool;   // Fin de Envio de Mensaje
      OrdSal_S01 : Bool;   // Orden de Salida por S1
      OrdSal_S03 : Bool;   // Orden de Salida por S3
      V_CNT_pHsMx : Int := 1000;   // Valor de Presencia
      V_CNT_pHsMx_FTF : Int := 250;   // Valor para activar FTF. Nota: < = V_CNT_pHsMx.
      V_CNTSeg_pHsMx : Int := 2000;   // Valor de Seguriadad para Presencia
      V_CNT_ApHsMx : Int := 200;   // Valor de Ausencia
      V_CNTSeg_ApHsMx : Int := 2000;   // Valor de Seguriadad para Ausencia
      V_TOut_Tx_Mx : Int := 7000;   // TimeOut de Entrada por E2
      V_TOut_TR : Int := 3000;   // TimeOut de Transfer
      V_TOut_TP : Int := 3000;   // TimeOut de Tope
      V_TOut_Interlock : Int := 5000;   // TimeOut de Interlock con el FSS
      V_CNT_PerdidapHs : Int := 1000;   // CNT de Perdida de pHs
      V_CNT_PosicionarCarga : Int := 500;   // Valor de Posicionar la Carga despues de la Entrada
      V_CNT_PresenciaPasarela : Int := 500;   // Valor de Posiconado para Pasarela
      V_CNT_HuecoTR1 : Int := 150;   // Valor de Hueco - Libre TR1
      V_CNT_HuecoTR2 : Int := 150;   // Valor de Hueco - Libre TR2
      V_TIM_EstabilidadCarga : Time := T#100MS;   // Valor de Eastabilidad de Carga por DCC
   END_VAR
   VAR_OUTPUT
      P_EnvMens_PMx : Bool;   // Permiso de Enviar Mensaje de Presencia
      P_EnvMens_AMx : Bool;   // Permiso de Enviar Mensaje de Ausencia
      P_RecepOK_Mx : Bool;   // Recepcion OK
      PTF_MAnt_Mx : Bool;   // E2 >> Mesa Anterior PTF
      FTF_MAnt_Mx : Bool;   // E2 >> Mesa Anterior FTF
      PMAnt_MSig_DescagaAct : Bool;   // Pasarela >> Descarga Act
      PAVTF_MAnt_MSig_BPequena : Bool;   // Pasarela >> AVTF - Grande
      PAVTF_MAnt_MSig_BGrande : Bool;   // Pasarela >> AVTF - Pequeña
      PPTF_MAnt_MSig : Bool;   // Pasarela >> PTF
      PFTF_MAnt_MSig : Bool;   // Pasarela >> FTF
   END_VAR
   VAR
      Mx_ET00 : Bool;
      Mx_ET01 : Bool;
      Mx_ET02 : Bool;
      Mx_ET07_1PRE : Bool;
      Mx_ET07_1FIN : Bool;
      Mx_ET07_2PRE : Bool;
      Mx_ET07_2FIN : Bool;
      Mx_ET07_3PRE : Bool;
      Mx_ET07_3FIN : Bool;
      Mx_ET07_4PRE : Bool;
      Mx_ET07_4FIN : Bool;
      Mx_ET08 : Bool;
      Mx_ET09 : Bool;
      Mx_ET10 : Bool;
      Mx_ET11 : Bool;
      Mx_ET12 : Bool;
      Mx_ET110 : Bool;
      Mx_ET111 : Bool;
      Mx_ET13 : Bool;
      Mx_ET14 : Bool;
      Mx_ET15 : Bool;
      Mx_ET16 : Bool;
      Mx_ET17 : Bool;
      Mx_ET40 : Bool;
      Mx_ET41 : Bool;
      Mx_ET42 : Bool;
      Mx_ET50 : Bool;
      Mx_ET51 : Bool;
      Mx_ET150 : Bool;
      Mx_ET151 : Bool;
      Mx_ET152 : Bool;
      Mx_ET250 : Bool;
      Mx_ET251 : Bool;
      Mx_ET60 : Bool;
      Mx_ET61 : Bool;
      Mx_ET160 : Bool;
      Mx_ET161 : Bool;
      Mx_ET162 : Bool;
      Mx_ET260 : Bool;
      Mx_ET261 : Bool;
      Mx_ET90 : Bool;
      Mx_ET91 : Bool;
      Mx_ET92 : Bool;
      TRAus_SinpHsSig : Bool;
      Mx_AutoArranque : Bool;   // Config >> Fin carga del FSS - Automatico
      FinCargaFSS_Auto : Bool;   // Intena >> AutoRearme Fin Carga del FSS
      Entrando_BGrande : Bool;   // Interna >> Bandeja Grande en Entrada
      Activado_Pasarela : Bool;   // Pasarela >> Activada
      Permiso_Pasarela : Bool;   // Pasarela >> Permiso de Movimiento
      S1_DesCargaAct : Bool;   // Interna >> DesCarga Activa de Salida por S1
      S3_DesCargaAct : Bool;   // Interna >> DesCarga Activa de Salida por S3
      Pos_TROK : Bool;   // Interna >> Posicion Correcta de los TRs
      Pos_TPOK : Bool;   // Interna >> Posicion Correcta de los TPs
      Select_S1 : Bool;   // Interna >> Selecionado Salida por S1
      Select_S3 : Bool;   // Interna >> Selecionado Salida por S3
      MemoriaPos_01 : Bool;   // Interna >> Memoria de Posicion Ocupada pHs_1
      MemoriaPos_02 : Bool;   // Interna >> Memoria de Posicion Ocupada pHs_2
      MemoriaPos_03 : Bool;   // Interna >> Memoria de Posicion Ocupada pHs_3
      MemoriaPos_04 : Bool;   // Interna >> Memoria de Posicion Ocupada pHs_4
      ProtocoloInciado : Bool;   // Iniciado el Envio del Mensaje de Presencia
      STAT_EnvMens_PMx : Bool;   // Interna >> Envio del Mensaje de Presencia
      STAT_EnvMens_AMx : Bool;   // Interna >> Envio de Mensaje de Ausencia
      STAT_AVTF_MAnt_Mx : Bool;   // Interna >> Aviso de Entrada
      STAT_FTF_MAnt_Mx : Bool;   // Interna >> FTF de MAnt >> Mx
      STAT_AvanceCarga : Bool;   // Interna >> Avance de Entrada de Carga
      STAT_AvanceDescarga : Bool;   // Interna >> Avance de Salida de Carga
      STAT_AvancePasarela : Bool;   // Interna >> Avance de Pasarela
      STAT_Velocidad_TxBO : Bool;   // Interna >> Velocidad Bit 0 de los Rodillos
      STAT_Velocidad_TxB1 : Bool;   // Interna >> Velocidad Bit 1 de los Rodillos
      MA_Avance_T1 : Bool;
      MA_Avance_T2 : Bool;
      MA_Avance_T3 : Bool;
      MA_Avance_T4 : Bool;
      MA_Inversion_Tx : Bool;
      MA_VelocidadAnalogica : Int;
      MA_Avance_TR1 : Bool;
      MA_Avance_TR2 : Bool;
      MA_VelocidaLenta_TRx : Bool;
      MA_Subir_TR1 : Bool;
      MA_Bajar_TR1 : Bool;
      MA_Subir_TR2 : Bool;
      MA_Bajar_TR2 : Bool;
      MA_Subir_TP1 : Bool;
      MA_Bajar_TP1 : Bool;
      MA_Subir_TP2 : Bool;
      MA_Bajar_TP2 : Bool;
      MA_Subir_TPS1 : Bool;
      MA_Bajar_TPS1 : Bool;
      MA_Subir_TPS3 : Bool;
      MA_Bajar_TPS3 : Bool;
      MA_PickUpOK_S1 : Bool;
      MA_PickUpOK_S3 : Bool;
      CNT_pHsMx_FTF_OK : Bool;   // Enviar ya FTF
      TIM_Estabilidad_Entrada { S7_SetPoint := 'True'} : TON_TIME;   // TIM De Estabilidad de Carga en la Entrada
      TIM_Estabilidad_S1 { S7_SetPoint := 'True'} : TON_TIME;   // TIM De Estabilidad de Carga en la Salida por S1
      TIM_Estabilidad_S3 { S7_SetPoint := 'True'} : TON_TIME;   // TIM De Estabilidad de Carga en la Salida por S3
      CNT_pHsMx { S7_SetPoint := 'True'} : "FB910_CNT_UHS";   // CNT de la Presencia
      CNTSeg_pHsMx { S7_SetPoint := 'True'} : "FB910_CNT_UHS";   // CNT de Seguridad de la Presencia
      CNT_ApHsMx { S7_SetPoint := 'True'} : "FB910_CNT_UHS";   // CNT de la Ausencia
      CNTSeg_ApHsMx { S7_SetPoint := 'True'} : "FB910_CNT_UHS";   // CNT de Seguridad de la Ausencia
      TMP_EnTension { S7_SetPoint := 'True'} : "FB910_CNT_UHS";
      TOut_Av_Tx { S7_SetPoint := 'True'} : "FB910_CNT_UHS";   // Time Out de Posicionado de la Carga
      TOut_Av_TRx { S7_SetPoint := 'True'} : "FB910_CNT_UHS";   // Time Out de Entrada de E2
      TOut_Subir_TR { S7_SetPoint := 'True'} : "FB910_CNT_UHS";   // Time Out de Subida del TR
      TOut_Bajar_TR { S7_SetPoint := 'True'} : "FB910_CNT_UHS";   // Time Out de Bajada del TR
      TOut_Subir_TP_E1E3 { S7_SetPoint := 'True'} : "FB910_CNT_UHS";   // Time Out de Subida del TP >> E1E3
      TOut_Bajar_TP_E1E3 { S7_SetPoint := 'True'} : "FB910_CNT_UHS";   // Time Out de Bajada del TP >> E1E3
      TOut_Subir_TP_E2E4 { S7_SetPoint := 'True'} : "FB910_CNT_UHS";   // Time Out de Subida del TP >> E2E4
      TOut_Bajar_TP_E2E4 { S7_SetPoint := 'True'} : "FB910_CNT_UHS";   // Time Out de Bajada del TP >> E2E4
      TOut_Interlock { S7_SetPoint := 'True'} : "FB910_CNT_UHS";   // Time Out de Interlock con el FSS
      CNT_PerdidapHs { S7_SetPoint := 'True'} : "FB910_CNT_UHS";   // CNT de Perdida de pHs
      CNT_HuecoTR1 { S7_SetPoint := 'True'} : "FB910_CNT_UHS";   // CNT de Hueco - Libre TR1
      CNT_HuecoTR2 { S7_SetPoint := 'True'} : "FB910_CNT_UHS";   // CNT de Hueco - Libre TR2
      CNT_PosicionarCarga { S7_SetPoint := 'True'} : "FB910_CNT_UHS";   // CNT Posicionar la Carga en la Mesa a la Entrada
      CNT_PrepararS1 { S7_SetPoint := 'True'} : "FB910_CNT_UHS";   // CNT Prepar la Carga en la Mesa en Salida S1
      CNT_PrepararS3 { S7_SetPoint := 'True'} : "FB910_CNT_UHS";   // CNT Prepar la Carga en la Mesa en Salida S3
      CNT_PresenciaPasarela { S7_SetPoint := 'True'} : "FB910_CNT_UHS";   // CNT Presencia de Carga en la Pasarela
      CNT_AusenciaPasarela { S7_SetPoint := 'True'} : "FB910_CNT_UHS";   // CNT Ausencia de Carga en la Pasarela
      Manual : "MoviManualMesa_FSS";
      Interlock_manual { S7_SetPoint := 'True'} : "UDT_Interlock_manual_TE_FSS";
   END_VAR
   VAR_TEMP
      EstadoZona : "EstadoZona";   // Estado de Zona de la Mesa
      EstadoVI : "EstadosMesa_FSS";   // Estado del Vehiculo Inteliguente de la Mesa
      ConfigFB : "UDT_ConfigFB";   // Configuracion de la FB de la Mesa
      Interlock : "UDT_Interlock_TE_FSS";
      retval : Int;
      cero : USInt;
      Aux_ET00 : Bool;
   END_VAR
   VAR_TEMP   // added for the SCL form of the ladder/FBD networks
      _w1 : Bool;
   END_VAR
BEGIN

REGION Network 1: CONFIGURACION ESPECIAL DE LA FB
   // Mandar Ausencia en el Reset (ON)
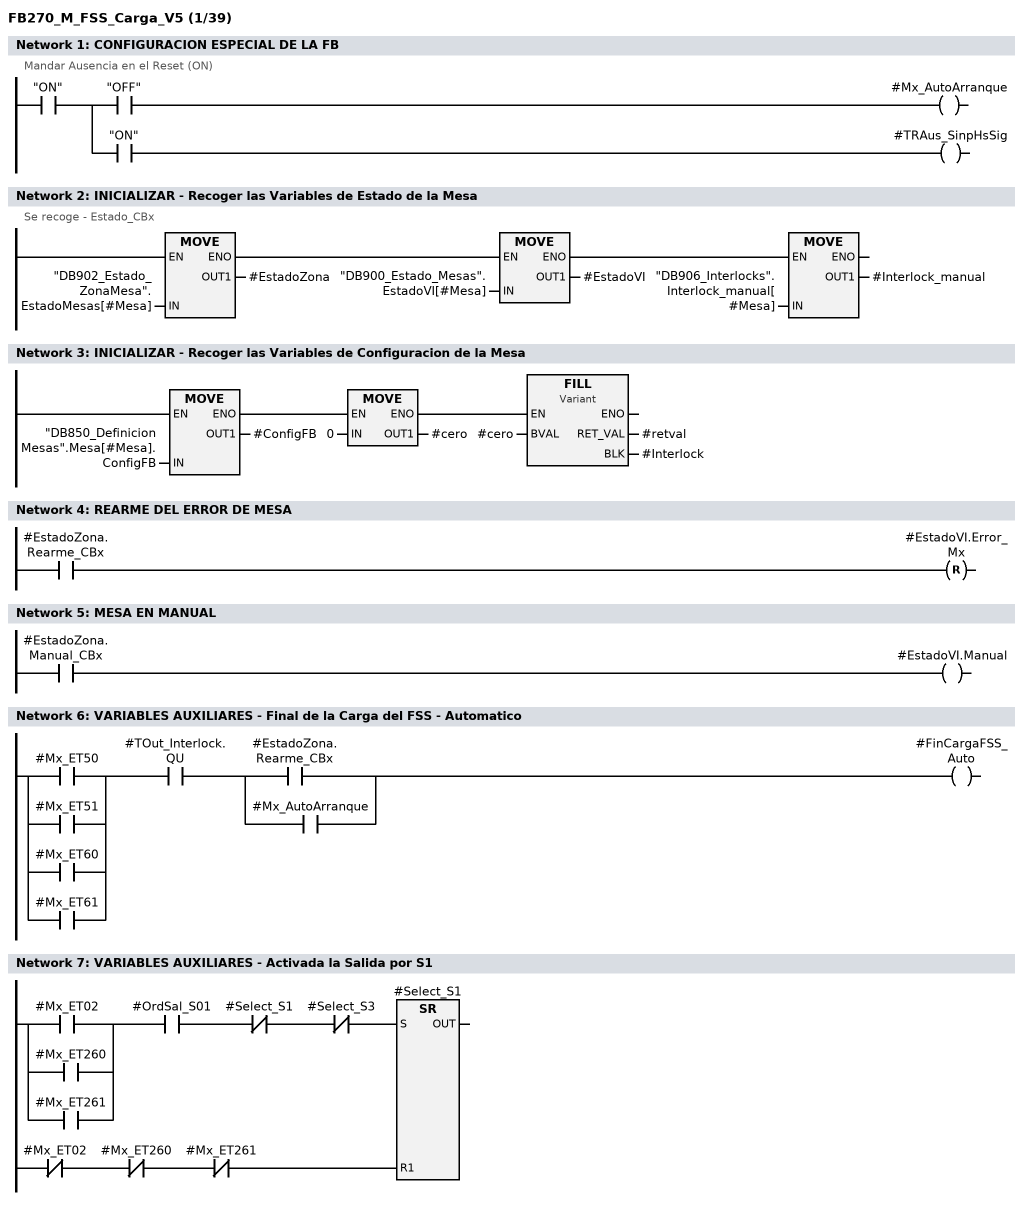
   RUNG wire#powerrail
      Contact( "ON" )
      wire#w1
      Contact( "OFF" )
      Coil( #Mx_AutoArranque )
   END_RUNG
   RUNG wire#w1
      Contact( "ON" )
      Coil( #TRAus_SinpHsSig )
   END_RUNG
   // the same network as SCL:
   #Mx_AutoArranque := "ON" AND "OFF";
   #TRAus_SinpHsSig := "ON" AND "ON";
END_REGION

REGION Network 2: INICIALIZAR - Recoger las Variables de Estado de la Mesa
   // Se recoge - Estado_CBx
   RUNG wire#powerrail
      Move(in := "DB902_Estado_ZonaMesa".EstadoMesas[#Mesa], out1 => #EstadoZona)
      Move(in := "DB900_Estado_Mesas".EstadoVI[#Mesa], out1 => #EstadoVI)
      Move(in := "DB906_Interlocks".Interlock_manual[#Mesa], out1 => #Interlock_manual)
   END_RUNG
   // the same network as SCL:
   #EstadoZona := "DB902_Estado_ZonaMesa".EstadoMesas[#Mesa];
   #EstadoVI := "DB900_Estado_Mesas".EstadoVI[#Mesa];
   #Interlock_manual := "DB906_Interlocks".Interlock_manual[#Mesa];
END_REGION

REGION Network 3: INICIALIZAR - Recoger las Variables de Configuracion de la Mesa
   RUNG wire#powerrail
      Move(in := "DB850_DefinicionMesas".Mesa[#Mesa].ConfigFB, out1 => #ConfigFB)
      Move(in := 0, out1 => #cero)
      { S7_Templates := "ptr_type := Variant" } FILL(BVAL := #cero, RET_VAL => #retval, BLK => #Interlock)
   END_RUNG
   // the same network as SCL:
   #ConfigFB := "DB850_DefinicionMesas".Mesa[#Mesa].ConfigFB;
   #cero := 0;
   #retval := FILL(BVAL := #cero, BLK => #Interlock);
END_REGION

REGION Network 4: REARME DEL ERROR DE MESA
   RUNG wire#powerrail
      Contact( #EstadoZona.Rearme_CBx )
      R_Coil( #EstadoVI.Error_Mx )
   END_RUNG
   // the same network as SCL:
   IF #EstadoZona.Rearme_CBx THEN #EstadoVI.Error_Mx := FALSE; END_IF;
END_REGION

REGION Network 5: MESA EN MANUAL
   RUNG wire#powerrail
      Contact( #EstadoZona.Manual_CBx )
      Coil( #EstadoVI.Manual )
   END_RUNG
   // the same network as SCL:
   #EstadoVI.Manual := #EstadoZona.Manual_CBx;
END_REGION

REGION Network 6: VARIABLES AUXILIARES - Final de la Carga del FSS - Automatico
   RUNG wire#powerrail
      Contact( #Mx_ET50 )
      wire#w1
      Contact( #TOut_Interlock.QU )
      wire#w2
      Contact( #EstadoZona.Rearme_CBx )
      wire#w3
      Coil( #FinCargaFSS_Auto )
   END_RUNG
   RUNG wire#powerrail
      Contact( #Mx_ET51 )
   END_RUNG wire#w1
   RUNG wire#powerrail
      Contact( #Mx_ET60 )
   END_RUNG wire#w1
   RUNG wire#powerrail
      Contact( #Mx_ET61 )
   END_RUNG wire#w1
   RUNG wire#w2
      Contact( #Mx_AutoArranque )
   END_RUNG wire#w3
   // the same network as SCL:
   #FinCargaFSS_Auto := (#Mx_ET50 OR #Mx_ET51 OR #Mx_ET60 OR #Mx_ET61) AND #TOut_Interlock.QU AND (#EstadoZona.Rearme_CBx OR #Mx_AutoArranque);
END_REGION

REGION Network 7: VARIABLES AUXILIARES - Activada la Salida por S1
   RUNG wire#powerrail
      Contact( #Mx_ET02 )
      wire#w1
      Contact( #OrdSal_S01 )
      I_Contact( #Select_S1 )
      I_Contact( #Select_S3 )
      S_SR(operand := #Select_S1, r1 := wire#w2)
   END_RUNG
   RUNG wire#powerrail
      Contact( #Mx_ET260 )
   END_RUNG wire#w1
   RUNG wire#powerrail
      Contact( #Mx_ET261 )
   END_RUNG wire#w1
   RUNG wire#powerrail
      I_Contact( #Mx_ET02 )
      I_Contact( #Mx_ET260 )
      I_Contact( #Mx_ET261 )
   END_RUNG wire#w2
   // the same network as SCL:
   IF (#Mx_ET02 OR #Mx_ET260 OR #Mx_ET261) AND #OrdSal_S01 AND NOT #Select_S1 AND NOT #Select_S3 THEN
       #Select_S1 := TRUE;   // SR flip-flop
   END_IF;
   IF NOT #Mx_ET02 AND NOT #Mx_ET260 AND NOT #Mx_ET261 THEN #Select_S1 := FALSE; END_IF;
END_REGION

REGION Network 8: VARIABLES AUXILIARES - Activada la Salida por S3
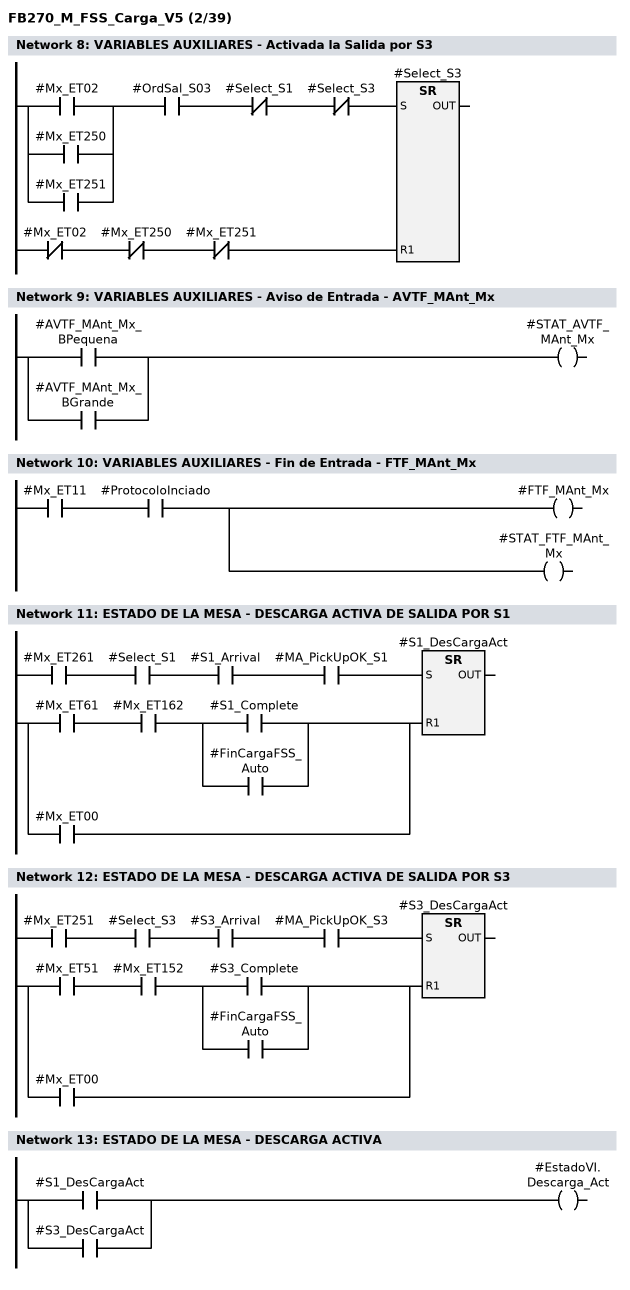
   RUNG wire#powerrail
      Contact( #Mx_ET02 )
      wire#w1
      Contact( #OrdSal_S03 )
      I_Contact( #Select_S1 )
      I_Contact( #Select_S3 )
      S_SR(operand := #Select_S3, r1 := wire#w2)
   END_RUNG
   RUNG wire#powerrail
      Contact( #Mx_ET250 )
   END_RUNG wire#w1
   RUNG wire#powerrail
      Contact( #Mx_ET251 )
   END_RUNG wire#w1
   RUNG wire#powerrail
      I_Contact( #Mx_ET02 )
      I_Contact( #Mx_ET250 )
      I_Contact( #Mx_ET251 )
   END_RUNG wire#w2
   // the same network as SCL:
   IF (#Mx_ET02 OR #Mx_ET250 OR #Mx_ET251) AND #OrdSal_S03 AND NOT #Select_S1 AND NOT #Select_S3 THEN
       #Select_S3 := TRUE;   // SR flip-flop
   END_IF;
   IF NOT #Mx_ET02 AND NOT #Mx_ET250 AND NOT #Mx_ET251 THEN #Select_S3 := FALSE; END_IF;
END_REGION

REGION Network 9: VARIABLES AUXILIARES - Aviso de Entrada - AVTF_MAnt_Mx
   RUNG wire#powerrail
      Contact( #AVTF_MAnt_Mx_BPequena )
      wire#w1
      Coil( #STAT_AVTF_MAnt_Mx )
   END_RUNG
   RUNG wire#powerrail
      Contact( #AVTF_MAnt_Mx_BGrande )
   END_RUNG wire#w1
   // the same network as SCL:
   #STAT_AVTF_MAnt_Mx := #AVTF_MAnt_Mx_BPequena OR #AVTF_MAnt_Mx_BGrande;
END_REGION

REGION Network 10: VARIABLES AUXILIARES - Fin de Entrada - FTF_MAnt_Mx
   RUNG wire#powerrail
      Contact( #Mx_ET11 )
      Contact( #ProtocoloInciado )
      wire#w1
      Coil( #FTF_MAnt_Mx )
   END_RUNG
   RUNG wire#w1
      Coil( #STAT_FTF_MAnt_Mx )
   END_RUNG
   // the same network as SCL:
   #FTF_MAnt_Mx := #Mx_ET11 AND #ProtocoloInciado;
   #STAT_FTF_MAnt_Mx := #FTF_MAnt_Mx;
END_REGION

REGION Network 11: ESTADO DE LA MESA - DESCARGA ACTIVA DE SALIDA POR S1
   RUNG wire#powerrail
      Contact( #Mx_ET261 )
      Contact( #Select_S1 )
      Contact( #S1_Arrival )
      Contact( #MA_PickUpOK_S1 )
      S_SR(operand := #S1_DesCargaAct, r1 := wire#w2)
   END_RUNG
   RUNG wire#powerrail
      Contact( #Mx_ET61 )
      Contact( #Mx_ET162 )
      wire#w1
      Contact( #S1_Complete )
   END_RUNG wire#w2
   RUNG wire#w1
      Contact( #FinCargaFSS_Auto )
   END_RUNG wire#w2
   RUNG wire#powerrail
      Contact( #Mx_ET00 )
   END_RUNG wire#w2
   // the same network as SCL:
   IF #Mx_ET261 AND #Select_S1 AND #S1_Arrival AND #MA_PickUpOK_S1 THEN
       #S1_DesCargaAct := TRUE;   // SR flip-flop
   END_IF;
   IF (#Mx_ET61 AND #Mx_ET162 AND (#S1_Complete OR #FinCargaFSS_Auto)) OR #Mx_ET00 THEN
       #S1_DesCargaAct := FALSE;
   END_IF;
END_REGION

REGION Network 12: ESTADO DE LA MESA - DESCARGA ACTIVA DE SALIDA POR S3
   RUNG wire#powerrail
      Contact( #Mx_ET251 )
      Contact( #Select_S3 )
      Contact( #S3_Arrival )
      Contact( #MA_PickUpOK_S3 )
      S_SR(operand := #S3_DesCargaAct, r1 := wire#w2)
   END_RUNG
   RUNG wire#powerrail
      Contact( #Mx_ET51 )
      Contact( #Mx_ET152 )
      wire#w1
      Contact( #S3_Complete )
   END_RUNG wire#w2
   RUNG wire#w1
      Contact( #FinCargaFSS_Auto )
   END_RUNG wire#w2
   RUNG wire#powerrail
      Contact( #Mx_ET00 )
   END_RUNG wire#w2
   // the same network as SCL:
   IF #Mx_ET251 AND #Select_S3 AND #S3_Arrival AND #MA_PickUpOK_S3 THEN
       #S3_DesCargaAct := TRUE;   // SR flip-flop
   END_IF;
   IF (#Mx_ET51 AND #Mx_ET152 AND (#S3_Complete OR #FinCargaFSS_Auto)) OR #Mx_ET00 THEN
       #S3_DesCargaAct := FALSE;
   END_IF;
END_REGION

REGION Network 13: ESTADO DE LA MESA - DESCARGA ACTIVA
   RUNG wire#powerrail
      Contact( #S1_DesCargaAct )
      wire#w1
      Coil( #EstadoVI.Descarga_Act )
   END_RUNG
   RUNG wire#powerrail
      Contact( #S3_DesCargaAct )
   END_RUNG wire#w1
   // the same network as SCL:
   #EstadoVI.Descarga_Act := #S1_DesCargaAct OR #S3_DesCargaAct;
END_REGION

REGION Network 14: ET92 - ACTIVACION DE PASARELA - OCUPADA LA MESA
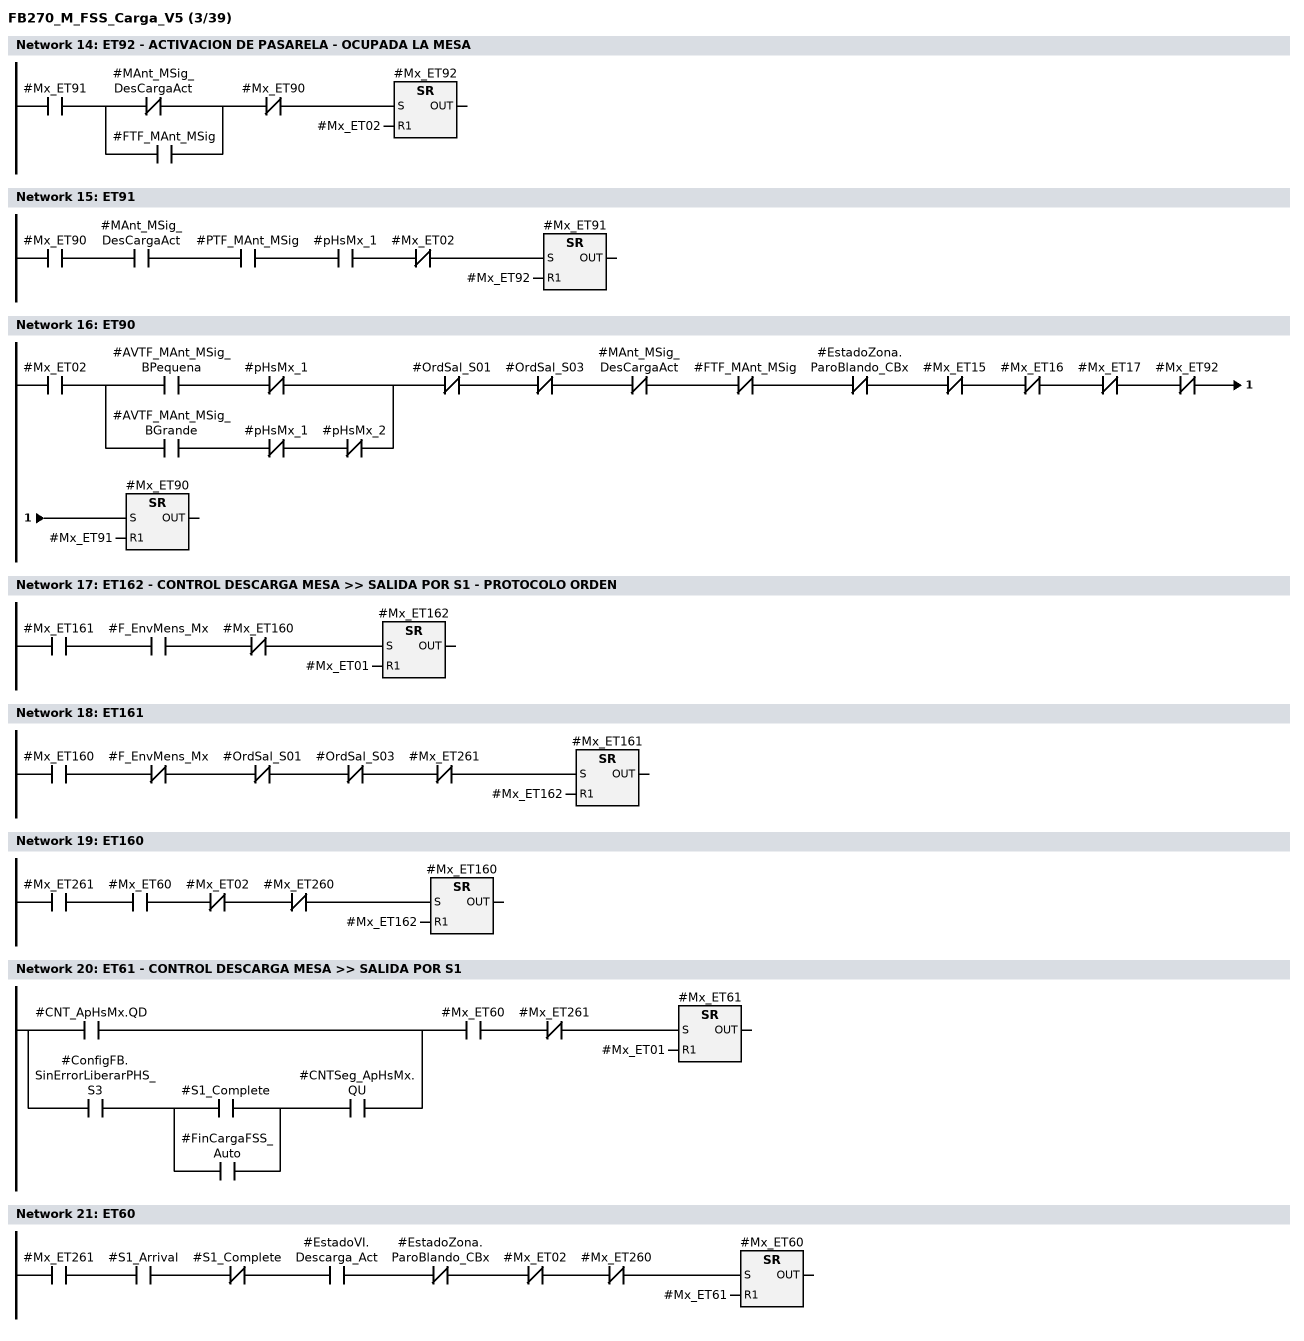
   RUNG wire#powerrail
      Contact( #Mx_ET91 )
      wire#w1
      I_Contact( #MAnt_MSig_DesCargaAct )
      wire#w2
      I_Contact( #Mx_ET90 )
      S_SR(operand := #Mx_ET92, r1 := #Mx_ET02)
   END_RUNG
   RUNG wire#w1
      Contact( #FTF_MAnt_MSig )
   END_RUNG wire#w2
   // the same network as SCL:
   IF #Mx_ET91 AND (NOT #MAnt_MSig_DesCargaAct OR #FTF_MAnt_MSig) AND NOT #Mx_ET90 THEN
       #Mx_ET92 := TRUE;   // SR flip-flop
   END_IF;
   IF #Mx_ET02 THEN #Mx_ET92 := FALSE; END_IF;
END_REGION

REGION Network 15: ET91
   RUNG wire#powerrail
      Contact( #Mx_ET90 )
      Contact( #MAnt_MSig_DesCargaAct )
      Contact( #PTF_MAnt_MSig )
      Contact( #pHsMx_1 )
      I_Contact( #Mx_ET02 )
      S_SR(operand := #Mx_ET91, r1 := #Mx_ET92)
   END_RUNG
   // the same network as SCL:
   IF #Mx_ET90 AND #MAnt_MSig_DesCargaAct AND #PTF_MAnt_MSig AND #pHsMx_1 AND NOT #Mx_ET02 THEN
       #Mx_ET91 := TRUE;   // SR flip-flop
   END_IF;
   IF #Mx_ET92 THEN #Mx_ET91 := FALSE; END_IF;
END_REGION

REGION Network 16: ET90
   RUNG wire#powerrail
      Contact( #Mx_ET02 )
      wire#w1
      Contact( #AVTF_MAnt_MSig_BPequena )
      I_Contact( #pHsMx_1 )
      wire#w2
      I_Contact( #OrdSal_S01 )
      I_Contact( #OrdSal_S03 )
      I_Contact( #MAnt_MSig_DesCargaAct )
      I_Contact( #FTF_MAnt_MSig )
      I_Contact( #EstadoZona.ParoBlando_CBx )
      I_Contact( #Mx_ET15 )
      I_Contact( #Mx_ET16 )
      I_Contact( #Mx_ET17 )
      I_Contact( #Mx_ET92 )
      S_SR(operand := #Mx_ET90, r1 := #Mx_ET91)
   END_RUNG
   RUNG wire#w1
      Contact( #AVTF_MAnt_MSig_BGrande )
      I_Contact( #pHsMx_1 )
      I_Contact( #pHsMx_2 )
   END_RUNG wire#w2
   // the same network as SCL:
   IF #Mx_ET02 AND ((#AVTF_MAnt_MSig_BPequena AND NOT #pHsMx_1) OR (#AVTF_MAnt_MSig_BGrande AND NOT #pHsMx_1 AND NOT #pHsMx_2)) AND NOT #OrdSal_S01 AND NOT #OrdSal_S03 AND NOT #MAnt_MSig_DesCargaAct AND NOT #FTF_MAnt_MSig AND NOT #EstadoZona.ParoBlando_CBx AND NOT #Mx_ET15 AND NOT #Mx_ET16 AND NOT #Mx_ET17 AND NOT #Mx_ET92 THEN
       #Mx_ET90 := TRUE;   // SR flip-flop
   END_IF;
   IF #Mx_ET91 THEN #Mx_ET90 := FALSE; END_IF;
END_REGION

REGION Network 17: ET162 - CONTROL DESCARGA MESA >> SALIDA POR S1 - PROTOCOLO ORDEN
   RUNG wire#powerrail
      Contact( #Mx_ET161 )
      Contact( #F_EnvMens_Mx )
      I_Contact( #Mx_ET160 )
      S_SR(operand := #Mx_ET162, r1 := #Mx_ET01)
   END_RUNG
   // the same network as SCL:
   IF #Mx_ET161 AND #F_EnvMens_Mx AND NOT #Mx_ET160 THEN
       #Mx_ET162 := TRUE;   // SR flip-flop
   END_IF;
   IF #Mx_ET01 THEN #Mx_ET162 := FALSE; END_IF;
END_REGION

REGION Network 18: ET161
   RUNG wire#powerrail
      Contact( #Mx_ET160 )
      I_Contact( #F_EnvMens_Mx )
      I_Contact( #OrdSal_S01 )
      I_Contact( #OrdSal_S03 )
      I_Contact( #Mx_ET261 )
      S_SR(operand := #Mx_ET161, r1 := #Mx_ET162)
   END_RUNG
   // the same network as SCL:
   IF #Mx_ET160 AND NOT #F_EnvMens_Mx AND NOT #OrdSal_S01 AND NOT #OrdSal_S03 AND NOT #Mx_ET261 THEN
       #Mx_ET161 := TRUE;   // SR flip-flop
   END_IF;
   IF #Mx_ET162 THEN #Mx_ET161 := FALSE; END_IF;
END_REGION

REGION Network 19: ET160
   RUNG wire#powerrail
      Contact( #Mx_ET261 )
      Contact( #Mx_ET60 )
      I_Contact( #Mx_ET02 )
      I_Contact( #Mx_ET260 )
      S_SR(operand := #Mx_ET160, r1 := #Mx_ET162)
   END_RUNG
   // the same network as SCL:
   IF #Mx_ET261 AND #Mx_ET60 AND NOT #Mx_ET02 AND NOT #Mx_ET260 THEN
       #Mx_ET160 := TRUE;   // SR flip-flop
   END_IF;
   IF #Mx_ET162 THEN #Mx_ET160 := FALSE; END_IF;
END_REGION

REGION Network 20: ET61 - CONTROL DESCARGA MESA >> SALIDA POR S1
   RUNG wire#powerrail
      Contact( #CNT_ApHsMx.QD )
      wire#w1
      Contact( #Mx_ET60 )
      I_Contact( #Mx_ET261 )
      S_SR(operand := #Mx_ET61, r1 := #Mx_ET01)
   END_RUNG
   RUNG wire#powerrail
      Contact( #ConfigFB.SinErrorLiberarPHS_S3 )
      wire#w2
      Contact( #S1_Complete )
      wire#w3
      Contact( #CNTSeg_ApHsMx.QU )
   END_RUNG wire#w1
   RUNG wire#w2
      Contact( #FinCargaFSS_Auto )
   END_RUNG wire#w3
   // the same network as SCL:
   IF (#CNT_ApHsMx.QD OR (#ConfigFB.SinErrorLiberarPHS_S3 AND (#S1_Complete OR #FinCargaFSS_Auto) AND #CNTSeg_ApHsMx.QU)) AND #Mx_ET60 AND NOT #Mx_ET261 THEN
       #Mx_ET61 := TRUE;   // SR flip-flop
   END_IF;
   IF #Mx_ET01 THEN #Mx_ET61 := FALSE; END_IF;
END_REGION

REGION Network 21: ET60
   RUNG wire#powerrail
      Contact( #Mx_ET261 )
      Contact( #S1_Arrival )
      I_Contact( #S1_Complete )
      Contact( #EstadoVI.Descarga_Act )
      I_Contact( #EstadoZona.ParoBlando_CBx )
      I_Contact( #Mx_ET02 )
      I_Contact( #Mx_ET260 )
      S_SR(operand := #Mx_ET60, r1 := #Mx_ET61)
   END_RUNG
   // the same network as SCL:
   IF #Mx_ET261 AND #S1_Arrival AND NOT #S1_Complete AND #EstadoVI.Descarga_Act AND NOT #EstadoZona.ParoBlando_CBx AND NOT #Mx_ET02 AND NOT #Mx_ET260 THEN
       #Mx_ET60 := TRUE;   // SR flip-flop
   END_IF;
   IF #Mx_ET61 THEN #Mx_ET60 := FALSE; END_IF;
END_REGION

REGION Network 22: ET261 - POSICIONAMIENTO PREVIO PARA LA DESCARGA MESA >> SALIDA POR S1
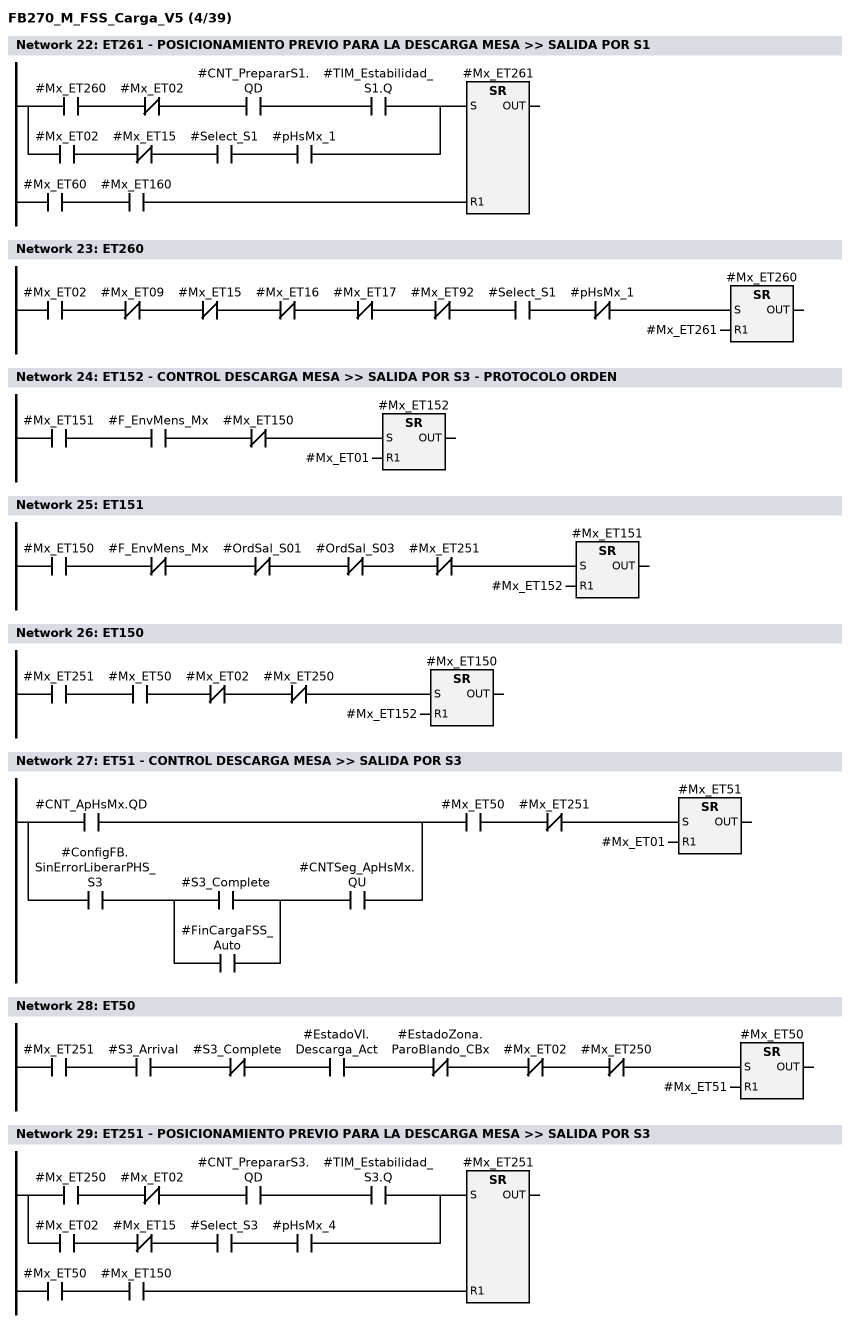
   RUNG wire#powerrail
      Contact( #Mx_ET260 )
      I_Contact( #Mx_ET02 )
      Contact( #CNT_PrepararS1.QD )
      Contact( #TIM_Estabilidad_S1.Q )
      wire#w1
      S_SR(operand := #Mx_ET261, r1 := wire#w2)
   END_RUNG
   RUNG wire#powerrail
      Contact( #Mx_ET02 )
      I_Contact( #Mx_ET15 )
      Contact( #Select_S1 )
      Contact( #pHsMx_1 )
   END_RUNG wire#w1
   RUNG wire#powerrail
      Contact( #Mx_ET60 )
      Contact( #Mx_ET160 )
   END_RUNG wire#w2
   // the same network as SCL:
   IF (#Mx_ET260 AND NOT #Mx_ET02 AND #CNT_PrepararS1.QD AND #TIM_Estabilidad_S1.Q) OR (#Mx_ET02 AND NOT #Mx_ET15 AND #Select_S1 AND #pHsMx_1) THEN
       #Mx_ET261 := TRUE;   // SR flip-flop
   END_IF;
   IF #Mx_ET60 AND #Mx_ET160 THEN #Mx_ET261 := FALSE; END_IF;
END_REGION

REGION Network 23: ET260
   RUNG wire#powerrail
      Contact( #Mx_ET02 )
      I_Contact( #Mx_ET09 )
      I_Contact( #Mx_ET15 )
      I_Contact( #Mx_ET16 )
      I_Contact( #Mx_ET17 )
      I_Contact( #Mx_ET92 )
      Contact( #Select_S1 )
      I_Contact( #pHsMx_1 )
      S_SR(operand := #Mx_ET260, r1 := #Mx_ET261)
   END_RUNG
   // the same network as SCL:
   IF #Mx_ET02 AND NOT #Mx_ET09 AND NOT #Mx_ET15 AND NOT #Mx_ET16 AND NOT #Mx_ET17 AND NOT #Mx_ET92 AND #Select_S1 AND NOT #pHsMx_1 THEN
       #Mx_ET260 := TRUE;   // SR flip-flop
   END_IF;
   IF #Mx_ET261 THEN #Mx_ET260 := FALSE; END_IF;
END_REGION

REGION Network 24: ET152 - CONTROL DESCARGA MESA >> SALIDA POR S3 - PROTOCOLO ORDEN
   RUNG wire#powerrail
      Contact( #Mx_ET151 )
      Contact( #F_EnvMens_Mx )
      I_Contact( #Mx_ET150 )
      S_SR(operand := #Mx_ET152, r1 := #Mx_ET01)
   END_RUNG
   // the same network as SCL:
   IF #Mx_ET151 AND #F_EnvMens_Mx AND NOT #Mx_ET150 THEN
       #Mx_ET152 := TRUE;   // SR flip-flop
   END_IF;
   IF #Mx_ET01 THEN #Mx_ET152 := FALSE; END_IF;
END_REGION

REGION Network 25: ET151
   RUNG wire#powerrail
      Contact( #Mx_ET150 )
      I_Contact( #F_EnvMens_Mx )
      I_Contact( #OrdSal_S01 )
      I_Contact( #OrdSal_S03 )
      I_Contact( #Mx_ET251 )
      S_SR(operand := #Mx_ET151, r1 := #Mx_ET152)
   END_RUNG
   // the same network as SCL:
   IF #Mx_ET150 AND NOT #F_EnvMens_Mx AND NOT #OrdSal_S01 AND NOT #OrdSal_S03 AND NOT #Mx_ET251 THEN
       #Mx_ET151 := TRUE;   // SR flip-flop
   END_IF;
   IF #Mx_ET152 THEN #Mx_ET151 := FALSE; END_IF;
END_REGION

REGION Network 26: ET150
   RUNG wire#powerrail
      Contact( #Mx_ET251 )
      Contact( #Mx_ET50 )
      I_Contact( #Mx_ET02 )
      I_Contact( #Mx_ET250 )
      S_SR(operand := #Mx_ET150, r1 := #Mx_ET152)
   END_RUNG
   // the same network as SCL:
   IF #Mx_ET251 AND #Mx_ET50 AND NOT #Mx_ET02 AND NOT #Mx_ET250 THEN
       #Mx_ET150 := TRUE;   // SR flip-flop
   END_IF;
   IF #Mx_ET152 THEN #Mx_ET150 := FALSE; END_IF;
END_REGION

REGION Network 27: ET51 - CONTROL DESCARGA MESA >> SALIDA POR S3
   RUNG wire#powerrail
      Contact( #CNT_ApHsMx.QD )
      wire#w1
      Contact( #Mx_ET50 )
      I_Contact( #Mx_ET251 )
      S_SR(operand := #Mx_ET51, r1 := #Mx_ET01)
   END_RUNG
   RUNG wire#powerrail
      Contact( #ConfigFB.SinErrorLiberarPHS_S3 )
      wire#w2
      Contact( #S3_Complete )
      wire#w3
      Contact( #CNTSeg_ApHsMx.QU )
   END_RUNG wire#w1
   RUNG wire#w2
      Contact( #FinCargaFSS_Auto )
   END_RUNG wire#w3
   // the same network as SCL:
   IF (#CNT_ApHsMx.QD OR (#ConfigFB.SinErrorLiberarPHS_S3 AND (#S3_Complete OR #FinCargaFSS_Auto) AND #CNTSeg_ApHsMx.QU)) AND #Mx_ET50 AND NOT #Mx_ET251 THEN
       #Mx_ET51 := TRUE;   // SR flip-flop
   END_IF;
   IF #Mx_ET01 THEN #Mx_ET51 := FALSE; END_IF;
END_REGION

REGION Network 28: ET50
   RUNG wire#powerrail
      Contact( #Mx_ET251 )
      Contact( #S3_Arrival )
      I_Contact( #S3_Complete )
      Contact( #EstadoVI.Descarga_Act )
      I_Contact( #EstadoZona.ParoBlando_CBx )
      I_Contact( #Mx_ET02 )
      I_Contact( #Mx_ET250 )
      S_SR(operand := #Mx_ET50, r1 := #Mx_ET51)
   END_RUNG
   // the same network as SCL:
   IF #Mx_ET251 AND #S3_Arrival AND NOT #S3_Complete AND #EstadoVI.Descarga_Act AND NOT #EstadoZona.ParoBlando_CBx AND NOT #Mx_ET02 AND NOT #Mx_ET250 THEN
       #Mx_ET50 := TRUE;   // SR flip-flop
   END_IF;
   IF #Mx_ET51 THEN #Mx_ET50 := FALSE; END_IF;
END_REGION

REGION Network 29: ET251 - POSICIONAMIENTO PREVIO PARA LA DESCARGA MESA >> SALIDA POR S3
   RUNG wire#powerrail
      Contact( #Mx_ET250 )
      I_Contact( #Mx_ET02 )
      Contact( #CNT_PrepararS3.QD )
      Contact( #TIM_Estabilidad_S3.Q )
      wire#w1
      S_SR(operand := #Mx_ET251, r1 := wire#w2)
   END_RUNG
   RUNG wire#powerrail
      Contact( #Mx_ET02 )
      I_Contact( #Mx_ET15 )
      Contact( #Select_S3 )
      Contact( #pHsMx_4 )
   END_RUNG wire#w1
   RUNG wire#powerrail
      Contact( #Mx_ET50 )
      Contact( #Mx_ET150 )
   END_RUNG wire#w2
   // the same network as SCL:
   IF (#Mx_ET250 AND NOT #Mx_ET02 AND #CNT_PrepararS3.QD AND #TIM_Estabilidad_S3.Q) OR (#Mx_ET02 AND NOT #Mx_ET15 AND #Select_S3 AND #pHsMx_4) THEN
       #Mx_ET251 := TRUE;   // SR flip-flop
   END_IF;
   IF #Mx_ET50 AND #Mx_ET150 THEN #Mx_ET251 := FALSE; END_IF;
END_REGION

REGION Network 30: ET250
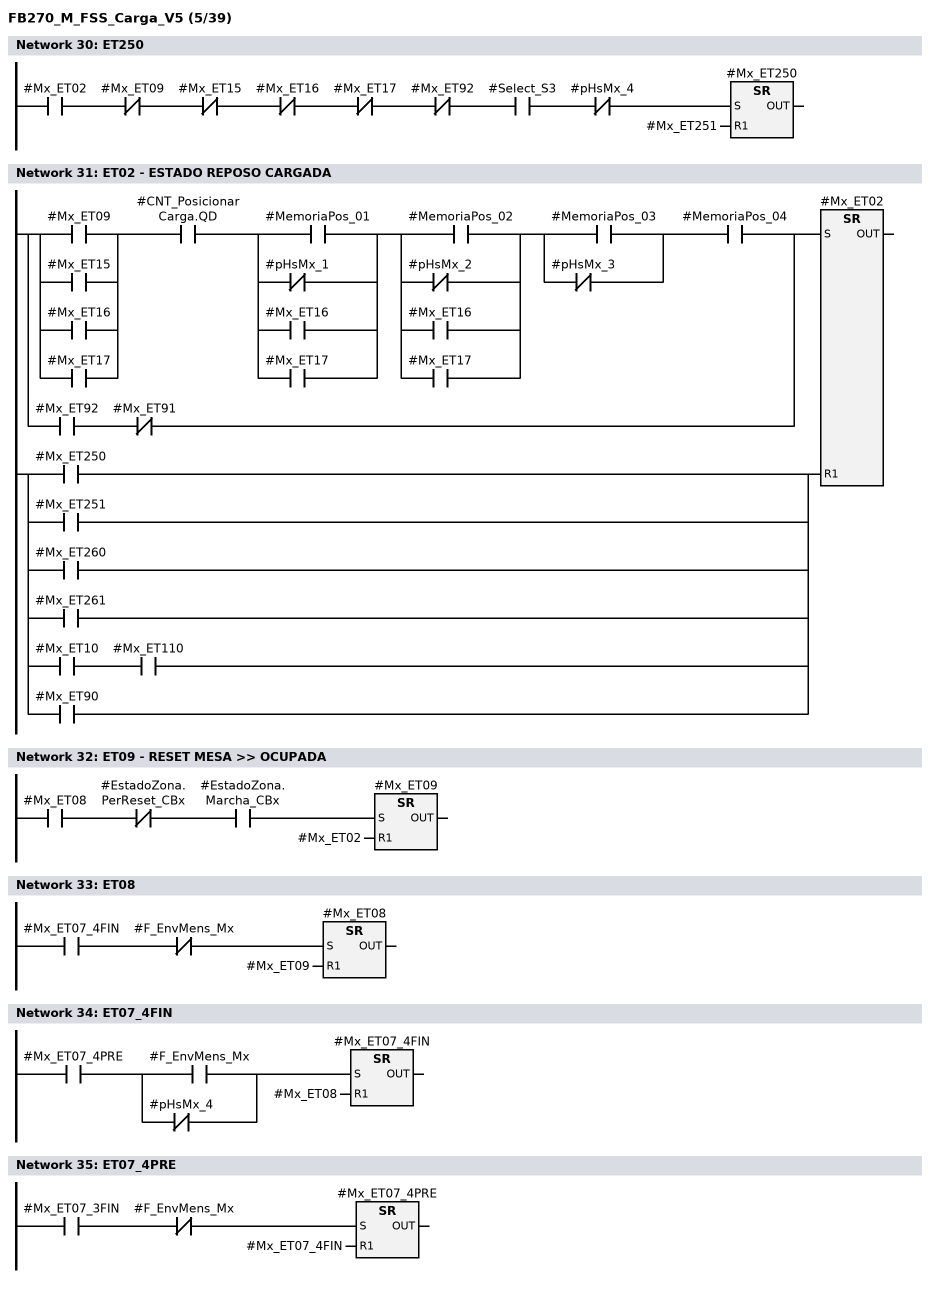
   RUNG wire#powerrail
      Contact( #Mx_ET02 )
      I_Contact( #Mx_ET09 )
      I_Contact( #Mx_ET15 )
      I_Contact( #Mx_ET16 )
      I_Contact( #Mx_ET17 )
      I_Contact( #Mx_ET92 )
      Contact( #Select_S3 )
      I_Contact( #pHsMx_4 )
      S_SR(operand := #Mx_ET250, r1 := #Mx_ET251)
   END_RUNG
   // the same network as SCL:
   IF #Mx_ET02 AND NOT #Mx_ET09 AND NOT #Mx_ET15 AND NOT #Mx_ET16 AND NOT #Mx_ET17 AND NOT #Mx_ET92 AND #Select_S3 AND NOT #pHsMx_4 THEN
       #Mx_ET250 := TRUE;   // SR flip-flop
   END_IF;
   IF #Mx_ET251 THEN #Mx_ET250 := FALSE; END_IF;
END_REGION

REGION Network 31: ET02 - ESTADO REPOSO CARGADA
   RUNG wire#powerrail
      Contact( #Mx_ET09 )
      wire#w1
      Contact( #CNT_PosicionarCarga.QD )
      wire#w2
      Contact( #MemoriaPos_01 )
      wire#w3
      Contact( #MemoriaPos_02 )
      wire#w4
      Contact( #MemoriaPos_03 )
      wire#w5
      Contact( #MemoriaPos_04 )
      wire#w6
      S_SR(operand := #Mx_ET02, r1 := wire#w7)
   END_RUNG
   RUNG wire#powerrail
      Contact( #Mx_ET15 )
   END_RUNG wire#w1
   RUNG wire#powerrail
      Contact( #Mx_ET16 )
   END_RUNG wire#w1
   RUNG wire#powerrail
      Contact( #Mx_ET17 )
   END_RUNG wire#w1
   RUNG wire#w2
      I_Contact( #pHsMx_1 )
   END_RUNG wire#w3
   RUNG wire#w2
      Contact( #Mx_ET16 )
   END_RUNG wire#w3
   RUNG wire#w2
      Contact( #Mx_ET17 )
   END_RUNG wire#w3
   RUNG wire#w3
      I_Contact( #pHsMx_2 )
   END_RUNG wire#w4
   RUNG wire#w3
      Contact( #Mx_ET16 )
   END_RUNG wire#w4
   RUNG wire#w3
      Contact( #Mx_ET17 )
   END_RUNG wire#w4
   RUNG wire#w4
      I_Contact( #pHsMx_3 )
   END_RUNG wire#w5
   RUNG wire#powerrail
      Contact( #Mx_ET92 )
      I_Contact( #Mx_ET91 )
   END_RUNG wire#w6
   RUNG wire#powerrail
      Contact( #Mx_ET250 )
   END_RUNG wire#w7
   RUNG wire#powerrail
      Contact( #Mx_ET251 )
   END_RUNG wire#w7
   RUNG wire#powerrail
      Contact( #Mx_ET260 )
   END_RUNG wire#w7
   RUNG wire#powerrail
      Contact( #Mx_ET261 )
   END_RUNG wire#w7
   RUNG wire#powerrail
      Contact( #Mx_ET10 )
      Contact( #Mx_ET110 )
   END_RUNG wire#w7
   RUNG wire#powerrail
      Contact( #Mx_ET90 )
   END_RUNG wire#w7
   // the same network as SCL:
   IF ((#Mx_ET09 OR #Mx_ET15 OR #Mx_ET16 OR #Mx_ET17) AND #CNT_PosicionarCarga.QD AND (#MemoriaPos_01 OR NOT #pHsMx_1 OR #Mx_ET16 OR #Mx_ET17) AND (#MemoriaPos_02 OR NOT #pHsMx_2 OR #Mx_ET16 OR #Mx_ET17) AND (#MemoriaPos_03 OR NOT #pHsMx_3) AND #MemoriaPos_04) OR (#Mx_ET92 AND NOT #Mx_ET91) THEN
       #Mx_ET02 := TRUE;   // SR flip-flop
   END_IF;
   IF #Mx_ET250 OR #Mx_ET251 OR #Mx_ET260 OR #Mx_ET261 OR (#Mx_ET10 AND #Mx_ET110) OR #Mx_ET90 THEN
       #Mx_ET02 := FALSE;
   END_IF;
END_REGION

REGION Network 32: ET09 - RESET MESA >> OCUPADA
   RUNG wire#powerrail
      Contact( #Mx_ET08 )
      I_Contact( #EstadoZona.PerReset_CBx )
      Contact( #EstadoZona.Marcha_CBx )
      S_SR(operand := #Mx_ET09, r1 := #Mx_ET02)
   END_RUNG
   // the same network as SCL:
   IF #Mx_ET08 AND NOT #EstadoZona.PerReset_CBx AND #EstadoZona.Marcha_CBx THEN
       #Mx_ET09 := TRUE;   // SR flip-flop
   END_IF;
   IF #Mx_ET02 THEN #Mx_ET09 := FALSE; END_IF;
END_REGION

REGION Network 33: ET08
   RUNG wire#powerrail
      Contact( #Mx_ET07_4FIN )
      I_Contact( #F_EnvMens_Mx )
      S_SR(operand := #Mx_ET08, r1 := #Mx_ET09)
   END_RUNG
   // the same network as SCL:
   IF #Mx_ET07_4FIN AND NOT #F_EnvMens_Mx THEN
       #Mx_ET08 := TRUE;   // SR flip-flop
   END_IF;
   IF #Mx_ET09 THEN #Mx_ET08 := FALSE; END_IF;
END_REGION

REGION Network 34: ET07_4FIN
   RUNG wire#powerrail
      Contact( #Mx_ET07_4PRE )
      wire#w1
      Contact( #F_EnvMens_Mx )
      wire#w2
      S_SR(operand := #Mx_ET07_4FIN, r1 := #Mx_ET08)
   END_RUNG
   RUNG wire#w1
      I_Contact( #pHsMx_4 )
   END_RUNG wire#w2
   // the same network as SCL:
   IF #Mx_ET07_4PRE AND (#F_EnvMens_Mx OR NOT #pHsMx_4) THEN
       #Mx_ET07_4FIN := TRUE;   // SR flip-flop
   END_IF;
   IF #Mx_ET08 THEN #Mx_ET07_4FIN := FALSE; END_IF;
END_REGION

REGION Network 35: ET07_4PRE
   RUNG wire#powerrail
      Contact( #Mx_ET07_3FIN )
      I_Contact( #F_EnvMens_Mx )
      S_SR(operand := #Mx_ET07_4PRE, r1 := #Mx_ET07_4FIN)
   END_RUNG
   // the same network as SCL:
   IF #Mx_ET07_3FIN AND NOT #F_EnvMens_Mx THEN
       #Mx_ET07_4PRE := TRUE;   // SR flip-flop
   END_IF;
   IF #Mx_ET07_4FIN THEN #Mx_ET07_4PRE := FALSE; END_IF;
END_REGION

REGION Network 36: ET07_3FIN
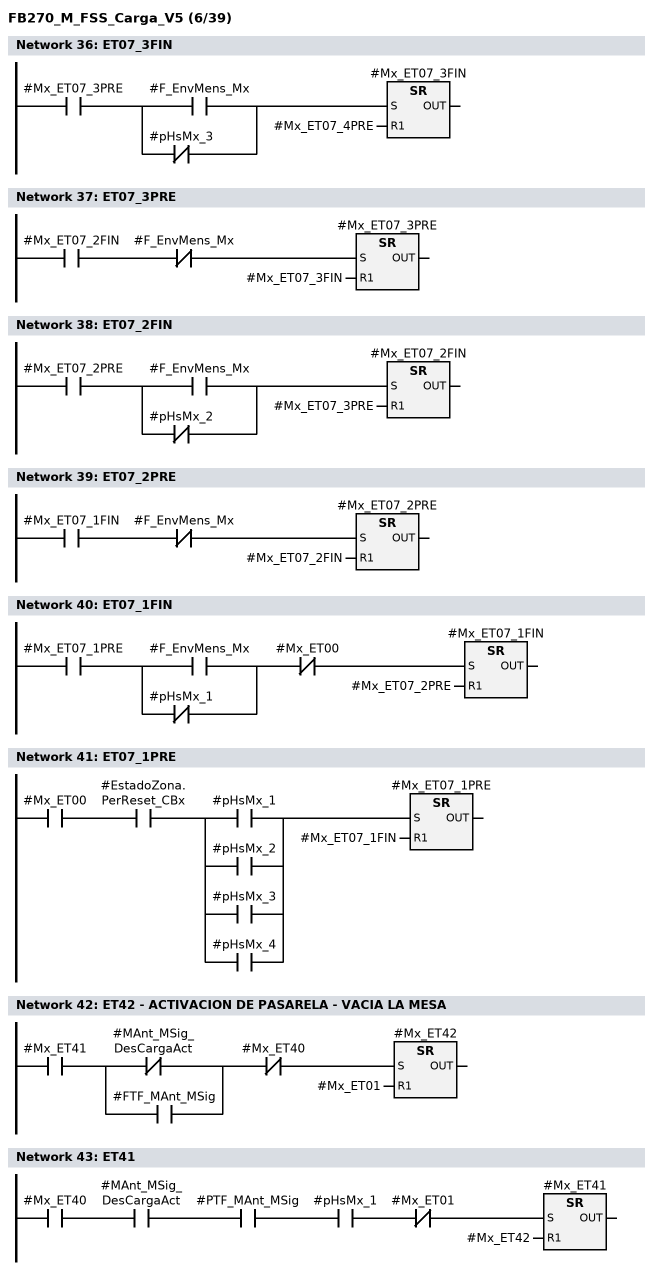
   RUNG wire#powerrail
      Contact( #Mx_ET07_3PRE )
      wire#w1
      Contact( #F_EnvMens_Mx )
      wire#w2
      S_SR(operand := #Mx_ET07_3FIN, r1 := #Mx_ET07_4PRE)
   END_RUNG
   RUNG wire#w1
      I_Contact( #pHsMx_3 )
   END_RUNG wire#w2
   // the same network as SCL:
   IF #Mx_ET07_3PRE AND (#F_EnvMens_Mx OR NOT #pHsMx_3) THEN
       #Mx_ET07_3FIN := TRUE;   // SR flip-flop
   END_IF;
   IF #Mx_ET07_4PRE THEN #Mx_ET07_3FIN := FALSE; END_IF;
END_REGION

REGION Network 37: ET07_3PRE
   RUNG wire#powerrail
      Contact( #Mx_ET07_2FIN )
      I_Contact( #F_EnvMens_Mx )
      S_SR(operand := #Mx_ET07_3PRE, r1 := #Mx_ET07_3FIN)
   END_RUNG
   // the same network as SCL:
   IF #Mx_ET07_2FIN AND NOT #F_EnvMens_Mx THEN
       #Mx_ET07_3PRE := TRUE;   // SR flip-flop
   END_IF;
   IF #Mx_ET07_3FIN THEN #Mx_ET07_3PRE := FALSE; END_IF;
END_REGION

REGION Network 38: ET07_2FIN
   RUNG wire#powerrail
      Contact( #Mx_ET07_2PRE )
      wire#w1
      Contact( #F_EnvMens_Mx )
      wire#w2
      S_SR(operand := #Mx_ET07_2FIN, r1 := #Mx_ET07_3PRE)
   END_RUNG
   RUNG wire#w1
      I_Contact( #pHsMx_2 )
   END_RUNG wire#w2
   // the same network as SCL:
   IF #Mx_ET07_2PRE AND (#F_EnvMens_Mx OR NOT #pHsMx_2) THEN
       #Mx_ET07_2FIN := TRUE;   // SR flip-flop
   END_IF;
   IF #Mx_ET07_3PRE THEN #Mx_ET07_2FIN := FALSE; END_IF;
END_REGION

REGION Network 39: ET07_2PRE
   RUNG wire#powerrail
      Contact( #Mx_ET07_1FIN )
      I_Contact( #F_EnvMens_Mx )
      S_SR(operand := #Mx_ET07_2PRE, r1 := #Mx_ET07_2FIN)
   END_RUNG
   // the same network as SCL:
   IF #Mx_ET07_1FIN AND NOT #F_EnvMens_Mx THEN
       #Mx_ET07_2PRE := TRUE;   // SR flip-flop
   END_IF;
   IF #Mx_ET07_2FIN THEN #Mx_ET07_2PRE := FALSE; END_IF;
END_REGION

REGION Network 40: ET07_1FIN
   RUNG wire#powerrail
      Contact( #Mx_ET07_1PRE )
      wire#w1
      Contact( #F_EnvMens_Mx )
      wire#w2
      I_Contact( #Mx_ET00 )
      S_SR(operand := #Mx_ET07_1FIN, r1 := #Mx_ET07_2PRE)
   END_RUNG
   RUNG wire#w1
      I_Contact( #pHsMx_1 )
   END_RUNG wire#w2
   // the same network as SCL:
   IF #Mx_ET07_1PRE AND (#F_EnvMens_Mx OR NOT #pHsMx_1) AND NOT #Mx_ET00 THEN
       #Mx_ET07_1FIN := TRUE;   // SR flip-flop
   END_IF;
   IF #Mx_ET07_2PRE THEN #Mx_ET07_1FIN := FALSE; END_IF;
END_REGION

REGION Network 41: ET07_1PRE
   RUNG wire#powerrail
      Contact( #Mx_ET00 )
      Contact( #EstadoZona.PerReset_CBx )
      wire#w1
      Contact( #pHsMx_1 )
      wire#w2
      S_SR(operand := #Mx_ET07_1PRE, r1 := #Mx_ET07_1FIN)
   END_RUNG
   RUNG wire#w1
      Contact( #pHsMx_2 )
   END_RUNG wire#w2
   RUNG wire#w1
      Contact( #pHsMx_3 )
   END_RUNG wire#w2
   RUNG wire#w1
      Contact( #pHsMx_4 )
   END_RUNG wire#w2
   // the same network as SCL:
   IF #Mx_ET00 AND #EstadoZona.PerReset_CBx AND (#pHsMx_1 OR #pHsMx_2 OR #pHsMx_3 OR #pHsMx_4) THEN
       #Mx_ET07_1PRE := TRUE;   // SR flip-flop
   END_IF;
   IF #Mx_ET07_1FIN THEN #Mx_ET07_1PRE := FALSE; END_IF;
END_REGION

REGION Network 42: ET42 - ACTIVACION DE PASARELA - VACIA LA MESA
   RUNG wire#powerrail
      Contact( #Mx_ET41 )
      wire#w1
      I_Contact( #MAnt_MSig_DesCargaAct )
      wire#w2
      I_Contact( #Mx_ET40 )
      S_SR(operand := #Mx_ET42, r1 := #Mx_ET01)
   END_RUNG
   RUNG wire#w1
      Contact( #FTF_MAnt_MSig )
   END_RUNG wire#w2
   // the same network as SCL:
   IF #Mx_ET41 AND (NOT #MAnt_MSig_DesCargaAct OR #FTF_MAnt_MSig) AND NOT #Mx_ET40 THEN
       #Mx_ET42 := TRUE;   // SR flip-flop
   END_IF;
   IF #Mx_ET01 THEN #Mx_ET42 := FALSE; END_IF;
END_REGION

REGION Network 43: ET41
   RUNG wire#powerrail
      Contact( #Mx_ET40 )
      Contact( #MAnt_MSig_DesCargaAct )
      Contact( #PTF_MAnt_MSig )
      Contact( #pHsMx_1 )
      I_Contact( #Mx_ET01 )
      S_SR(operand := #Mx_ET41, r1 := #Mx_ET42)
   END_RUNG
   // the same network as SCL:
   IF #Mx_ET40 AND #MAnt_MSig_DesCargaAct AND #PTF_MAnt_MSig AND #pHsMx_1 AND NOT #Mx_ET01 THEN
       #Mx_ET41 := TRUE;   // SR flip-flop
   END_IF;
   IF #Mx_ET42 THEN #Mx_ET41 := FALSE; END_IF;
END_REGION

REGION Network 44: ET40
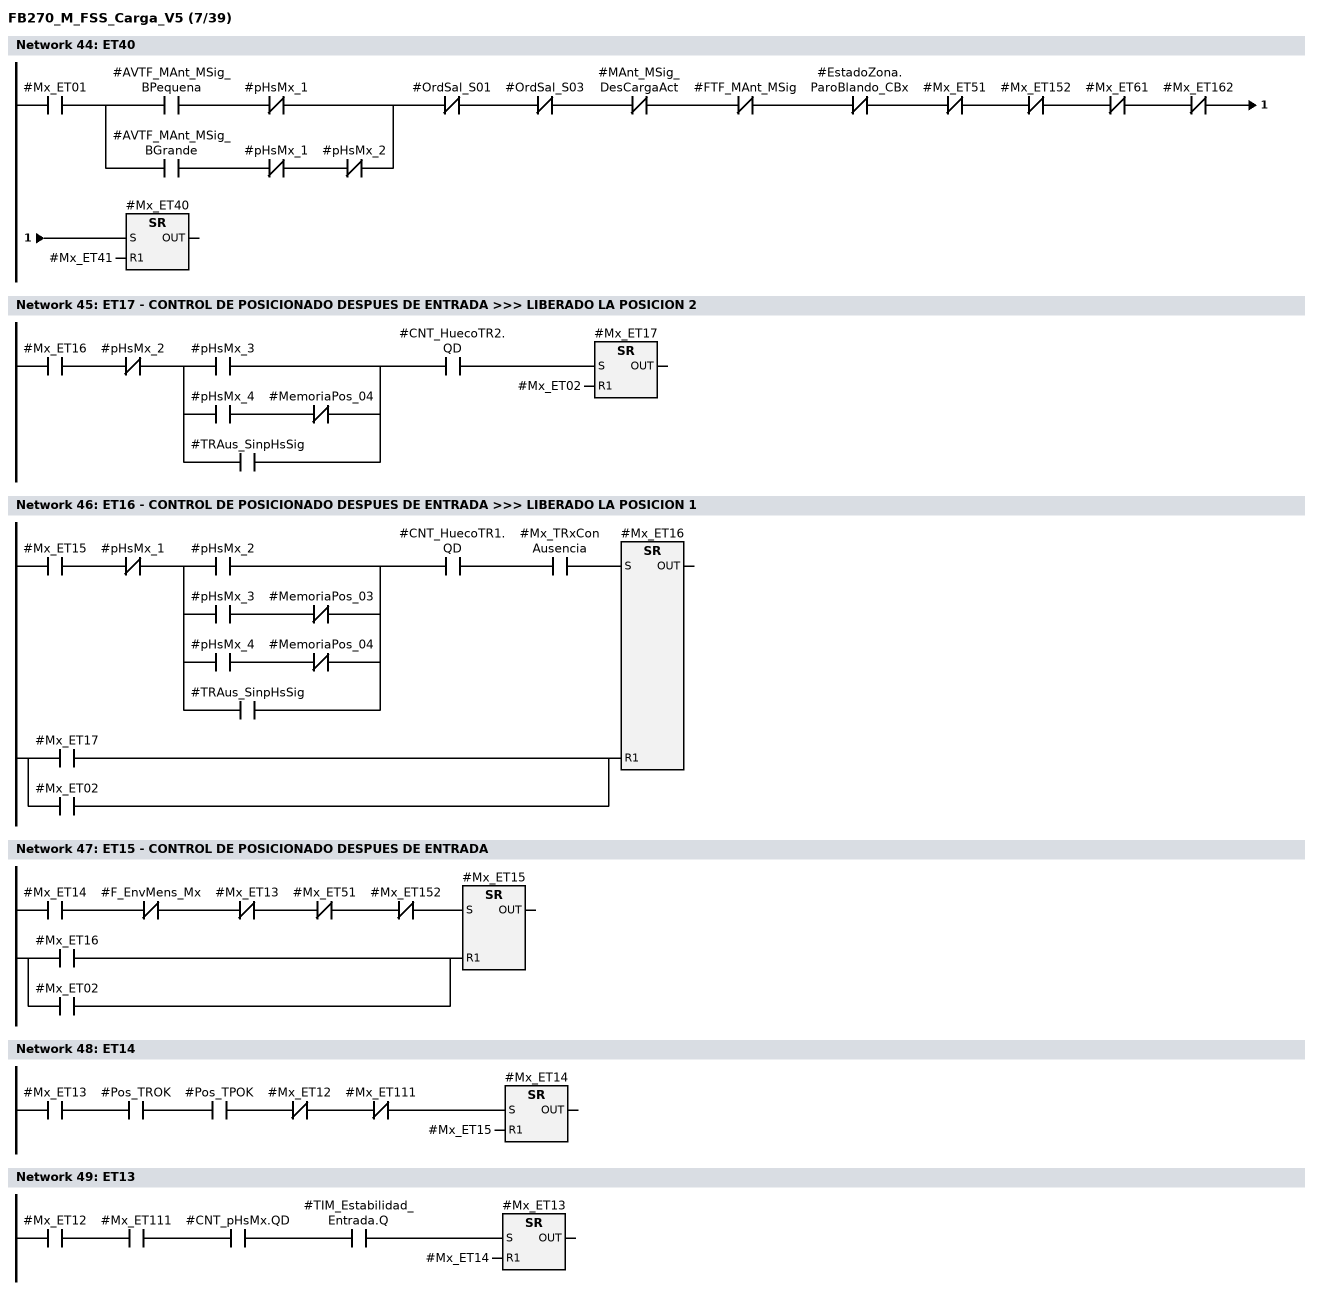
   RUNG wire#powerrail
      Contact( #Mx_ET01 )
      wire#w1
      Contact( #AVTF_MAnt_MSig_BPequena )
      I_Contact( #pHsMx_1 )
      wire#w2
      I_Contact( #OrdSal_S01 )
      I_Contact( #OrdSal_S03 )
      I_Contact( #MAnt_MSig_DesCargaAct )
      I_Contact( #FTF_MAnt_MSig )
      I_Contact( #EstadoZona.ParoBlando_CBx )
      I_Contact( #Mx_ET51 )
      I_Contact( #Mx_ET152 )
      I_Contact( #Mx_ET61 )
      I_Contact( #Mx_ET162 )
      S_SR(operand := #Mx_ET40, r1 := #Mx_ET41)
   END_RUNG
   RUNG wire#w1
      Contact( #AVTF_MAnt_MSig_BGrande )
      I_Contact( #pHsMx_1 )
      I_Contact( #pHsMx_2 )
   END_RUNG wire#w2
   // the same network as SCL:
   IF #Mx_ET01 AND ((#AVTF_MAnt_MSig_BPequena AND NOT #pHsMx_1) OR (#AVTF_MAnt_MSig_BGrande AND NOT #pHsMx_1 AND NOT #pHsMx_2)) AND NOT #OrdSal_S01 AND NOT #OrdSal_S03 AND NOT #MAnt_MSig_DesCargaAct AND NOT #FTF_MAnt_MSig AND NOT #EstadoZona.ParoBlando_CBx AND NOT #Mx_ET51 AND NOT #Mx_ET152 AND NOT #Mx_ET61 AND NOT #Mx_ET162 THEN
       #Mx_ET40 := TRUE;   // SR flip-flop
   END_IF;
   IF #Mx_ET41 THEN #Mx_ET40 := FALSE; END_IF;
END_REGION

REGION Network 45: ET17 - CONTROL DE POSICIONADO DESPUES DE ENTRADA >>> LIBERADO LA POSICION 2
   RUNG wire#powerrail
      Contact( #Mx_ET16 )
      I_Contact( #pHsMx_2 )
      wire#w1
      Contact( #pHsMx_3 )
      wire#w2
      Contact( #CNT_HuecoTR2.QD )
      S_SR(operand := #Mx_ET17, r1 := #Mx_ET02)
   END_RUNG
   RUNG wire#w1
      Contact( #pHsMx_4 )
      I_Contact( #MemoriaPos_04 )
   END_RUNG wire#w2
   RUNG wire#w1
      Contact( #TRAus_SinpHsSig )
   END_RUNG wire#w2
   // the same network as SCL:
   IF #Mx_ET16 AND NOT #pHsMx_2 AND (#pHsMx_3 OR (#pHsMx_4 AND NOT #MemoriaPos_04) OR #TRAus_SinpHsSig) AND #CNT_HuecoTR2.QD THEN
       #Mx_ET17 := TRUE;   // SR flip-flop
   END_IF;
   IF #Mx_ET02 THEN #Mx_ET17 := FALSE; END_IF;
END_REGION

REGION Network 46: ET16 - CONTROL DE POSICIONADO DESPUES DE ENTRADA >>> LIBERADO LA POSICION 1
   RUNG wire#powerrail
      Contact( #Mx_ET15 )
      I_Contact( #pHsMx_1 )
      wire#w1
      Contact( #pHsMx_2 )
      wire#w2
      Contact( #CNT_HuecoTR1.QD )
      Contact( #Mx_TRxConAusencia )
      S_SR(operand := #Mx_ET16, r1 := wire#w3)
   END_RUNG
   RUNG wire#w1
      Contact( #pHsMx_3 )
      I_Contact( #MemoriaPos_03 )
   END_RUNG wire#w2
   RUNG wire#w1
      Contact( #pHsMx_4 )
      I_Contact( #MemoriaPos_04 )
   END_RUNG wire#w2
   RUNG wire#w1
      Contact( #TRAus_SinpHsSig )
   END_RUNG wire#w2
   RUNG wire#powerrail
      Contact( #Mx_ET17 )
   END_RUNG wire#w3
   RUNG wire#powerrail
      Contact( #Mx_ET02 )
   END_RUNG wire#w3
   // the same network as SCL:
   IF #Mx_ET15 AND NOT #pHsMx_1 AND (#pHsMx_2 OR (#pHsMx_3 AND NOT #MemoriaPos_03) OR (#pHsMx_4 AND NOT #MemoriaPos_04) OR #TRAus_SinpHsSig) AND #CNT_HuecoTR1.QD AND #Mx_TRxConAusencia THEN
       #Mx_ET16 := TRUE;   // SR flip-flop
   END_IF;
   IF #Mx_ET17 OR #Mx_ET02 THEN #Mx_ET16 := FALSE; END_IF;
END_REGION

REGION Network 47: ET15 - CONTROL DE POSICIONADO DESPUES DE ENTRADA
   RUNG wire#powerrail
      Contact( #Mx_ET14 )
      I_Contact( #F_EnvMens_Mx )
      I_Contact( #Mx_ET13 )
      I_Contact( #Mx_ET51 )
      I_Contact( #Mx_ET152 )
      S_SR(operand := #Mx_ET15, r1 := wire#w1)
   END_RUNG
   RUNG wire#powerrail
      Contact( #Mx_ET16 )
   END_RUNG wire#w1
   RUNG wire#powerrail
      Contact( #Mx_ET02 )
   END_RUNG wire#w1
   // the same network as SCL:
   IF #Mx_ET14 AND NOT #F_EnvMens_Mx AND NOT #Mx_ET13 AND NOT #Mx_ET51 AND NOT #Mx_ET152 THEN
       #Mx_ET15 := TRUE;   // SR flip-flop
   END_IF;
   IF #Mx_ET16 OR #Mx_ET02 THEN #Mx_ET15 := FALSE; END_IF;
END_REGION

REGION Network 48: ET14
   RUNG wire#powerrail
      Contact( #Mx_ET13 )
      Contact( #Pos_TROK )
      Contact( #Pos_TPOK )
      I_Contact( #Mx_ET12 )
      I_Contact( #Mx_ET111 )
      S_SR(operand := #Mx_ET14, r1 := #Mx_ET15)
   END_RUNG
   // the same network as SCL:
   IF #Mx_ET13 AND #Pos_TROK AND #Pos_TPOK AND NOT #Mx_ET12 AND NOT #Mx_ET111 THEN
       #Mx_ET14 := TRUE;   // SR flip-flop
   END_IF;
   IF #Mx_ET15 THEN #Mx_ET14 := FALSE; END_IF;
END_REGION

REGION Network 49: ET13
   RUNG wire#powerrail
      Contact( #Mx_ET12 )
      Contact( #Mx_ET111 )
      Contact( #CNT_pHsMx.QD )
      Contact( #TIM_Estabilidad_Entrada.Q )
      S_SR(operand := #Mx_ET13, r1 := #Mx_ET14)
   END_RUNG
   // the same network as SCL:
   IF #Mx_ET12 AND #Mx_ET111 AND #CNT_pHsMx.QD AND #TIM_Estabilidad_Entrada.Q THEN
       #Mx_ET13 := TRUE;   // SR flip-flop
   END_IF;
   IF #Mx_ET14 THEN #Mx_ET13 := FALSE; END_IF;
END_REGION

REGION Network 50: ET111 - CONTROL CARGA MESA - MENSAJE DE PRESENCIA
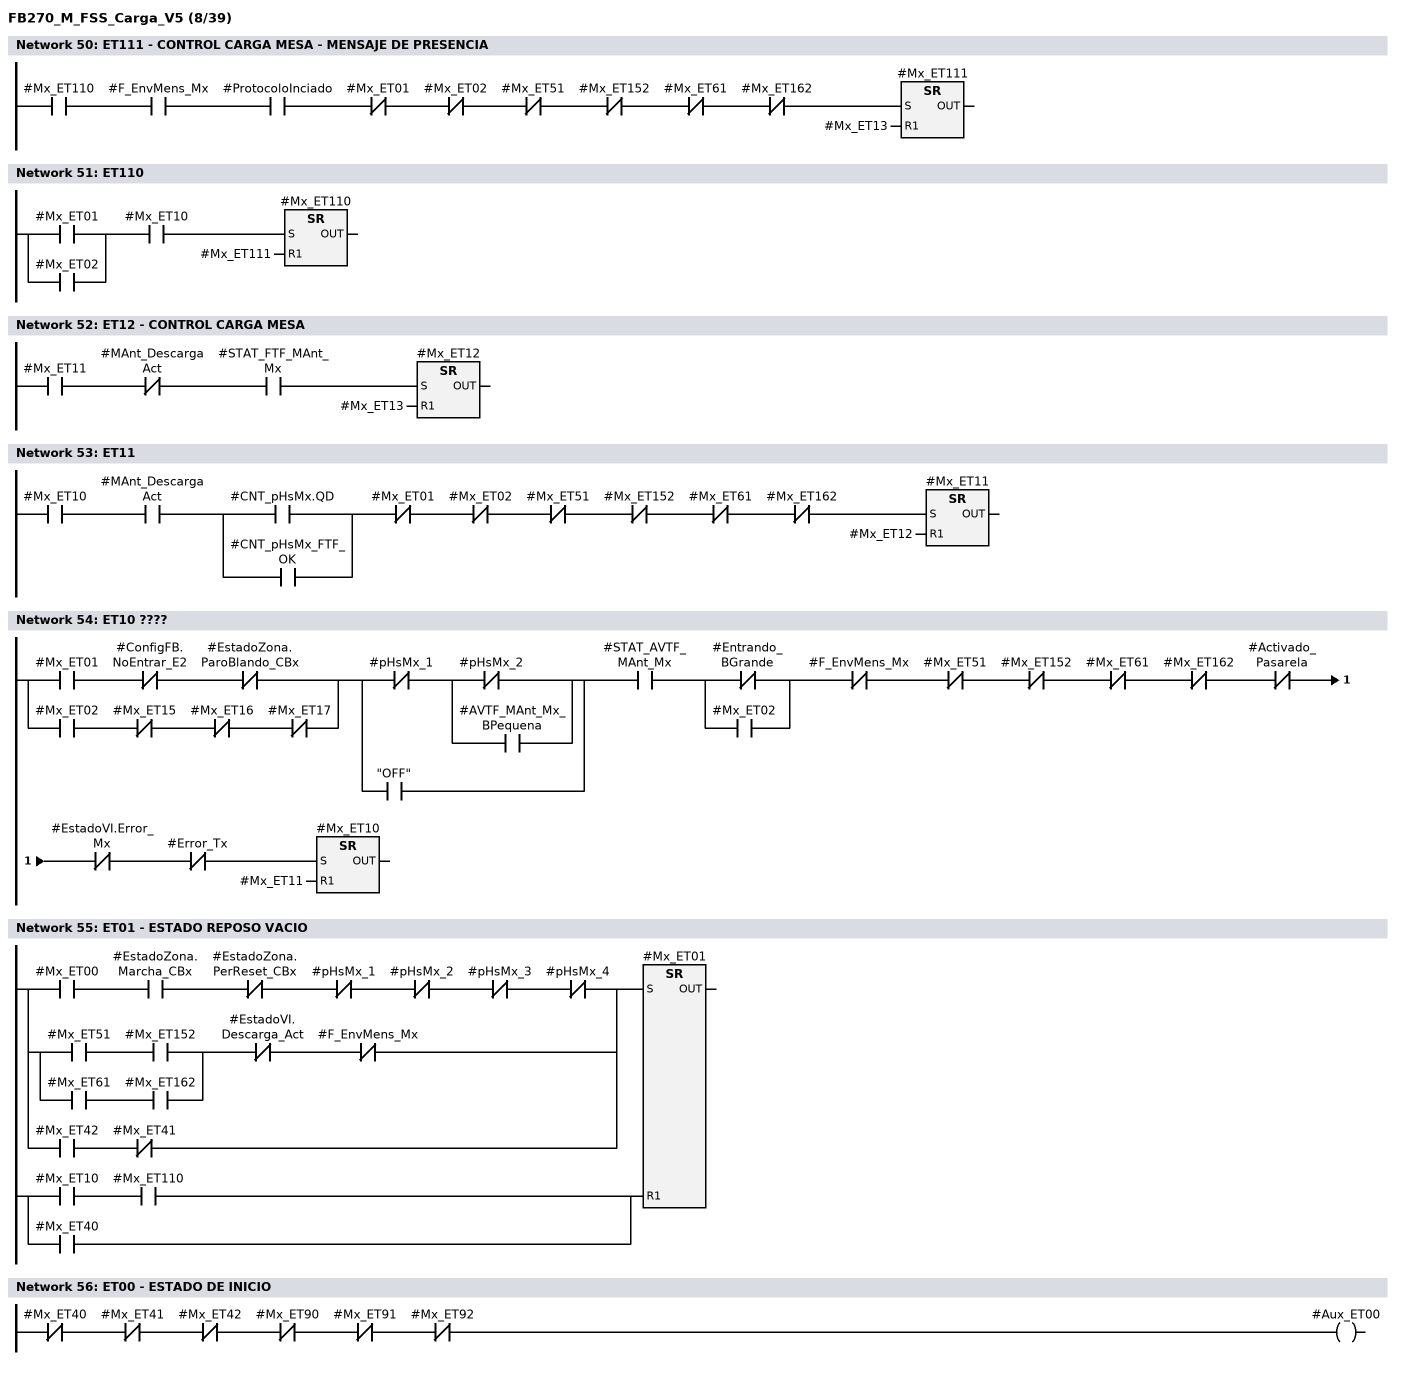
   RUNG wire#powerrail
      Contact( #Mx_ET110 )
      Contact( #F_EnvMens_Mx )
      Contact( #ProtocoloInciado )
      I_Contact( #Mx_ET01 )
      I_Contact( #Mx_ET02 )
      I_Contact( #Mx_ET51 )
      I_Contact( #Mx_ET152 )
      I_Contact( #Mx_ET61 )
      I_Contact( #Mx_ET162 )
      S_SR(operand := #Mx_ET111, r1 := #Mx_ET13)
   END_RUNG
   // the same network as SCL:
   IF #Mx_ET110 AND #F_EnvMens_Mx AND #ProtocoloInciado AND NOT #Mx_ET01 AND NOT #Mx_ET02 AND NOT #Mx_ET51 AND NOT #Mx_ET152 AND NOT #Mx_ET61 AND NOT #Mx_ET162 THEN
       #Mx_ET111 := TRUE;   // SR flip-flop
   END_IF;
   IF #Mx_ET13 THEN #Mx_ET111 := FALSE; END_IF;
END_REGION

REGION Network 51: ET110
   RUNG wire#powerrail
      Contact( #Mx_ET01 )
      wire#w1
      Contact( #Mx_ET10 )
      S_SR(operand := #Mx_ET110, r1 := #Mx_ET111)
   END_RUNG
   RUNG wire#powerrail
      Contact( #Mx_ET02 )
   END_RUNG wire#w1
   // the same network as SCL:
   IF (#Mx_ET01 OR #Mx_ET02) AND #Mx_ET10 THEN
       #Mx_ET110 := TRUE;   // SR flip-flop
   END_IF;
   IF #Mx_ET111 THEN #Mx_ET110 := FALSE; END_IF;
END_REGION

REGION Network 52: ET12 - CONTROL CARGA MESA
   RUNG wire#powerrail
      Contact( #Mx_ET11 )
      I_Contact( #MAnt_DescargaAct )
      Contact( #STAT_FTF_MAnt_Mx )
      S_SR(operand := #Mx_ET12, r1 := #Mx_ET13)
   END_RUNG
   // the same network as SCL:
   IF #Mx_ET11 AND NOT #MAnt_DescargaAct AND #STAT_FTF_MAnt_Mx THEN
       #Mx_ET12 := TRUE;   // SR flip-flop
   END_IF;
   IF #Mx_ET13 THEN #Mx_ET12 := FALSE; END_IF;
END_REGION

REGION Network 53: ET11
   RUNG wire#powerrail
      Contact( #Mx_ET10 )
      Contact( #MAnt_DescargaAct )
      wire#w1
      Contact( #CNT_pHsMx.QD )
      wire#w2
      I_Contact( #Mx_ET01 )
      I_Contact( #Mx_ET02 )
      I_Contact( #Mx_ET51 )
      I_Contact( #Mx_ET152 )
      I_Contact( #Mx_ET61 )
      I_Contact( #Mx_ET162 )
      S_SR(operand := #Mx_ET11, r1 := #Mx_ET12)
   END_RUNG
   RUNG wire#w1
      Contact( #CNT_pHsMx_FTF_OK )
   END_RUNG wire#w2
   // the same network as SCL:
   IF #Mx_ET10 AND #MAnt_DescargaAct AND (#CNT_pHsMx.QD OR #CNT_pHsMx_FTF_OK) AND NOT #Mx_ET01 AND NOT #Mx_ET02 AND NOT #Mx_ET51 AND NOT #Mx_ET152 AND NOT #Mx_ET61 AND NOT #Mx_ET162 THEN
       #Mx_ET11 := TRUE;   // SR flip-flop
   END_IF;
   IF #Mx_ET12 THEN #Mx_ET11 := FALSE; END_IF;
END_REGION

REGION Network 54: ET10 ????
   RUNG wire#powerrail
      Contact( #Mx_ET01 )
      I_Contact( #ConfigFB.NoEntrar_E2 )
      I_Contact( #EstadoZona.ParoBlando_CBx )
      wire#w1
      I_Contact( #pHsMx_1 )
      wire#w2
      I_Contact( #pHsMx_2 )
      wire#w3
      Contact( #STAT_AVTF_MAnt_Mx )
      wire#w4
      I_Contact( #Entrando_BGrande )
      wire#w5
      I_Contact( #F_EnvMens_Mx )
      I_Contact( #Mx_ET51 )
      I_Contact( #Mx_ET152 )
      I_Contact( #Mx_ET61 )
      I_Contact( #Mx_ET162 )
      I_Contact( #Activado_Pasarela )
      I_Contact( #EstadoVI.Error_Mx )
      I_Contact( #Error_Tx )
      S_SR(operand := #Mx_ET10, r1 := #Mx_ET11)
   END_RUNG
   RUNG wire#powerrail
      Contact( #Mx_ET02 )
      I_Contact( #Mx_ET15 )
      I_Contact( #Mx_ET16 )
      I_Contact( #Mx_ET17 )
   END_RUNG wire#w1
   RUNG wire#w2
      Contact( #AVTF_MAnt_Mx_BPequena )
   END_RUNG wire#w3
   RUNG wire#w1
      Contact( "OFF" )
   END_RUNG wire#w3
   RUNG wire#w4
      Contact( #Mx_ET02 )
   END_RUNG wire#w5
   // the same network as SCL:
   IF ((#Mx_ET01 AND NOT #ConfigFB.NoEntrar_E2 AND NOT #EstadoZona.ParoBlando_CBx) OR (#Mx_ET02 AND NOT #Mx_ET15 AND NOT #Mx_ET16 AND NOT #Mx_ET17)) AND ((NOT #pHsMx_1 AND (NOT #pHsMx_2 OR #AVTF_MAnt_Mx_BPequena)) OR "OFF") AND #STAT_AVTF_MAnt_Mx AND (NOT #Entrando_BGrande OR #Mx_ET02) AND NOT #F_EnvMens_Mx AND NOT #Mx_ET51 AND NOT #Mx_ET152 AND NOT #Mx_ET61 AND NOT #Mx_ET162 AND NOT #Activado_Pasarela AND NOT #EstadoVI.Error_Mx AND NOT #Error_Tx THEN
       #Mx_ET10 := TRUE;   // SR flip-flop
   END_IF;
   IF #Mx_ET11 THEN #Mx_ET10 := FALSE; END_IF;
END_REGION

REGION Network 55: ET01 - ESTADO REPOSO VACIO
   RUNG wire#powerrail
      Contact( #Mx_ET00 )
      Contact( #EstadoZona.Marcha_CBx )
      I_Contact( #EstadoZona.PerReset_CBx )
      I_Contact( #pHsMx_1 )
      I_Contact( #pHsMx_2 )
      I_Contact( #pHsMx_3 )
      I_Contact( #pHsMx_4 )
      wire#w1
      S_SR(operand := #Mx_ET01, r1 := wire#w3)
   END_RUNG
   RUNG wire#powerrail
      Contact( #Mx_ET51 )
      Contact( #Mx_ET152 )
      wire#w2
      I_Contact( #EstadoVI.Descarga_Act )
      I_Contact( #F_EnvMens_Mx )
   END_RUNG wire#w1
   RUNG wire#powerrail
      Contact( #Mx_ET61 )
      Contact( #Mx_ET162 )
   END_RUNG wire#w2
   RUNG wire#powerrail
      Contact( #Mx_ET42 )
      I_Contact( #Mx_ET41 )
   END_RUNG wire#w1
   RUNG wire#powerrail
      Contact( #Mx_ET10 )
      Contact( #Mx_ET110 )
   END_RUNG wire#w3
   RUNG wire#powerrail
      Contact( #Mx_ET40 )
   END_RUNG wire#w3
   // the same network as SCL:
   IF (#Mx_ET00 AND #EstadoZona.Marcha_CBx AND NOT #EstadoZona.PerReset_CBx AND NOT #pHsMx_1 AND NOT #pHsMx_2 AND NOT #pHsMx_3 AND NOT #pHsMx_4) OR (((#Mx_ET51 AND #Mx_ET152) OR (#Mx_ET61 AND #Mx_ET162)) AND NOT #EstadoVI.Descarga_Act AND NOT #F_EnvMens_Mx) OR (#Mx_ET42 AND NOT #Mx_ET41) THEN
       #Mx_ET01 := TRUE;   // SR flip-flop
   END_IF;
   IF (#Mx_ET10 AND #Mx_ET110) OR #Mx_ET40 THEN #Mx_ET01 := FALSE; END_IF;
END_REGION

REGION Network 56: ET00 - ESTADO DE INICIO
   RUNG wire#powerrail
      I_Contact( #Mx_ET40 )
      I_Contact( #Mx_ET41 )
      I_Contact( #Mx_ET42 )
      I_Contact( #Mx_ET90 )
      I_Contact( #Mx_ET91 )
      I_Contact( #Mx_ET92 )
      Coil( #Aux_ET00 )
   END_RUNG
   // the same network as SCL:
   #Aux_ET00 := NOT #Mx_ET40 AND NOT #Mx_ET41 AND NOT #Mx_ET42 AND NOT #Mx_ET90 AND NOT #Mx_ET91 AND NOT #Mx_ET92;
END_REGION

REGION Network 57: ----
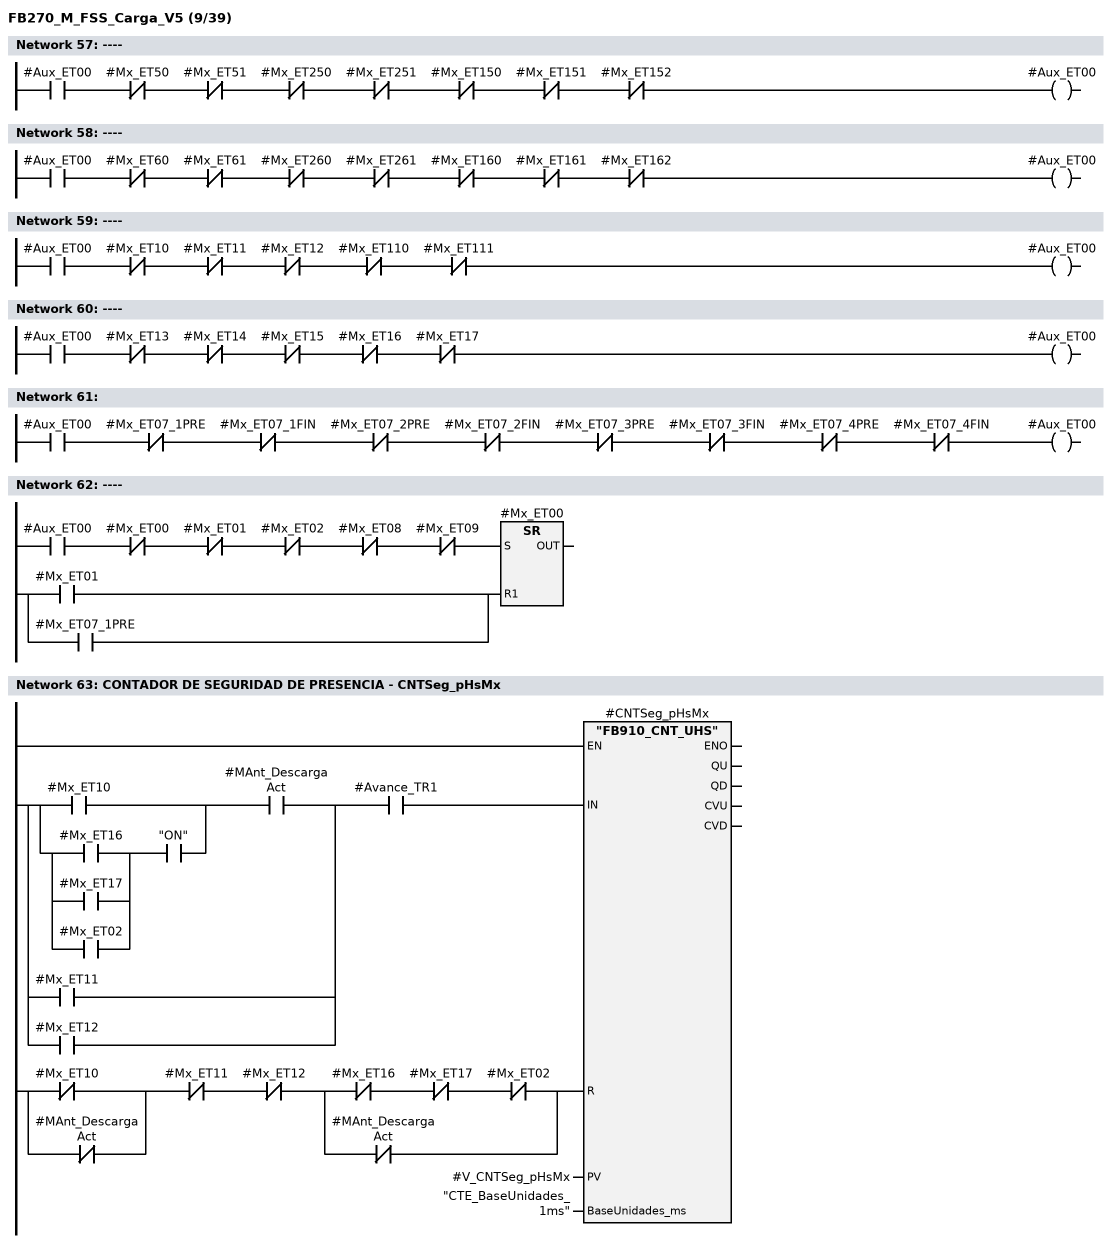
   RUNG wire#powerrail
      Contact( #Aux_ET00 )
      I_Contact( #Mx_ET50 )
      I_Contact( #Mx_ET51 )
      I_Contact( #Mx_ET250 )
      I_Contact( #Mx_ET251 )
      I_Contact( #Mx_ET150 )
      I_Contact( #Mx_ET151 )
      I_Contact( #Mx_ET152 )
      Coil( #Aux_ET00 )
   END_RUNG
   // the same network as SCL:
   #Aux_ET00 := #Aux_ET00 AND NOT #Mx_ET50 AND NOT #Mx_ET51 AND NOT #Mx_ET250 AND NOT #Mx_ET251 AND NOT #Mx_ET150 AND NOT #Mx_ET151 AND NOT #Mx_ET152;
END_REGION

REGION Network 58: ----
   RUNG wire#powerrail
      Contact( #Aux_ET00 )
      I_Contact( #Mx_ET60 )
      I_Contact( #Mx_ET61 )
      I_Contact( #Mx_ET260 )
      I_Contact( #Mx_ET261 )
      I_Contact( #Mx_ET160 )
      I_Contact( #Mx_ET161 )
      I_Contact( #Mx_ET162 )
      Coil( #Aux_ET00 )
   END_RUNG
   // the same network as SCL:
   #Aux_ET00 := #Aux_ET00 AND NOT #Mx_ET60 AND NOT #Mx_ET61 AND NOT #Mx_ET260 AND NOT #Mx_ET261 AND NOT #Mx_ET160 AND NOT #Mx_ET161 AND NOT #Mx_ET162;
END_REGION

REGION Network 59: ----
   RUNG wire#powerrail
      Contact( #Aux_ET00 )
      I_Contact( #Mx_ET10 )
      I_Contact( #Mx_ET11 )
      I_Contact( #Mx_ET12 )
      I_Contact( #Mx_ET110 )
      I_Contact( #Mx_ET111 )
      Coil( #Aux_ET00 )
   END_RUNG
   // the same network as SCL:
   #Aux_ET00 := #Aux_ET00 AND NOT #Mx_ET10 AND NOT #Mx_ET11 AND NOT #Mx_ET12 AND NOT #Mx_ET110 AND NOT #Mx_ET111;
END_REGION

REGION Network 60: ----
   RUNG wire#powerrail
      Contact( #Aux_ET00 )
      I_Contact( #Mx_ET13 )
      I_Contact( #Mx_ET14 )
      I_Contact( #Mx_ET15 )
      I_Contact( #Mx_ET16 )
      I_Contact( #Mx_ET17 )
      Coil( #Aux_ET00 )
   END_RUNG
   // the same network as SCL:
   #Aux_ET00 := #Aux_ET00 AND NOT #Mx_ET13 AND NOT #Mx_ET14 AND NOT #Mx_ET15 AND NOT #Mx_ET16 AND NOT #Mx_ET17;
END_REGION

REGION Network 61
   RUNG wire#powerrail
      Contact( #Aux_ET00 )
      I_Contact( #Mx_ET07_1PRE )
      I_Contact( #Mx_ET07_1FIN )
      I_Contact( #Mx_ET07_2PRE )
      I_Contact( #Mx_ET07_2FIN )
      I_Contact( #Mx_ET07_3PRE )
      I_Contact( #Mx_ET07_3FIN )
      I_Contact( #Mx_ET07_4PRE )
      I_Contact( #Mx_ET07_4FIN )
      Coil( #Aux_ET00 )
   END_RUNG
   // the same network as SCL:
   #Aux_ET00 := #Aux_ET00 AND NOT #Mx_ET07_1PRE AND NOT #Mx_ET07_1FIN AND NOT #Mx_ET07_2PRE AND NOT #Mx_ET07_2FIN AND NOT #Mx_ET07_3PRE AND NOT #Mx_ET07_3FIN AND NOT #Mx_ET07_4PRE AND NOT #Mx_ET07_4FIN;
END_REGION

REGION Network 62: ----
   RUNG wire#powerrail
      Contact( #Aux_ET00 )
      I_Contact( #Mx_ET00 )
      I_Contact( #Mx_ET01 )
      I_Contact( #Mx_ET02 )
      I_Contact( #Mx_ET08 )
      I_Contact( #Mx_ET09 )
      S_SR(operand := #Mx_ET00, r1 := wire#w1)
   END_RUNG
   RUNG wire#powerrail
      Contact( #Mx_ET01 )
   END_RUNG wire#w1
   RUNG wire#powerrail
      Contact( #Mx_ET07_1PRE )
   END_RUNG wire#w1
   // the same network as SCL:
   IF #Aux_ET00 AND NOT #Mx_ET00 AND NOT #Mx_ET01 AND NOT #Mx_ET02 AND NOT #Mx_ET08 AND NOT #Mx_ET09 THEN
       #Mx_ET00 := TRUE;   // SR flip-flop
   END_IF;
   IF #Mx_ET01 OR #Mx_ET07_1PRE THEN #Mx_ET00 := FALSE; END_IF;
END_REGION

